// TIA Portal V17 export
// export: Created 2025-07-01T14:26:04.7163189Z, ExportSetting WithDefaults, DisplayName Totally Integrated Automation Portal, DisplayVersion V17 Update 8, DisplayName TIA Portal Openness, DisplayVersion V17 Update 8, DisplayName TIA Portal Version Control Interface, DisplayVersion V17, DisplayName SINAMICS Startdrive Advanced, DisplayVersion V17 SP2, DisplayName SINAMICS Startdrive G110M, G120, G120C, G120D, G120P, G115D, DisplayVersion V17 SP2, DisplayName SINAMICS Startdrive G130, G150, S120, S150, SINAMICS MV, S210, DisplayVersion V17 SP2, DisplayName STEP 7 Professional, DisplayVersion V17 Update 8, DisplayName SINUMERIK ONE STEP 7 Toolbox, DisplayVersion V17 Update 12, DisplayName SINUMERIK ONE PLC Basic Program Plus, DisplayVersion V17 Update 12, DisplayName SINUMERIK 840D sl STEP 7 Toolbox, DisplayVersion V17 Update 12, DisplayName STEP 7 Safety, DisplayVersion V17 Update 6, DisplayName WinCC Advanced, DisplayVersion V17 Update 8
FUNCTION "FC1032_TEST_STOP_CLADDING" : Void   // FC1032, LAD
{ S7_Optimized_Access := 'FALSE' }
AUTHOR : ETXETAR
VERSION : 1.0
// stored: AutoNumber false, IsIECCheckEnabled false, SetENOAutomatically false, UDAEnableTagReadback false
   VAR_TEMP
      AUX_START_TEST_STOP : Bool;   // AUXILIARY START TEST STOP
      OPTION_ON : Bool;   // OPTION ON
      OPTION_OFF : Bool;   // OPTION OFF
      BRAKE_TEST_AXIS_X13 : Bool;   // BRAKE TEST AXIS X13
      BRAKE_TEST_AXIS_X23 : Bool;   // BRAKE TEST AXIS X23
      BRAKE_TEST_AXIS_W11 : Bool;   // BRAKE TEST AXIS W11
      BRAKE_TEST_AXIS_Z13 : Bool;   // BRAKE TEST AXIS Z13
      BRAKE_TEST_AXIS_Z14 : Bool;   // BRAKE TEST AXIS Z14
      BRAKE_TEST_AXIS_W21 : Bool;   // BRAKE TEST AXIS W21
      BRAKE_TEST_AXIS_Z23 : Bool;   // BRAKE TEST AXIS Z23
      BRAKE_TEST_AXIS_Z24 : Bool;   // BRAKE TEST AXIS Z24
      BRAKE_TEST_AXIS_C11 : Bool;   // BRAKE TEST AXIS C11
      BRAKE_TEST_AXIS_C12 : Bool;   // BRAKE TEST AXIS C12
      BRAKE_TEST_AXIS_C13 : Bool;   // BRAKE TEST AXIS C13
      BRAKE_TEST_AXIS_C14 : Bool;   // BRAKE TEST AXIS C14
      BRAKE_TEST_AXIS_C21 : Bool;   // BRAKE TEST AXIS C21
      BRAKE_TEST_AXIS_C22 : Bool;   // BRAKE TEST AXIS C22
      BRAKE_TEST_AXIS_C23 : Bool;   // BRAKE TEST AXIS C23
      BRAKE_TEST_AXIS_C24 : Bool;   // BRAKE TEST AXIS C24
      BRAKE_TEST_AXIS_C31 : Bool;   // BRAKE TEST AXISC31
   END_VAR
   VAR CONSTANT
      FC_NUMBER : DInt := 1032;
   END_VAR
   VAR_TEMP   // added for the SCL form of the ladder/FBD networks
      _w1 : Bool;
   END_VAR
BEGIN

REGION Network 1: OPTIONS OFF
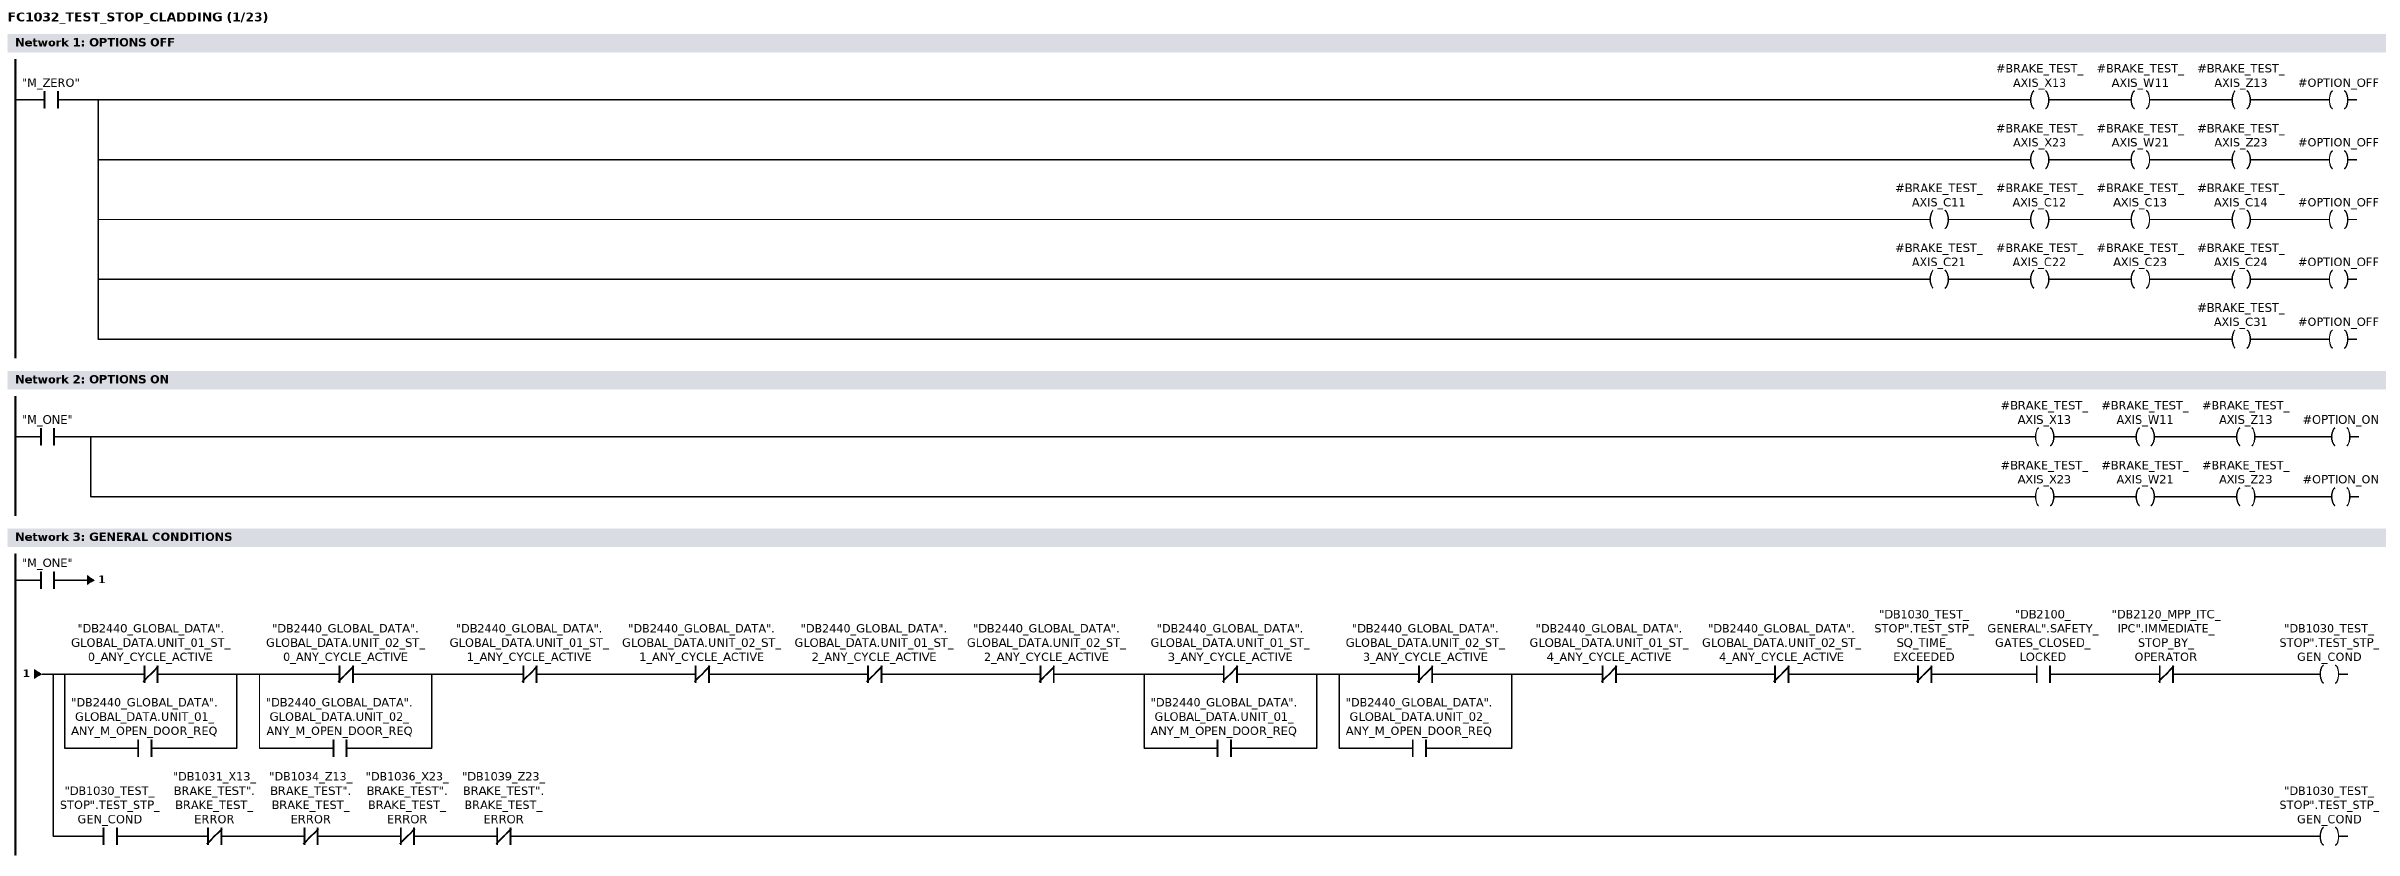
   RUNG wire#powerrail
      Contact( "M_ZERO" )
      wire#w1
      Coil( #BRAKE_TEST_AXIS_X13 )
      Coil( #BRAKE_TEST_AXIS_W11 )
      Coil( #BRAKE_TEST_AXIS_Z13 )
      Coil( #OPTION_OFF )
   END_RUNG
   RUNG wire#w1
      Coil( #BRAKE_TEST_AXIS_X23 )
      Coil( #BRAKE_TEST_AXIS_W21 )
      Coil( #BRAKE_TEST_AXIS_Z23 )
      Coil( #OPTION_OFF )
   END_RUNG
   RUNG wire#w1
      Coil( #BRAKE_TEST_AXIS_C11 )
      Coil( #BRAKE_TEST_AXIS_C12 )
      Coil( #BRAKE_TEST_AXIS_C13 )
      Coil( #BRAKE_TEST_AXIS_C14 )
      Coil( #OPTION_OFF )
   END_RUNG
   RUNG wire#w1
      Coil( #BRAKE_TEST_AXIS_C21 )
      Coil( #BRAKE_TEST_AXIS_C22 )
      Coil( #BRAKE_TEST_AXIS_C23 )
      Coil( #BRAKE_TEST_AXIS_C24 )
      Coil( #OPTION_OFF )
   END_RUNG
   RUNG wire#w1
      Coil( #BRAKE_TEST_AXIS_C31 )
      Coil( #OPTION_OFF )
   END_RUNG
   // the same network as SCL:
   #BRAKE_TEST_AXIS_X13 := "M_ZERO";
   #BRAKE_TEST_AXIS_W11 := "M_ZERO";
   #BRAKE_TEST_AXIS_Z13 := "M_ZERO";
   #OPTION_OFF := "M_ZERO";
   #BRAKE_TEST_AXIS_X23 := "M_ZERO";
   #BRAKE_TEST_AXIS_W21 := "M_ZERO";
   #BRAKE_TEST_AXIS_Z23 := "M_ZERO";
   #OPTION_OFF := "M_ZERO";
   #BRAKE_TEST_AXIS_C11 := "M_ZERO";
   #BRAKE_TEST_AXIS_C12 := "M_ZERO";
   #BRAKE_TEST_AXIS_C13 := "M_ZERO";
   #BRAKE_TEST_AXIS_C14 := "M_ZERO";
   #OPTION_OFF := "M_ZERO";
   #BRAKE_TEST_AXIS_C21 := "M_ZERO";
   #BRAKE_TEST_AXIS_C22 := "M_ZERO";
   #BRAKE_TEST_AXIS_C23 := "M_ZERO";
   #BRAKE_TEST_AXIS_C24 := "M_ZERO";
   #OPTION_OFF := "M_ZERO";
   #BRAKE_TEST_AXIS_C31 := "M_ZERO";
   #OPTION_OFF := "M_ZERO";
END_REGION

REGION Network 2: OPTIONS ON
   RUNG wire#powerrail
      Contact( "M_ONE" )
      wire#w1
      Coil( #BRAKE_TEST_AXIS_X13 )
      Coil( #BRAKE_TEST_AXIS_W11 )
      Coil( #BRAKE_TEST_AXIS_Z13 )
      Coil( #OPTION_ON )
   END_RUNG
   RUNG wire#w1
      Coil( #BRAKE_TEST_AXIS_X23 )
      Coil( #BRAKE_TEST_AXIS_W21 )
      Coil( #BRAKE_TEST_AXIS_Z23 )
      Coil( #OPTION_ON )
   END_RUNG
   // the same network as SCL:
   #BRAKE_TEST_AXIS_X13 := "M_ONE";
   #BRAKE_TEST_AXIS_W11 := "M_ONE";
   #BRAKE_TEST_AXIS_Z13 := "M_ONE";
   #OPTION_ON := "M_ONE";
   #BRAKE_TEST_AXIS_X23 := "M_ONE";
   #BRAKE_TEST_AXIS_W21 := "M_ONE";
   #BRAKE_TEST_AXIS_Z23 := "M_ONE";
   #OPTION_ON := "M_ONE";
END_REGION

REGION Network 3: GENERAL CONDITIONS
   RUNG wire#powerrail
      Contact( "M_ONE" )
      wire#w1
      I_Contact( "DB2440_GLOBAL_DATA".GLOBAL_DATA.UNIT_01_ST_0_ANY_CYCLE_ACTIVE )
      wire#w2
      I_Contact( "DB2440_GLOBAL_DATA".GLOBAL_DATA.UNIT_02_ST_0_ANY_CYCLE_ACTIVE )
      wire#w3
      I_Contact( "DB2440_GLOBAL_DATA".GLOBAL_DATA.UNIT_01_ST_1_ANY_CYCLE_ACTIVE )
      I_Contact( "DB2440_GLOBAL_DATA".GLOBAL_DATA.UNIT_02_ST_1_ANY_CYCLE_ACTIVE )
      I_Contact( "DB2440_GLOBAL_DATA".GLOBAL_DATA.UNIT_01_ST_2_ANY_CYCLE_ACTIVE )
      I_Contact( "DB2440_GLOBAL_DATA".GLOBAL_DATA.UNIT_02_ST_2_ANY_CYCLE_ACTIVE )
      wire#w4
      I_Contact( "DB2440_GLOBAL_DATA".GLOBAL_DATA.UNIT_01_ST_3_ANY_CYCLE_ACTIVE )
      wire#w5
      I_Contact( "DB2440_GLOBAL_DATA".GLOBAL_DATA.UNIT_02_ST_3_ANY_CYCLE_ACTIVE )
      wire#w6
      I_Contact( "DB2440_GLOBAL_DATA".GLOBAL_DATA.UNIT_01_ST_4_ANY_CYCLE_ACTIVE )
      I_Contact( "DB2440_GLOBAL_DATA".GLOBAL_DATA.UNIT_02_ST_4_ANY_CYCLE_ACTIVE )
      I_Contact( "DB1030_TEST_STOP".TEST_STP_SQ_TIME_EXCEEDED )
      Contact( "DB2100_GENERAL".SAFETY_GATES_CLOSED_LOCKED )
      I_Contact( "DB2120_MPP_ITC_IPC".IMMEDIATE_STOP_BY_OPERATOR )
      Coil( "DB1030_TEST_STOP".TEST_STP_GEN_COND )
   END_RUNG
   RUNG wire#w1
      Contact( "DB2440_GLOBAL_DATA".GLOBAL_DATA.UNIT_01_ANY_M_OPEN_DOOR_REQ )
   END_RUNG wire#w2
   RUNG wire#w2
      Contact( "DB2440_GLOBAL_DATA".GLOBAL_DATA.UNIT_02_ANY_M_OPEN_DOOR_REQ )
   END_RUNG wire#w3
   RUNG wire#w4
      Contact( "DB2440_GLOBAL_DATA".GLOBAL_DATA.UNIT_01_ANY_M_OPEN_DOOR_REQ )
   END_RUNG wire#w5
   RUNG wire#w5
      Contact( "DB2440_GLOBAL_DATA".GLOBAL_DATA.UNIT_02_ANY_M_OPEN_DOOR_REQ )
   END_RUNG wire#w6
   RUNG wire#w1
      Contact( "DB1030_TEST_STOP".TEST_STP_GEN_COND )
      I_Contact( "DB1031_X13_BRAKE_TEST".BRAKE_TEST_ERROR )
      I_Contact( "DB1034_Z13_BRAKE_TEST".BRAKE_TEST_ERROR )
      I_Contact( "DB1036_X23_BRAKE_TEST".BRAKE_TEST_ERROR )
      I_Contact( "DB1039_Z23_BRAKE_TEST".BRAKE_TEST_ERROR )
      Coil( "DB1030_TEST_STOP".TEST_STP_GEN_COND )
   END_RUNG
   // the same network as SCL:
   "DB1030_TEST_STOP".TEST_STP_GEN_COND := "M_ONE" AND (NOT "DB2440_GLOBAL_DATA".GLOBAL_DATA.UNIT_01_ST_0_ANY_CYCLE_ACTIVE OR "DB2440_GLOBAL_DATA".GLOBAL_DATA.UNIT_01_ANY_M_OPEN_DOOR_REQ) AND (NOT "DB2440_GLOBAL_DATA".GLOBAL_DATA.UNIT_02_ST_0_ANY_CYCLE_ACTIVE OR "DB2440_GLOBAL_DATA".GLOBAL_DATA.UNIT_02_ANY_M_OPEN_DOOR_REQ) AND NOT "DB2440_GLOBAL_DATA".GLOBAL_DATA.UNIT_01_ST_1_ANY_CYCLE_ACTIVE AND NOT "DB2440_GLOBAL_DATA".GLOBAL_DATA.UNIT_02_ST_1_ANY_CYCLE_ACTIVE AND NOT "DB2440_GLOBAL_DATA".GLOBAL_DATA.UNIT_01_ST_2_ANY_CYCLE_ACTIVE AND NOT "DB2440_GLOBAL_DATA".GLOBAL_DATA.UNIT_02_ST_2_ANY_CYCLE_ACTIVE AND (NOT "DB2440_GLOBAL_DATA".GLOBAL_DATA.UNIT_01_ST_3_ANY_CYCLE_ACTIVE OR "DB2440_GLOBAL_DATA".GLOBAL_DATA.UNIT_01_ANY_M_OPEN_DOOR_REQ) AND (NOT "DB2440_GLOBAL_DATA".GLOBAL_DATA.UNIT_02_ST_3_ANY_CYCLE_ACTIVE OR "DB2440_GLOBAL_DATA".GLOBAL_DATA.UNIT_02_ANY_M_OPEN_DOOR_REQ) AND NOT "DB2440_GLOBAL_DATA".GLOBAL_DATA.UNIT_01_ST_4_ANY_CYCLE_ACTIVE AND NOT "DB2440_GLOBAL_DATA".GLOBAL_DATA.UNIT_02_ST_4_ANY_CYCLE_ACTIVE AND NOT "DB1030_TEST_STOP".TEST_STP_SQ_TIME_EXCEEDED AND "DB2100_GENERAL".SAFETY_GATES_CLOSED_LOCKED AND NOT "DB2120_MPP_ITC_IPC".IMMEDIATE_STOP_BY_OPERATOR;
   "DB1030_TEST_STOP".TEST_STP_GEN_COND := "M_ONE" AND "DB1030_TEST_STOP".TEST_STP_GEN_COND AND NOT "DB1031_X13_BRAKE_TEST".BRAKE_TEST_ERROR AND NOT "DB1034_Z13_BRAKE_TEST".BRAKE_TEST_ERROR AND NOT "DB1036_X23_BRAKE_TEST".BRAKE_TEST_ERROR AND NOT "DB1039_Z23_BRAKE_TEST".BRAKE_TEST_ERROR;
END_REGION

REGION Network 4: INITIAL CONDITIONS
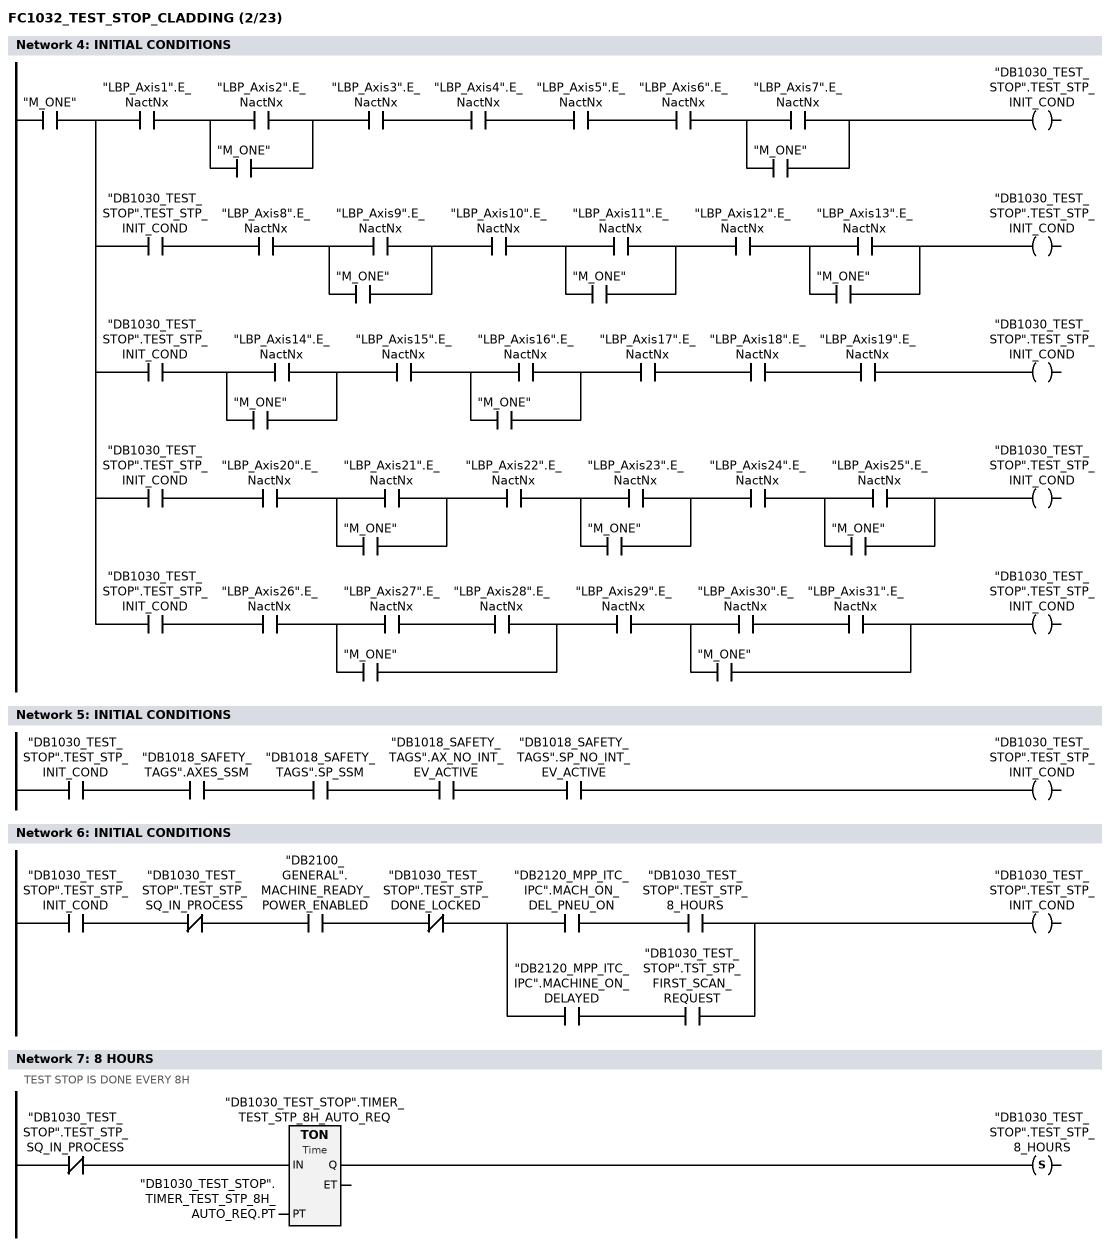
   RUNG wire#powerrail
      Contact( "M_ONE" )
      wire#w1
      Contact( "LBP_Axis1".E_NactNx )
      wire#w2
      Contact( "LBP_Axis2".E_NactNx )
      wire#w3
      Contact( "LBP_Axis3".E_NactNx )
      Contact( "LBP_Axis4".E_NactNx )
      Contact( "LBP_Axis5".E_NactNx )
      Contact( "LBP_Axis6".E_NactNx )
      wire#w4
      Contact( "LBP_Axis7".E_NactNx )
      wire#w5
      Coil( "DB1030_TEST_STOP".TEST_STP_INIT_COND )
   END_RUNG
   RUNG wire#w2
      Contact( "M_ONE" )
   END_RUNG wire#w3
   RUNG wire#w4
      Contact( "M_ONE" )
   END_RUNG wire#w5
   RUNG wire#w1
      Contact( "DB1030_TEST_STOP".TEST_STP_INIT_COND )
      Contact( "LBP_Axis8".E_NactNx )
      wire#w6
      Contact( "LBP_Axis9".E_NactNx )
      wire#w7
      Contact( "LBP_Axis10".E_NactNx )
      wire#w8
      Contact( "LBP_Axis11".E_NactNx )
      wire#w9
      Contact( "LBP_Axis12".E_NactNx )
      wire#w10
      Contact( "LBP_Axis13".E_NactNx )
      wire#w11
      Coil( "DB1030_TEST_STOP".TEST_STP_INIT_COND )
   END_RUNG
   RUNG wire#w6
      Contact( "M_ONE" )
   END_RUNG wire#w7
   RUNG wire#w8
      Contact( "M_ONE" )
   END_RUNG wire#w9
   RUNG wire#w10
      Contact( "M_ONE" )
   END_RUNG wire#w11
   RUNG wire#w1
      Contact( "DB1030_TEST_STOP".TEST_STP_INIT_COND )
      wire#w12
      Contact( "LBP_Axis14".E_NactNx )
      wire#w13
      Contact( "LBP_Axis15".E_NactNx )
      wire#w14
      Contact( "LBP_Axis16".E_NactNx )
      wire#w15
      Contact( "LBP_Axis17".E_NactNx )
      Contact( "LBP_Axis18".E_NactNx )
      Contact( "LBP_Axis19".E_NactNx )
      Coil( "DB1030_TEST_STOP".TEST_STP_INIT_COND )
   END_RUNG
   RUNG wire#w12
      Contact( "M_ONE" )
   END_RUNG wire#w13
   RUNG wire#w14
      Contact( "M_ONE" )
   END_RUNG wire#w15
   RUNG wire#w1
      Contact( "DB1030_TEST_STOP".TEST_STP_INIT_COND )
      Contact( "LBP_Axis20".E_NactNx )
      wire#w16
      Contact( "LBP_Axis21".E_NactNx )
      wire#w17
      Contact( "LBP_Axis22".E_NactNx )
      wire#w18
      Contact( "LBP_Axis23".E_NactNx )
      wire#w19
      Contact( "LBP_Axis24".E_NactNx )
      wire#w20
      Contact( "LBP_Axis25".E_NactNx )
      wire#w21
      Coil( "DB1030_TEST_STOP".TEST_STP_INIT_COND )
   END_RUNG
   RUNG wire#w16
      Contact( "M_ONE" )
   END_RUNG wire#w17
   RUNG wire#w18
      Contact( "M_ONE" )
   END_RUNG wire#w19
   RUNG wire#w20
      Contact( "M_ONE" )
   END_RUNG wire#w21
   RUNG wire#w1
      Contact( "DB1030_TEST_STOP".TEST_STP_INIT_COND )
      Contact( "LBP_Axis26".E_NactNx )
      wire#w22
      Contact( "LBP_Axis27".E_NactNx )
      Contact( "LBP_Axis28".E_NactNx )
      wire#w23
      Contact( "LBP_Axis29".E_NactNx )
      wire#w24
      Contact( "LBP_Axis30".E_NactNx )
      Contact( "LBP_Axis31".E_NactNx )
      wire#w25
      Coil( "DB1030_TEST_STOP".TEST_STP_INIT_COND )
   END_RUNG
   RUNG wire#w22
      Contact( "M_ONE" )
   END_RUNG wire#w23
   RUNG wire#w24
      Contact( "M_ONE" )
   END_RUNG wire#w25
   // the same network as SCL:
   "DB1030_TEST_STOP".TEST_STP_INIT_COND := "M_ONE" AND "LBP_Axis1".E_NactNx AND ("LBP_Axis2".E_NactNx OR "M_ONE") AND "LBP_Axis3".E_NactNx AND "LBP_Axis4".E_NactNx AND "LBP_Axis5".E_NactNx AND "LBP_Axis6".E_NactNx AND ("LBP_Axis7".E_NactNx OR "M_ONE");
   "DB1030_TEST_STOP".TEST_STP_INIT_COND := "M_ONE" AND "DB1030_TEST_STOP".TEST_STP_INIT_COND AND "LBP_Axis8".E_NactNx AND ("LBP_Axis9".E_NactNx OR "M_ONE") AND "LBP_Axis10".E_NactNx AND ("LBP_Axis11".E_NactNx OR "M_ONE") AND "LBP_Axis12".E_NactNx AND ("LBP_Axis13".E_NactNx OR "M_ONE");
   "DB1030_TEST_STOP".TEST_STP_INIT_COND := "M_ONE" AND "DB1030_TEST_STOP".TEST_STP_INIT_COND AND ("LBP_Axis14".E_NactNx OR "M_ONE") AND "LBP_Axis15".E_NactNx AND ("LBP_Axis16".E_NactNx OR "M_ONE") AND "LBP_Axis17".E_NactNx AND "LBP_Axis18".E_NactNx AND "LBP_Axis19".E_NactNx;
   "DB1030_TEST_STOP".TEST_STP_INIT_COND := "M_ONE" AND "DB1030_TEST_STOP".TEST_STP_INIT_COND AND "LBP_Axis20".E_NactNx AND ("LBP_Axis21".E_NactNx OR "M_ONE") AND "LBP_Axis22".E_NactNx AND ("LBP_Axis23".E_NactNx OR "M_ONE") AND "LBP_Axis24".E_NactNx AND ("LBP_Axis25".E_NactNx OR "M_ONE");
   "DB1030_TEST_STOP".TEST_STP_INIT_COND := "M_ONE" AND "DB1030_TEST_STOP".TEST_STP_INIT_COND AND "LBP_Axis26".E_NactNx AND (("LBP_Axis27".E_NactNx AND "LBP_Axis28".E_NactNx) OR "M_ONE") AND "LBP_Axis29".E_NactNx AND (("LBP_Axis30".E_NactNx AND "LBP_Axis31".E_NactNx) OR "M_ONE");
END_REGION

REGION Network 5: INITIAL CONDITIONS
   RUNG wire#powerrail
      Contact( "DB1030_TEST_STOP".TEST_STP_INIT_COND )
      Contact( "DB1018_SAFETY_TAGS".AXES_SSM )
      Contact( "DB1018_SAFETY_TAGS".SP_SSM )
      Contact( "DB1018_SAFETY_TAGS".AX_NO_INT_EV_ACTIVE )
      Contact( "DB1018_SAFETY_TAGS".SP_NO_INT_EV_ACTIVE )
      Coil( "DB1030_TEST_STOP".TEST_STP_INIT_COND )
   END_RUNG
   // the same network as SCL:
   "DB1030_TEST_STOP".TEST_STP_INIT_COND := "DB1030_TEST_STOP".TEST_STP_INIT_COND AND "DB1018_SAFETY_TAGS".AXES_SSM AND "DB1018_SAFETY_TAGS".SP_SSM AND "DB1018_SAFETY_TAGS".AX_NO_INT_EV_ACTIVE AND "DB1018_SAFETY_TAGS".SP_NO_INT_EV_ACTIVE;
END_REGION

REGION Network 6: INITIAL CONDITIONS
   RUNG wire#powerrail
      Contact( "DB1030_TEST_STOP".TEST_STP_INIT_COND )
      I_Contact( "DB1030_TEST_STOP".TEST_STP_SQ_IN_PROCESS )
      Contact( "DB2100_GENERAL".MACHINE_READY_POWER_ENABLED )
      I_Contact( "DB1030_TEST_STOP".TEST_STP_DONE_LOCKED )
      wire#w1
      Contact( "DB2120_MPP_ITC_IPC".MACH_ON_DEL_PNEU_ON )
      Contact( "DB1030_TEST_STOP".TEST_STP_8_HOURS )
      wire#w2
      Coil( "DB1030_TEST_STOP".TEST_STP_INIT_COND )
   END_RUNG
   RUNG wire#w1
      Contact( "DB2120_MPP_ITC_IPC".MACHINE_ON_DELAYED )
      Contact( "DB1030_TEST_STOP".TST_STP_FIRST_SCAN_REQUEST )
   END_RUNG wire#w2
   // the same network as SCL:
   "DB1030_TEST_STOP".TEST_STP_INIT_COND := "DB1030_TEST_STOP".TEST_STP_INIT_COND AND NOT "DB1030_TEST_STOP".TEST_STP_SQ_IN_PROCESS AND "DB2100_GENERAL".MACHINE_READY_POWER_ENABLED AND NOT "DB1030_TEST_STOP".TEST_STP_DONE_LOCKED AND (("DB2120_MPP_ITC_IPC".MACH_ON_DEL_PNEU_ON AND "DB1030_TEST_STOP".TEST_STP_8_HOURS) OR ("DB2120_MPP_ITC_IPC".MACHINE_ON_DELAYED AND "DB1030_TEST_STOP".TST_STP_FIRST_SCAN_REQUEST));
END_REGION

REGION Network 7: 8 HOURS
   // TEST STOP IS DONE EVERY 8H
   RUNG wire#powerrail
      I_Contact( "DB1030_TEST_STOP".TEST_STP_SQ_IN_PROCESS )
      { S7_Templates := "time_type := Time" } "DB1030_TEST_STOP".TIMER_TEST_STP_8H_AUTO_REQ.TON(pt := "DB1030_TEST_STOP".TIMER_TEST_STP_8H_AUTO_REQ.PT, et =>)
      S_Coil( "DB1030_TEST_STOP".TEST_STP_8_HOURS )
   END_RUNG
   // the same network as SCL:
   "DB1030_TEST_STOP".TIMER_TEST_STP_8H_AUTO_REQ.TON(IN := NOT "DB1030_TEST_STOP".TEST_STP_SQ_IN_PROCESS,
                           PT := "DB1030_TEST_STOP".TIMER_TEST_STP_8H_AUTO_REQ.PT);
   IF "DB1030_TEST_STOP".TIMER_TEST_STP_8H_AUTO_REQ.Q THEN
       "DB1030_TEST_STOP".TEST_STP_8_HOURS := TRUE;
   END_IF;
END_REGION

REGION Network 8: START REQUEST
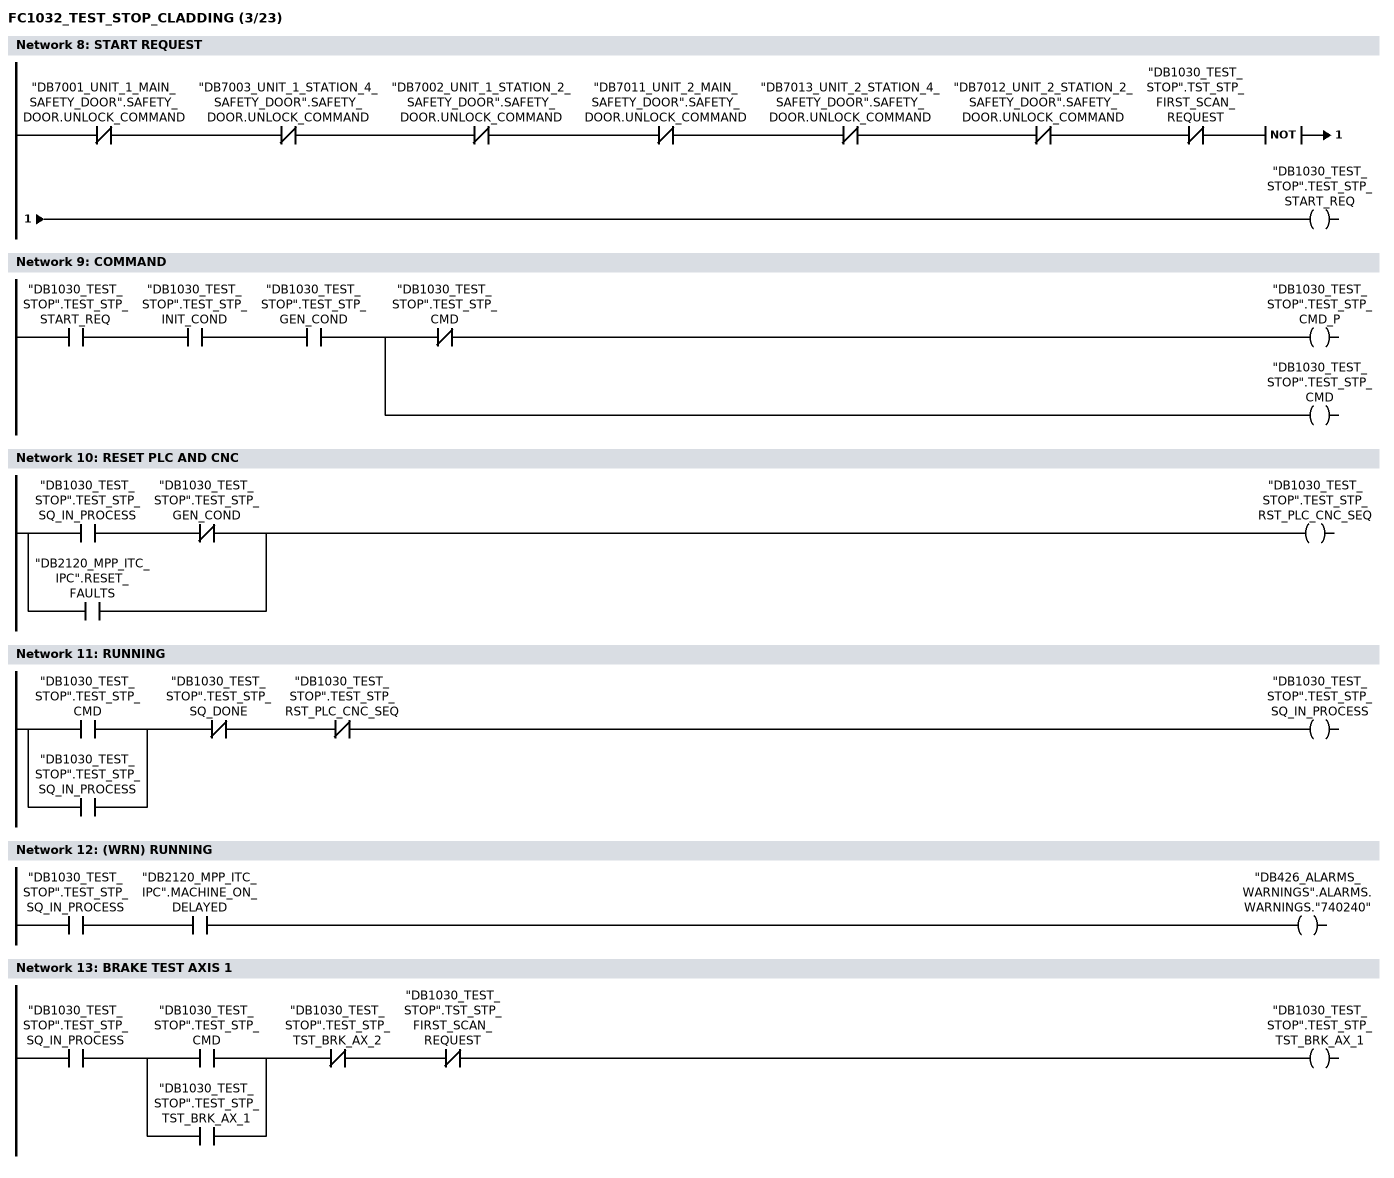
   RUNG wire#powerrail
      I_Contact( "DB7001_UNIT_1_MAIN_SAFETY_DOOR".SAFETY_DOOR.UNLOCK_COMMAND )
      I_Contact( "DB7003_UNIT_1_STATION_4_SAFETY_DOOR".SAFETY_DOOR.UNLOCK_COMMAND )
      I_Contact( "DB7002_UNIT_1_STATION_2_SAFETY_DOOR".SAFETY_DOOR.UNLOCK_COMMAND )
      I_Contact( "DB7011_UNIT_2_MAIN_SAFETY_DOOR".SAFETY_DOOR.UNLOCK_COMMAND )
      I_Contact( "DB7013_UNIT_2_STATION_4_SAFETY_DOOR".SAFETY_DOOR.UNLOCK_COMMAND )
      I_Contact( "DB7012_UNIT_2_STATION_2_SAFETY_DOOR".SAFETY_DOOR.UNLOCK_COMMAND )
      I_Contact( "DB1030_TEST_STOP".TST_STP_FIRST_SCAN_REQUEST )
      Not()
      Coil( "DB1030_TEST_STOP".TEST_STP_START_REQ )
   END_RUNG
   // the same network as SCL:
   "DB1030_TEST_STOP".TEST_STP_START_REQ := NOT (NOT "DB7001_UNIT_1_MAIN_SAFETY_DOOR".SAFETY_DOOR.UNLOCK_COMMAND AND NOT "DB7003_UNIT_1_STATION_4_SAFETY_DOOR".SAFETY_DOOR.UNLOCK_COMMAND AND NOT "DB7002_UNIT_1_STATION_2_SAFETY_DOOR".SAFETY_DOOR.UNLOCK_COMMAND AND NOT "DB7011_UNIT_2_MAIN_SAFETY_DOOR".SAFETY_DOOR.UNLOCK_COMMAND AND NOT "DB7013_UNIT_2_STATION_4_SAFETY_DOOR".SAFETY_DOOR.UNLOCK_COMMAND AND NOT "DB7012_UNIT_2_STATION_2_SAFETY_DOOR".SAFETY_DOOR.UNLOCK_COMMAND AND NOT "DB1030_TEST_STOP".TST_STP_FIRST_SCAN_REQUEST);
END_REGION

REGION Network 9: COMMAND
   RUNG wire#powerrail
      Contact( "DB1030_TEST_STOP".TEST_STP_START_REQ )
      Contact( "DB1030_TEST_STOP".TEST_STP_INIT_COND )
      Contact( "DB1030_TEST_STOP".TEST_STP_GEN_COND )
      wire#w1
      I_Contact( "DB1030_TEST_STOP".TEST_STP_CMD )
      Coil( "DB1030_TEST_STOP".TEST_STP_CMD_P )
   END_RUNG
   RUNG wire#w1
      Coil( "DB1030_TEST_STOP".TEST_STP_CMD )
   END_RUNG
   // the same network as SCL:
   #_w1 := "DB1030_TEST_STOP".TEST_STP_START_REQ AND "DB1030_TEST_STOP".TEST_STP_INIT_COND AND "DB1030_TEST_STOP".TEST_STP_GEN_COND;
   "DB1030_TEST_STOP".TEST_STP_CMD_P := #_w1 AND NOT "DB1030_TEST_STOP".TEST_STP_CMD;
   "DB1030_TEST_STOP".TEST_STP_CMD := #_w1;
END_REGION

REGION Network 10: RESET PLC AND CNC
   RUNG wire#powerrail
      Contact( "DB1030_TEST_STOP".TEST_STP_SQ_IN_PROCESS )
      I_Contact( "DB1030_TEST_STOP".TEST_STP_GEN_COND )
      wire#w1
      Coil( "DB1030_TEST_STOP".TEST_STP_RST_PLC_CNC_SEQ )
   END_RUNG
   RUNG wire#powerrail
      Contact( "DB2120_MPP_ITC_IPC".RESET_FAULTS )
   END_RUNG wire#w1
   // the same network as SCL:
   "DB1030_TEST_STOP".TEST_STP_RST_PLC_CNC_SEQ := ("DB1030_TEST_STOP".TEST_STP_SQ_IN_PROCESS AND NOT "DB1030_TEST_STOP".TEST_STP_GEN_COND) OR "DB2120_MPP_ITC_IPC".RESET_FAULTS;
END_REGION

REGION Network 11: RUNNING
   RUNG wire#powerrail
      Contact( "DB1030_TEST_STOP".TEST_STP_CMD )
      wire#w1
      I_Contact( "DB1030_TEST_STOP".TEST_STP_SQ_DONE )
      I_Contact( "DB1030_TEST_STOP".TEST_STP_RST_PLC_CNC_SEQ )
      Coil( "DB1030_TEST_STOP".TEST_STP_SQ_IN_PROCESS )
   END_RUNG
   RUNG wire#powerrail
      Contact( "DB1030_TEST_STOP".TEST_STP_SQ_IN_PROCESS )
   END_RUNG wire#w1
   // the same network as SCL:
   "DB1030_TEST_STOP".TEST_STP_SQ_IN_PROCESS := ("DB1030_TEST_STOP".TEST_STP_CMD OR "DB1030_TEST_STOP".TEST_STP_SQ_IN_PROCESS) AND NOT "DB1030_TEST_STOP".TEST_STP_SQ_DONE AND NOT "DB1030_TEST_STOP".TEST_STP_RST_PLC_CNC_SEQ;
END_REGION

REGION Network 12: (WRN) RUNNING
   RUNG wire#powerrail
      Contact( "DB1030_TEST_STOP".TEST_STP_SQ_IN_PROCESS )
      Contact( "DB2120_MPP_ITC_IPC".MACHINE_ON_DELAYED )
      Coil( "DB426_ALARMS_WARNINGS".ALARMS.WARNINGS."740240" )
   END_RUNG
   // the same network as SCL:
   "DB426_ALARMS_WARNINGS".ALARMS.WARNINGS."740240" := "DB1030_TEST_STOP".TEST_STP_SQ_IN_PROCESS AND "DB2120_MPP_ITC_IPC".MACHINE_ON_DELAYED;
END_REGION

REGION Network 13: BRAKE TEST AXIS 1
   RUNG wire#powerrail
      Contact( "DB1030_TEST_STOP".TEST_STP_SQ_IN_PROCESS )
      wire#w1
      Contact( "DB1030_TEST_STOP".TEST_STP_CMD )
      wire#w2
      I_Contact( "DB1030_TEST_STOP".TEST_STP_TST_BRK_AX_2 )
      I_Contact( "DB1030_TEST_STOP".TST_STP_FIRST_SCAN_REQUEST )
      Coil( "DB1030_TEST_STOP".TEST_STP_TST_BRK_AX_1 )
   END_RUNG
   RUNG wire#w1
      Contact( "DB1030_TEST_STOP".TEST_STP_TST_BRK_AX_1 )
   END_RUNG wire#w2
   // the same network as SCL:
   "DB1030_TEST_STOP".TEST_STP_TST_BRK_AX_1 := "DB1030_TEST_STOP".TEST_STP_SQ_IN_PROCESS AND ("DB1030_TEST_STOP".TEST_STP_CMD OR "DB1030_TEST_STOP".TEST_STP_TST_BRK_AX_1) AND NOT "DB1030_TEST_STOP".TEST_STP_TST_BRK_AX_2 AND NOT "DB1030_TEST_STOP".TST_STP_FIRST_SCAN_REQUEST;
END_REGION

REGION Network 14: CALL FB1031 BRAKE TEST AXIS 1
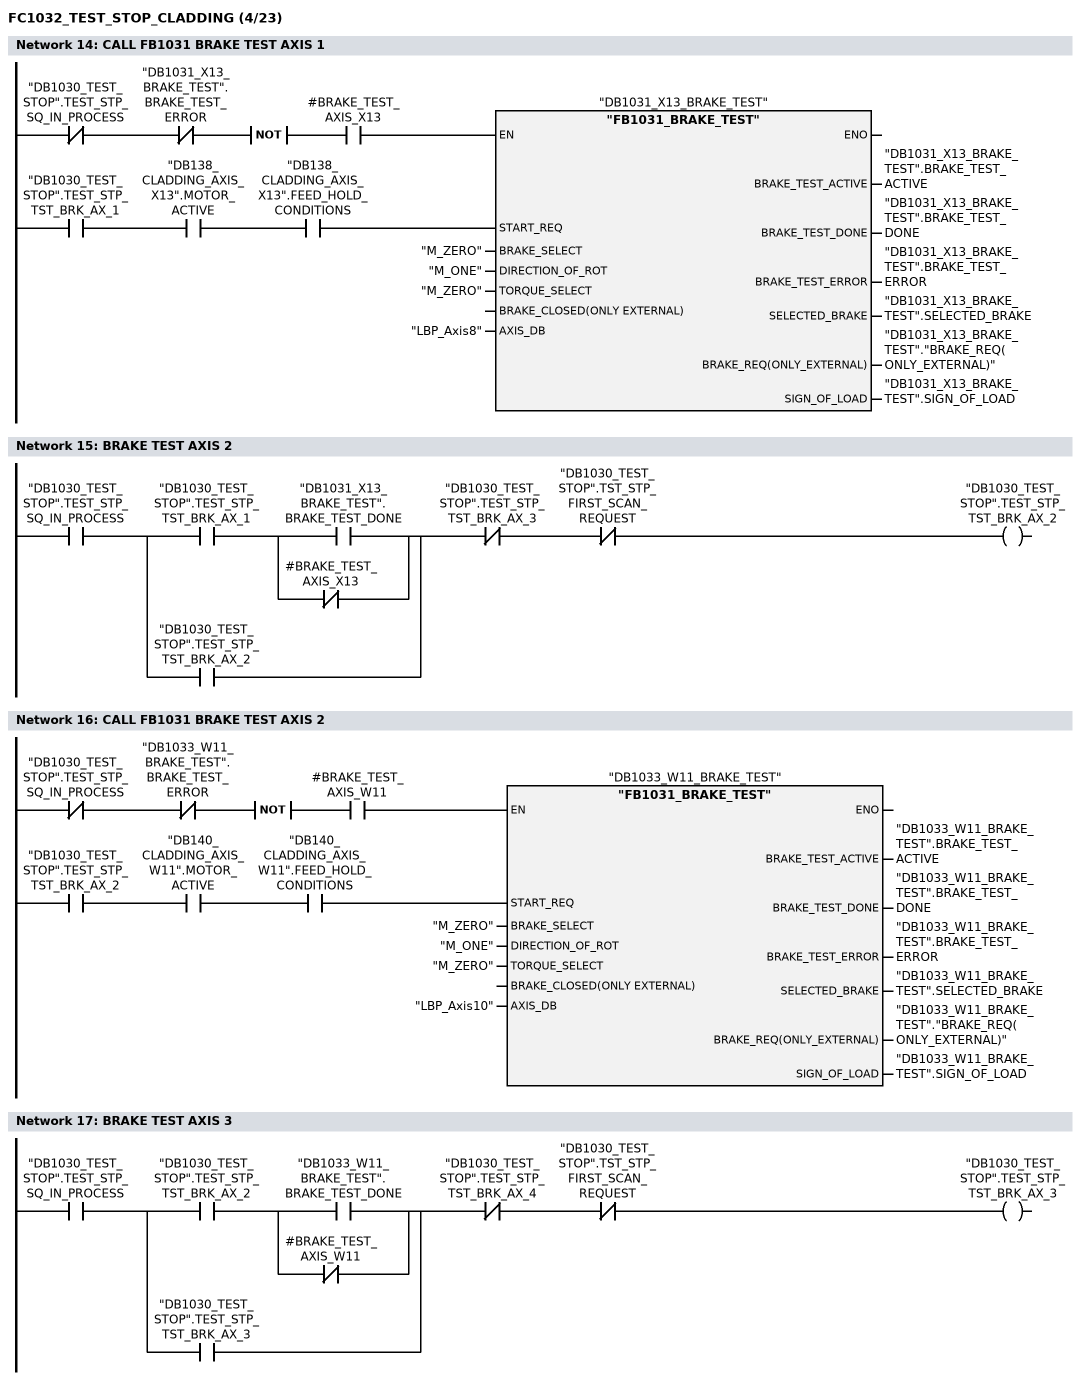
   RUNG wire#powerrail
      I_Contact( "DB1030_TEST_STOP".TEST_STP_SQ_IN_PROCESS )
      I_Contact( "DB1031_X13_BRAKE_TEST".BRAKE_TEST_ERROR )
      Not()
      Contact( #BRAKE_TEST_AXIS_X13 )
      "DB1031_X13_BRAKE_TEST"(START_REQ := wire#w1, BRAKE_SELECT := "M_ZERO", DIRECTION_OF_ROT := "M_ONE", TORQUE_SELECT := "M_ZERO", "BRAKE_CLOSED(ONLY EXTERNAL)" :=, AXIS_DB := "LBP_Axis8", BRAKE_TEST_ACTIVE => "DB1031_X13_BRAKE_TEST".BRAKE_TEST_ACTIVE, BRAKE_TEST_DONE => "DB1031_X13_BRAKE_TEST".BRAKE_TEST_DONE, BRAKE_TEST_ERROR => "DB1031_X13_BRAKE_TEST".BRAKE_TEST_ERROR, SELECTED_BRAKE => "DB1031_X13_BRAKE_TEST".SELECTED_BRAKE, "BRAKE_REQ(ONLY_EXTERNAL)" => "DB1031_X13_BRAKE_TEST"."BRAKE_REQ(ONLY_EXTERNAL)", SIGN_OF_LOAD => "DB1031_X13_BRAKE_TEST".SIGN_OF_LOAD)
   END_RUNG
   RUNG wire#powerrail
      Contact( "DB1030_TEST_STOP".TEST_STP_TST_BRK_AX_1 )
      Contact( "DB138_CLADDING_AXIS_X13".MOTOR_ACTIVE )
      Contact( "DB138_CLADDING_AXIS_X13".FEED_HOLD_CONDITIONS )
   END_RUNG wire#w1
   // the same network as SCL:
   IF NOT (NOT "DB1030_TEST_STOP".TEST_STP_SQ_IN_PROCESS AND NOT "DB1031_X13_BRAKE_TEST".BRAKE_TEST_ERROR) AND #BRAKE_TEST_AXIS_X13 THEN
       "DB1031_X13_BRAKE_TEST"(START_REQ := "DB1030_TEST_STOP".TEST_STP_TST_BRK_AX_1 AND "DB138_CLADDING_AXIS_X13".MOTOR_ACTIVE AND "DB138_CLADDING_AXIS_X13".FEED_HOLD_CONDITIONS,   // "FB1031_BRAKE_TEST"
                               BRAKE_SELECT := "M_ZERO",
                               DIRECTION_OF_ROT := "M_ONE",
                               TORQUE_SELECT := "M_ZERO",
                               AXIS_DB := "LBP_Axis8",
                               BRAKE_TEST_ACTIVE => "DB1031_X13_BRAKE_TEST".BRAKE_TEST_ACTIVE,
                               BRAKE_TEST_DONE => "DB1031_X13_BRAKE_TEST".BRAKE_TEST_DONE,
                               BRAKE_TEST_ERROR => "DB1031_X13_BRAKE_TEST".BRAKE_TEST_ERROR,
                               SELECTED_BRAKE => "DB1031_X13_BRAKE_TEST".SELECTED_BRAKE,
                               "BRAKE_REQ(ONLY_EXTERNAL)" => "DB1031_X13_BRAKE_TEST"."BRAKE_REQ(ONLY_EXTERNAL)",
                               SIGN_OF_LOAD => "DB1031_X13_BRAKE_TEST".SIGN_OF_LOAD);
   END_IF;
END_REGION

REGION Network 15: BRAKE TEST AXIS 2
   RUNG wire#powerrail
      Contact( "DB1030_TEST_STOP".TEST_STP_SQ_IN_PROCESS )
      wire#w1
      Contact( "DB1030_TEST_STOP".TEST_STP_TST_BRK_AX_1 )
      wire#w2
      Contact( "DB1031_X13_BRAKE_TEST".BRAKE_TEST_DONE )
      wire#w3
      I_Contact( "DB1030_TEST_STOP".TEST_STP_TST_BRK_AX_3 )
      I_Contact( "DB1030_TEST_STOP".TST_STP_FIRST_SCAN_REQUEST )
      Coil( "DB1030_TEST_STOP".TEST_STP_TST_BRK_AX_2 )
   END_RUNG
   RUNG wire#w2
      I_Contact( #BRAKE_TEST_AXIS_X13 )
   END_RUNG wire#w3
   RUNG wire#w1
      Contact( "DB1030_TEST_STOP".TEST_STP_TST_BRK_AX_2 )
   END_RUNG wire#w3
   // the same network as SCL:
   "DB1030_TEST_STOP".TEST_STP_TST_BRK_AX_2 := "DB1030_TEST_STOP".TEST_STP_SQ_IN_PROCESS AND (("DB1030_TEST_STOP".TEST_STP_TST_BRK_AX_1 AND ("DB1031_X13_BRAKE_TEST".BRAKE_TEST_DONE OR NOT #BRAKE_TEST_AXIS_X13)) OR "DB1030_TEST_STOP".TEST_STP_TST_BRK_AX_2) AND NOT "DB1030_TEST_STOP".TEST_STP_TST_BRK_AX_3 AND NOT "DB1030_TEST_STOP".TST_STP_FIRST_SCAN_REQUEST;
END_REGION

REGION Network 16: CALL FB1031 BRAKE TEST AXIS 2
   RUNG wire#powerrail
      I_Contact( "DB1030_TEST_STOP".TEST_STP_SQ_IN_PROCESS )
      I_Contact( "DB1033_W11_BRAKE_TEST".BRAKE_TEST_ERROR )
      Not()
      Contact( #BRAKE_TEST_AXIS_W11 )
      "DB1033_W11_BRAKE_TEST"(START_REQ := wire#w1, BRAKE_SELECT := "M_ZERO", DIRECTION_OF_ROT := "M_ONE", TORQUE_SELECT := "M_ZERO", "BRAKE_CLOSED(ONLY EXTERNAL)" :=, AXIS_DB := "LBP_Axis10", BRAKE_TEST_ACTIVE => "DB1033_W11_BRAKE_TEST".BRAKE_TEST_ACTIVE, BRAKE_TEST_DONE => "DB1033_W11_BRAKE_TEST".BRAKE_TEST_DONE, BRAKE_TEST_ERROR => "DB1033_W11_BRAKE_TEST".BRAKE_TEST_ERROR, SELECTED_BRAKE => "DB1033_W11_BRAKE_TEST".SELECTED_BRAKE, "BRAKE_REQ(ONLY_EXTERNAL)" => "DB1033_W11_BRAKE_TEST"."BRAKE_REQ(ONLY_EXTERNAL)", SIGN_OF_LOAD => "DB1033_W11_BRAKE_TEST".SIGN_OF_LOAD)
   END_RUNG
   RUNG wire#powerrail
      Contact( "DB1030_TEST_STOP".TEST_STP_TST_BRK_AX_2 )
      Contact( "DB140_CLADDING_AXIS_W11".MOTOR_ACTIVE )
      Contact( "DB140_CLADDING_AXIS_W11".FEED_HOLD_CONDITIONS )
   END_RUNG wire#w1
   // the same network as SCL:
   IF NOT (NOT "DB1030_TEST_STOP".TEST_STP_SQ_IN_PROCESS AND NOT "DB1033_W11_BRAKE_TEST".BRAKE_TEST_ERROR) AND #BRAKE_TEST_AXIS_W11 THEN
       "DB1033_W11_BRAKE_TEST"(START_REQ := "DB1030_TEST_STOP".TEST_STP_TST_BRK_AX_2 AND "DB140_CLADDING_AXIS_W11".MOTOR_ACTIVE AND "DB140_CLADDING_AXIS_W11".FEED_HOLD_CONDITIONS,   // "FB1031_BRAKE_TEST"
                               BRAKE_SELECT := "M_ZERO",
                               DIRECTION_OF_ROT := "M_ONE",
                               TORQUE_SELECT := "M_ZERO",
                               AXIS_DB := "LBP_Axis10",
                               BRAKE_TEST_ACTIVE => "DB1033_W11_BRAKE_TEST".BRAKE_TEST_ACTIVE,
                               BRAKE_TEST_DONE => "DB1033_W11_BRAKE_TEST".BRAKE_TEST_DONE,
                               BRAKE_TEST_ERROR => "DB1033_W11_BRAKE_TEST".BRAKE_TEST_ERROR,
                               SELECTED_BRAKE => "DB1033_W11_BRAKE_TEST".SELECTED_BRAKE,
                               "BRAKE_REQ(ONLY_EXTERNAL)" => "DB1033_W11_BRAKE_TEST"."BRAKE_REQ(ONLY_EXTERNAL)",
                               SIGN_OF_LOAD => "DB1033_W11_BRAKE_TEST".SIGN_OF_LOAD);
   END_IF;
END_REGION

REGION Network 17: BRAKE TEST AXIS 3
   RUNG wire#powerrail
      Contact( "DB1030_TEST_STOP".TEST_STP_SQ_IN_PROCESS )
      wire#w1
      Contact( "DB1030_TEST_STOP".TEST_STP_TST_BRK_AX_2 )
      wire#w2
      Contact( "DB1033_W11_BRAKE_TEST".BRAKE_TEST_DONE )
      wire#w3
      I_Contact( "DB1030_TEST_STOP".TEST_STP_TST_BRK_AX_4 )
      I_Contact( "DB1030_TEST_STOP".TST_STP_FIRST_SCAN_REQUEST )
      Coil( "DB1030_TEST_STOP".TEST_STP_TST_BRK_AX_3 )
   END_RUNG
   RUNG wire#w2
      I_Contact( #BRAKE_TEST_AXIS_W11 )
   END_RUNG wire#w3
   RUNG wire#w1
      Contact( "DB1030_TEST_STOP".TEST_STP_TST_BRK_AX_3 )
   END_RUNG wire#w3
   // the same network as SCL:
   "DB1030_TEST_STOP".TEST_STP_TST_BRK_AX_3 := "DB1030_TEST_STOP".TEST_STP_SQ_IN_PROCESS AND (("DB1030_TEST_STOP".TEST_STP_TST_BRK_AX_2 AND ("DB1033_W11_BRAKE_TEST".BRAKE_TEST_DONE OR NOT #BRAKE_TEST_AXIS_W11)) OR "DB1030_TEST_STOP".TEST_STP_TST_BRK_AX_3) AND NOT "DB1030_TEST_STOP".TEST_STP_TST_BRK_AX_4 AND NOT "DB1030_TEST_STOP".TST_STP_FIRST_SCAN_REQUEST;
END_REGION

REGION Network 18: CALL FB1031 BRAKE TEST AXIS 3
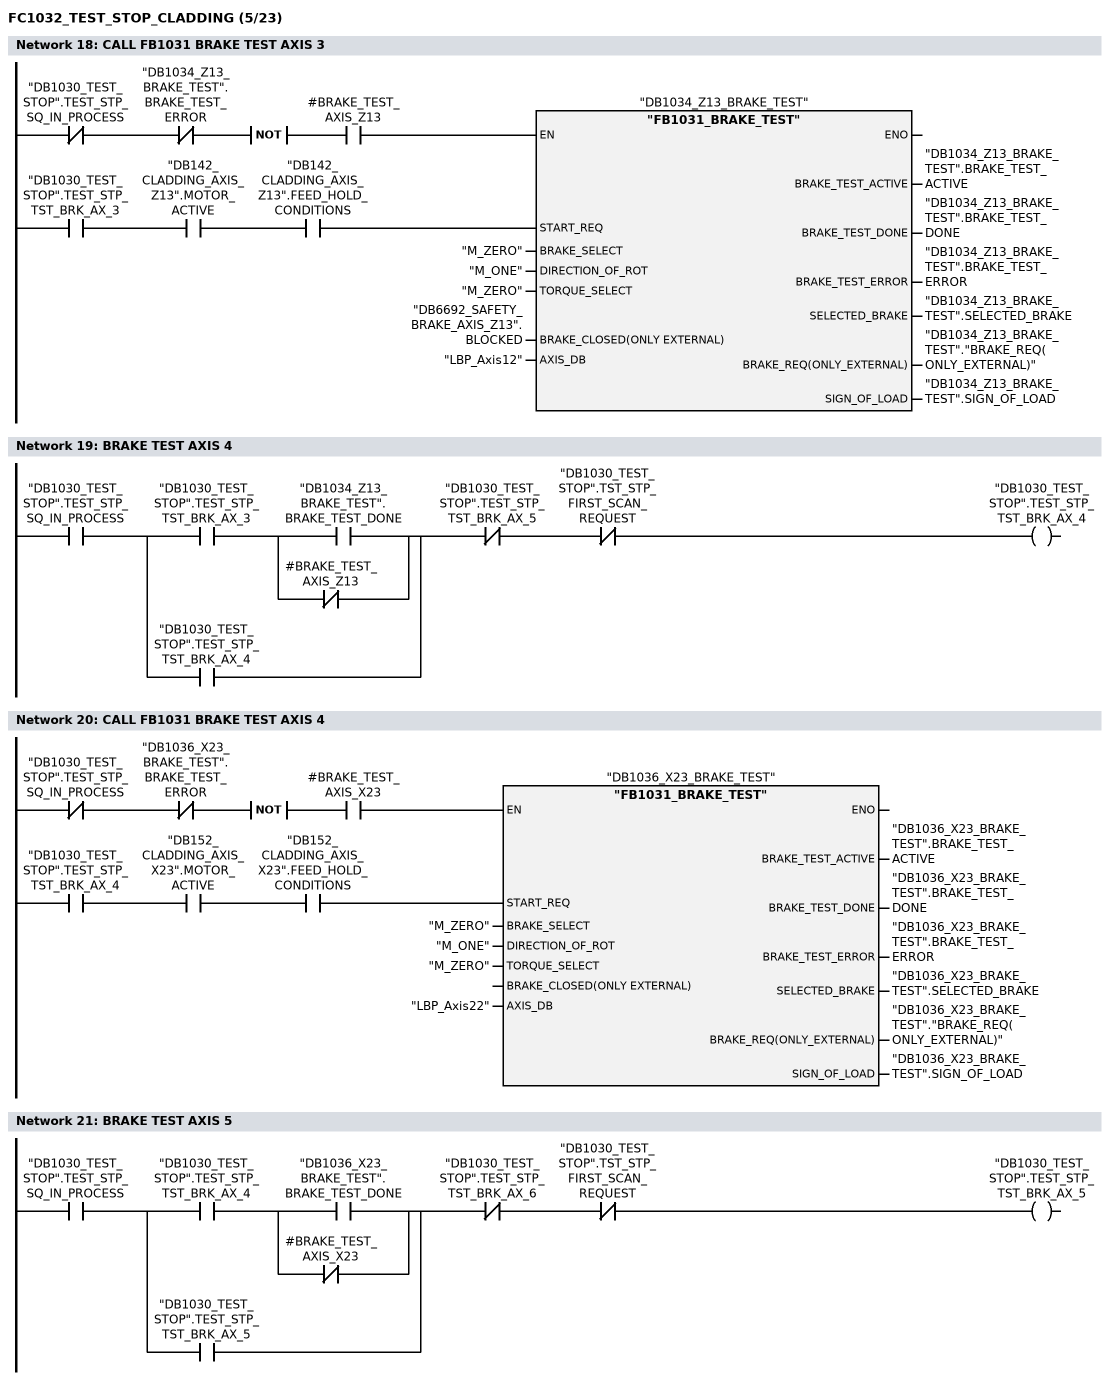
   RUNG wire#powerrail
      I_Contact( "DB1030_TEST_STOP".TEST_STP_SQ_IN_PROCESS )
      I_Contact( "DB1034_Z13_BRAKE_TEST".BRAKE_TEST_ERROR )
      Not()
      Contact( #BRAKE_TEST_AXIS_Z13 )
      "DB1034_Z13_BRAKE_TEST"(START_REQ := wire#w1, BRAKE_SELECT := "M_ZERO", DIRECTION_OF_ROT := "M_ONE", TORQUE_SELECT := "M_ZERO", "BRAKE_CLOSED(ONLY EXTERNAL)" := "DB6692_SAFETY_BRAKE_AXIS_Z13".BLOCKED, AXIS_DB := "LBP_Axis12", BRAKE_TEST_ACTIVE => "DB1034_Z13_BRAKE_TEST".BRAKE_TEST_ACTIVE, BRAKE_TEST_DONE => "DB1034_Z13_BRAKE_TEST".BRAKE_TEST_DONE, BRAKE_TEST_ERROR => "DB1034_Z13_BRAKE_TEST".BRAKE_TEST_ERROR, SELECTED_BRAKE => "DB1034_Z13_BRAKE_TEST".SELECTED_BRAKE, "BRAKE_REQ(ONLY_EXTERNAL)" => "DB1034_Z13_BRAKE_TEST"."BRAKE_REQ(ONLY_EXTERNAL)", SIGN_OF_LOAD => "DB1034_Z13_BRAKE_TEST".SIGN_OF_LOAD)
   END_RUNG
   RUNG wire#powerrail
      Contact( "DB1030_TEST_STOP".TEST_STP_TST_BRK_AX_3 )
      Contact( "DB142_CLADDING_AXIS_Z13".MOTOR_ACTIVE )
      Contact( "DB142_CLADDING_AXIS_Z13".FEED_HOLD_CONDITIONS )
   END_RUNG wire#w1
   // the same network as SCL:
   IF NOT (NOT "DB1030_TEST_STOP".TEST_STP_SQ_IN_PROCESS AND NOT "DB1034_Z13_BRAKE_TEST".BRAKE_TEST_ERROR) AND #BRAKE_TEST_AXIS_Z13 THEN
       "DB1034_Z13_BRAKE_TEST"(START_REQ := "DB1030_TEST_STOP".TEST_STP_TST_BRK_AX_3 AND "DB142_CLADDING_AXIS_Z13".MOTOR_ACTIVE AND "DB142_CLADDING_AXIS_Z13".FEED_HOLD_CONDITIONS,   // "FB1031_BRAKE_TEST"
                               BRAKE_SELECT := "M_ZERO",
                               DIRECTION_OF_ROT := "M_ONE",
                               TORQUE_SELECT := "M_ZERO",
                               "BRAKE_CLOSED(ONLY EXTERNAL)" := "DB6692_SAFETY_BRAKE_AXIS_Z13".BLOCKED,
                               AXIS_DB := "LBP_Axis12",
                               BRAKE_TEST_ACTIVE => "DB1034_Z13_BRAKE_TEST".BRAKE_TEST_ACTIVE,
                               BRAKE_TEST_DONE => "DB1034_Z13_BRAKE_TEST".BRAKE_TEST_DONE,
                               BRAKE_TEST_ERROR => "DB1034_Z13_BRAKE_TEST".BRAKE_TEST_ERROR,
                               SELECTED_BRAKE => "DB1034_Z13_BRAKE_TEST".SELECTED_BRAKE,
                               "BRAKE_REQ(ONLY_EXTERNAL)" => "DB1034_Z13_BRAKE_TEST"."BRAKE_REQ(ONLY_EXTERNAL)",
                               SIGN_OF_LOAD => "DB1034_Z13_BRAKE_TEST".SIGN_OF_LOAD);
   END_IF;
END_REGION

REGION Network 19: BRAKE TEST AXIS 4
   RUNG wire#powerrail
      Contact( "DB1030_TEST_STOP".TEST_STP_SQ_IN_PROCESS )
      wire#w1
      Contact( "DB1030_TEST_STOP".TEST_STP_TST_BRK_AX_3 )
      wire#w2
      Contact( "DB1034_Z13_BRAKE_TEST".BRAKE_TEST_DONE )
      wire#w3
      I_Contact( "DB1030_TEST_STOP".TEST_STP_TST_BRK_AX_5 )
      I_Contact( "DB1030_TEST_STOP".TST_STP_FIRST_SCAN_REQUEST )
      Coil( "DB1030_TEST_STOP".TEST_STP_TST_BRK_AX_4 )
   END_RUNG
   RUNG wire#w2
      I_Contact( #BRAKE_TEST_AXIS_Z13 )
   END_RUNG wire#w3
   RUNG wire#w1
      Contact( "DB1030_TEST_STOP".TEST_STP_TST_BRK_AX_4 )
   END_RUNG wire#w3
   // the same network as SCL:
   "DB1030_TEST_STOP".TEST_STP_TST_BRK_AX_4 := "DB1030_TEST_STOP".TEST_STP_SQ_IN_PROCESS AND (("DB1030_TEST_STOP".TEST_STP_TST_BRK_AX_3 AND ("DB1034_Z13_BRAKE_TEST".BRAKE_TEST_DONE OR NOT #BRAKE_TEST_AXIS_Z13)) OR "DB1030_TEST_STOP".TEST_STP_TST_BRK_AX_4) AND NOT "DB1030_TEST_STOP".TEST_STP_TST_BRK_AX_5 AND NOT "DB1030_TEST_STOP".TST_STP_FIRST_SCAN_REQUEST;
END_REGION

REGION Network 20: CALL FB1031 BRAKE TEST AXIS 4
   RUNG wire#powerrail
      I_Contact( "DB1030_TEST_STOP".TEST_STP_SQ_IN_PROCESS )
      I_Contact( "DB1036_X23_BRAKE_TEST".BRAKE_TEST_ERROR )
      Not()
      Contact( #BRAKE_TEST_AXIS_X23 )
      "DB1036_X23_BRAKE_TEST"(START_REQ := wire#w1, BRAKE_SELECT := "M_ZERO", DIRECTION_OF_ROT := "M_ONE", TORQUE_SELECT := "M_ZERO", "BRAKE_CLOSED(ONLY EXTERNAL)" :=, AXIS_DB := "LBP_Axis22", BRAKE_TEST_ACTIVE => "DB1036_X23_BRAKE_TEST".BRAKE_TEST_ACTIVE, BRAKE_TEST_DONE => "DB1036_X23_BRAKE_TEST".BRAKE_TEST_DONE, BRAKE_TEST_ERROR => "DB1036_X23_BRAKE_TEST".BRAKE_TEST_ERROR, SELECTED_BRAKE => "DB1036_X23_BRAKE_TEST".SELECTED_BRAKE, "BRAKE_REQ(ONLY_EXTERNAL)" => "DB1036_X23_BRAKE_TEST"."BRAKE_REQ(ONLY_EXTERNAL)", SIGN_OF_LOAD => "DB1036_X23_BRAKE_TEST".SIGN_OF_LOAD)
   END_RUNG
   RUNG wire#powerrail
      Contact( "DB1030_TEST_STOP".TEST_STP_TST_BRK_AX_4 )
      Contact( "DB152_CLADDING_AXIS_X23".MOTOR_ACTIVE )
      Contact( "DB152_CLADDING_AXIS_X23".FEED_HOLD_CONDITIONS )
   END_RUNG wire#w1
   // the same network as SCL:
   IF NOT (NOT "DB1030_TEST_STOP".TEST_STP_SQ_IN_PROCESS AND NOT "DB1036_X23_BRAKE_TEST".BRAKE_TEST_ERROR) AND #BRAKE_TEST_AXIS_X23 THEN
       "DB1036_X23_BRAKE_TEST"(START_REQ := "DB1030_TEST_STOP".TEST_STP_TST_BRK_AX_4 AND "DB152_CLADDING_AXIS_X23".MOTOR_ACTIVE AND "DB152_CLADDING_AXIS_X23".FEED_HOLD_CONDITIONS,   // "FB1031_BRAKE_TEST"
                               BRAKE_SELECT := "M_ZERO",
                               DIRECTION_OF_ROT := "M_ONE",
                               TORQUE_SELECT := "M_ZERO",
                               AXIS_DB := "LBP_Axis22",
                               BRAKE_TEST_ACTIVE => "DB1036_X23_BRAKE_TEST".BRAKE_TEST_ACTIVE,
                               BRAKE_TEST_DONE => "DB1036_X23_BRAKE_TEST".BRAKE_TEST_DONE,
                               BRAKE_TEST_ERROR => "DB1036_X23_BRAKE_TEST".BRAKE_TEST_ERROR,
                               SELECTED_BRAKE => "DB1036_X23_BRAKE_TEST".SELECTED_BRAKE,
                               "BRAKE_REQ(ONLY_EXTERNAL)" => "DB1036_X23_BRAKE_TEST"."BRAKE_REQ(ONLY_EXTERNAL)",
                               SIGN_OF_LOAD => "DB1036_X23_BRAKE_TEST".SIGN_OF_LOAD);
   END_IF;
END_REGION

REGION Network 21: BRAKE TEST AXIS 5
   RUNG wire#powerrail
      Contact( "DB1030_TEST_STOP".TEST_STP_SQ_IN_PROCESS )
      wire#w1
      Contact( "DB1030_TEST_STOP".TEST_STP_TST_BRK_AX_4 )
      wire#w2
      Contact( "DB1036_X23_BRAKE_TEST".BRAKE_TEST_DONE )
      wire#w3
      I_Contact( "DB1030_TEST_STOP".TEST_STP_TST_BRK_AX_6 )
      I_Contact( "DB1030_TEST_STOP".TST_STP_FIRST_SCAN_REQUEST )
      Coil( "DB1030_TEST_STOP".TEST_STP_TST_BRK_AX_5 )
   END_RUNG
   RUNG wire#w2
      I_Contact( #BRAKE_TEST_AXIS_X23 )
   END_RUNG wire#w3
   RUNG wire#w1
      Contact( "DB1030_TEST_STOP".TEST_STP_TST_BRK_AX_5 )
   END_RUNG wire#w3
   // the same network as SCL:
   "DB1030_TEST_STOP".TEST_STP_TST_BRK_AX_5 := "DB1030_TEST_STOP".TEST_STP_SQ_IN_PROCESS AND (("DB1030_TEST_STOP".TEST_STP_TST_BRK_AX_4 AND ("DB1036_X23_BRAKE_TEST".BRAKE_TEST_DONE OR NOT #BRAKE_TEST_AXIS_X23)) OR "DB1030_TEST_STOP".TEST_STP_TST_BRK_AX_5) AND NOT "DB1030_TEST_STOP".TEST_STP_TST_BRK_AX_6 AND NOT "DB1030_TEST_STOP".TST_STP_FIRST_SCAN_REQUEST;
END_REGION

REGION Network 22: CALL FB1031 BRAKE TEST AXIS 5
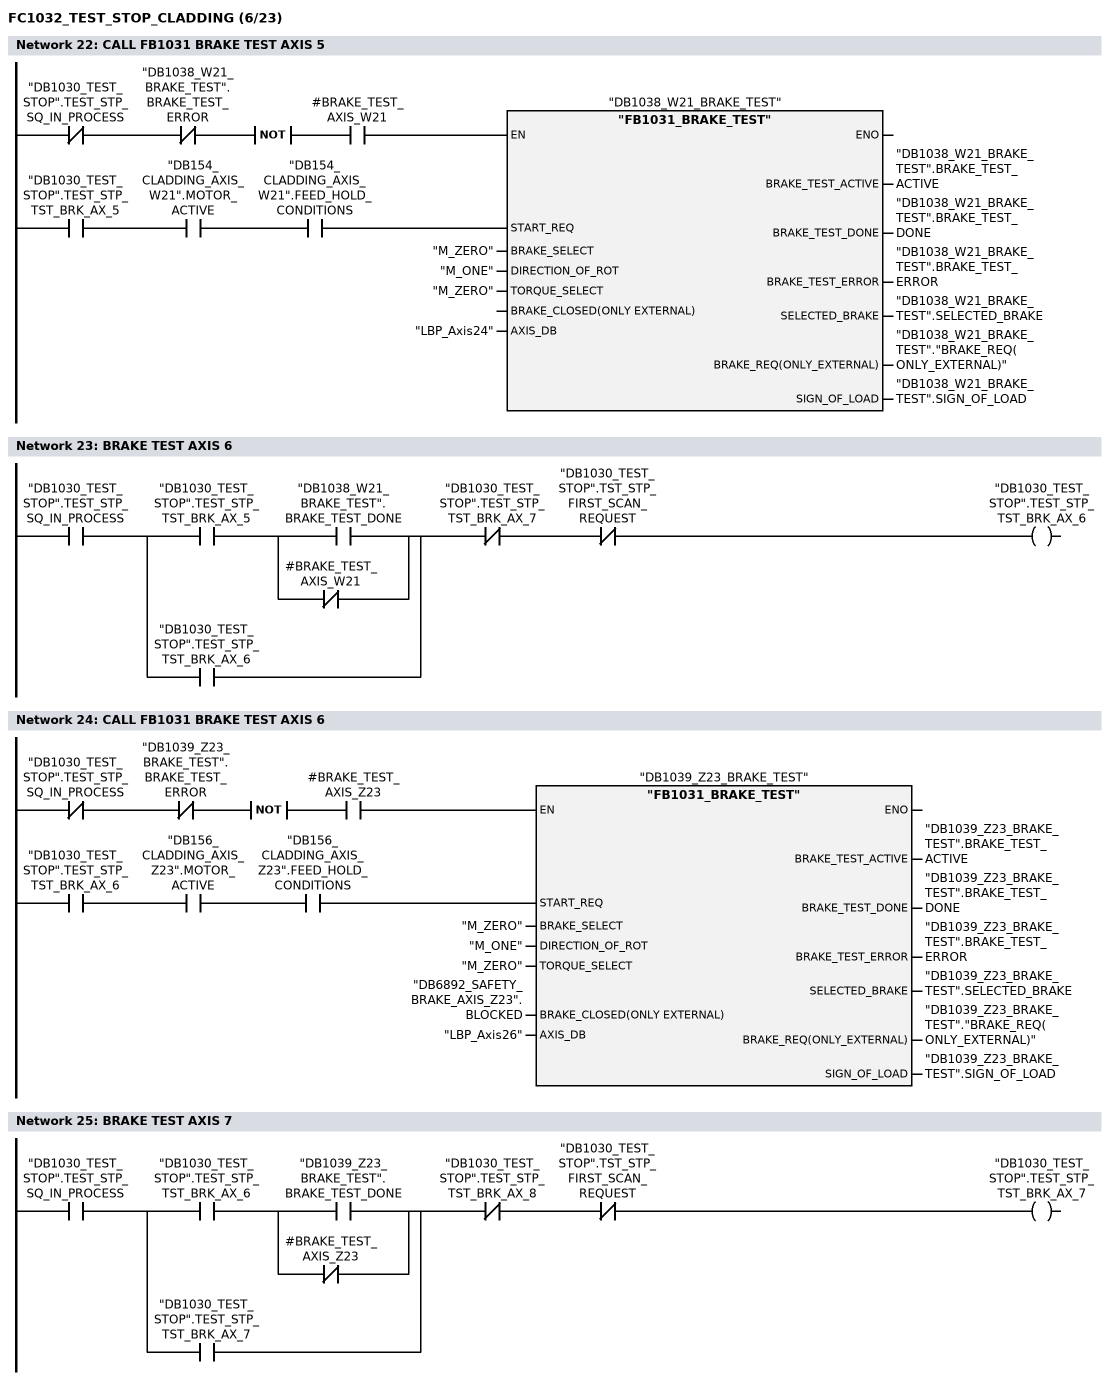
   RUNG wire#powerrail
      I_Contact( "DB1030_TEST_STOP".TEST_STP_SQ_IN_PROCESS )
      I_Contact( "DB1038_W21_BRAKE_TEST".BRAKE_TEST_ERROR )
      Not()
      Contact( #BRAKE_TEST_AXIS_W21 )
      "DB1038_W21_BRAKE_TEST"(START_REQ := wire#w1, BRAKE_SELECT := "M_ZERO", DIRECTION_OF_ROT := "M_ONE", TORQUE_SELECT := "M_ZERO", "BRAKE_CLOSED(ONLY EXTERNAL)" :=, AXIS_DB := "LBP_Axis24", BRAKE_TEST_ACTIVE => "DB1038_W21_BRAKE_TEST".BRAKE_TEST_ACTIVE, BRAKE_TEST_DONE => "DB1038_W21_BRAKE_TEST".BRAKE_TEST_DONE, BRAKE_TEST_ERROR => "DB1038_W21_BRAKE_TEST".BRAKE_TEST_ERROR, SELECTED_BRAKE => "DB1038_W21_BRAKE_TEST".SELECTED_BRAKE, "BRAKE_REQ(ONLY_EXTERNAL)" => "DB1038_W21_BRAKE_TEST"."BRAKE_REQ(ONLY_EXTERNAL)", SIGN_OF_LOAD => "DB1038_W21_BRAKE_TEST".SIGN_OF_LOAD)
   END_RUNG
   RUNG wire#powerrail
      Contact( "DB1030_TEST_STOP".TEST_STP_TST_BRK_AX_5 )
      Contact( "DB154_CLADDING_AXIS_W21".MOTOR_ACTIVE )
      Contact( "DB154_CLADDING_AXIS_W21".FEED_HOLD_CONDITIONS )
   END_RUNG wire#w1
   // the same network as SCL:
   IF NOT (NOT "DB1030_TEST_STOP".TEST_STP_SQ_IN_PROCESS AND NOT "DB1038_W21_BRAKE_TEST".BRAKE_TEST_ERROR) AND #BRAKE_TEST_AXIS_W21 THEN
       "DB1038_W21_BRAKE_TEST"(START_REQ := "DB1030_TEST_STOP".TEST_STP_TST_BRK_AX_5 AND "DB154_CLADDING_AXIS_W21".MOTOR_ACTIVE AND "DB154_CLADDING_AXIS_W21".FEED_HOLD_CONDITIONS,   // "FB1031_BRAKE_TEST"
                               BRAKE_SELECT := "M_ZERO",
                               DIRECTION_OF_ROT := "M_ONE",
                               TORQUE_SELECT := "M_ZERO",
                               AXIS_DB := "LBP_Axis24",
                               BRAKE_TEST_ACTIVE => "DB1038_W21_BRAKE_TEST".BRAKE_TEST_ACTIVE,
                               BRAKE_TEST_DONE => "DB1038_W21_BRAKE_TEST".BRAKE_TEST_DONE,
                               BRAKE_TEST_ERROR => "DB1038_W21_BRAKE_TEST".BRAKE_TEST_ERROR,
                               SELECTED_BRAKE => "DB1038_W21_BRAKE_TEST".SELECTED_BRAKE,
                               "BRAKE_REQ(ONLY_EXTERNAL)" => "DB1038_W21_BRAKE_TEST"."BRAKE_REQ(ONLY_EXTERNAL)",
                               SIGN_OF_LOAD => "DB1038_W21_BRAKE_TEST".SIGN_OF_LOAD);
   END_IF;
END_REGION

REGION Network 23: BRAKE TEST AXIS 6
   RUNG wire#powerrail
      Contact( "DB1030_TEST_STOP".TEST_STP_SQ_IN_PROCESS )
      wire#w1
      Contact( "DB1030_TEST_STOP".TEST_STP_TST_BRK_AX_5 )
      wire#w2
      Contact( "DB1038_W21_BRAKE_TEST".BRAKE_TEST_DONE )
      wire#w3
      I_Contact( "DB1030_TEST_STOP".TEST_STP_TST_BRK_AX_7 )
      I_Contact( "DB1030_TEST_STOP".TST_STP_FIRST_SCAN_REQUEST )
      Coil( "DB1030_TEST_STOP".TEST_STP_TST_BRK_AX_6 )
   END_RUNG
   RUNG wire#w2
      I_Contact( #BRAKE_TEST_AXIS_W21 )
   END_RUNG wire#w3
   RUNG wire#w1
      Contact( "DB1030_TEST_STOP".TEST_STP_TST_BRK_AX_6 )
   END_RUNG wire#w3
   // the same network as SCL:
   "DB1030_TEST_STOP".TEST_STP_TST_BRK_AX_6 := "DB1030_TEST_STOP".TEST_STP_SQ_IN_PROCESS AND (("DB1030_TEST_STOP".TEST_STP_TST_BRK_AX_5 AND ("DB1038_W21_BRAKE_TEST".BRAKE_TEST_DONE OR NOT #BRAKE_TEST_AXIS_W21)) OR "DB1030_TEST_STOP".TEST_STP_TST_BRK_AX_6) AND NOT "DB1030_TEST_STOP".TEST_STP_TST_BRK_AX_7 AND NOT "DB1030_TEST_STOP".TST_STP_FIRST_SCAN_REQUEST;
END_REGION

REGION Network 24: CALL FB1031 BRAKE TEST AXIS 6
   RUNG wire#powerrail
      I_Contact( "DB1030_TEST_STOP".TEST_STP_SQ_IN_PROCESS )
      I_Contact( "DB1039_Z23_BRAKE_TEST".BRAKE_TEST_ERROR )
      Not()
      Contact( #BRAKE_TEST_AXIS_Z23 )
      "DB1039_Z23_BRAKE_TEST"(START_REQ := wire#w1, BRAKE_SELECT := "M_ZERO", DIRECTION_OF_ROT := "M_ONE", TORQUE_SELECT := "M_ZERO", "BRAKE_CLOSED(ONLY EXTERNAL)" := "DB6892_SAFETY_BRAKE_AXIS_Z23".BLOCKED, AXIS_DB := "LBP_Axis26", BRAKE_TEST_ACTIVE => "DB1039_Z23_BRAKE_TEST".BRAKE_TEST_ACTIVE, BRAKE_TEST_DONE => "DB1039_Z23_BRAKE_TEST".BRAKE_TEST_DONE, BRAKE_TEST_ERROR => "DB1039_Z23_BRAKE_TEST".BRAKE_TEST_ERROR, SELECTED_BRAKE => "DB1039_Z23_BRAKE_TEST".SELECTED_BRAKE, "BRAKE_REQ(ONLY_EXTERNAL)" => "DB1039_Z23_BRAKE_TEST"."BRAKE_REQ(ONLY_EXTERNAL)", SIGN_OF_LOAD => "DB1039_Z23_BRAKE_TEST".SIGN_OF_LOAD)
   END_RUNG
   RUNG wire#powerrail
      Contact( "DB1030_TEST_STOP".TEST_STP_TST_BRK_AX_6 )
      Contact( "DB156_CLADDING_AXIS_Z23".MOTOR_ACTIVE )
      Contact( "DB156_CLADDING_AXIS_Z23".FEED_HOLD_CONDITIONS )
   END_RUNG wire#w1
   // the same network as SCL:
   IF NOT (NOT "DB1030_TEST_STOP".TEST_STP_SQ_IN_PROCESS AND NOT "DB1039_Z23_BRAKE_TEST".BRAKE_TEST_ERROR) AND #BRAKE_TEST_AXIS_Z23 THEN
       "DB1039_Z23_BRAKE_TEST"(START_REQ := "DB1030_TEST_STOP".TEST_STP_TST_BRK_AX_6 AND "DB156_CLADDING_AXIS_Z23".MOTOR_ACTIVE AND "DB156_CLADDING_AXIS_Z23".FEED_HOLD_CONDITIONS,   // "FB1031_BRAKE_TEST"
                               BRAKE_SELECT := "M_ZERO",
                               DIRECTION_OF_ROT := "M_ONE",
                               TORQUE_SELECT := "M_ZERO",
                               "BRAKE_CLOSED(ONLY EXTERNAL)" := "DB6892_SAFETY_BRAKE_AXIS_Z23".BLOCKED,
                               AXIS_DB := "LBP_Axis26",
                               BRAKE_TEST_ACTIVE => "DB1039_Z23_BRAKE_TEST".BRAKE_TEST_ACTIVE,
                               BRAKE_TEST_DONE => "DB1039_Z23_BRAKE_TEST".BRAKE_TEST_DONE,
                               BRAKE_TEST_ERROR => "DB1039_Z23_BRAKE_TEST".BRAKE_TEST_ERROR,
                               SELECTED_BRAKE => "DB1039_Z23_BRAKE_TEST".SELECTED_BRAKE,
                               "BRAKE_REQ(ONLY_EXTERNAL)" => "DB1039_Z23_BRAKE_TEST"."BRAKE_REQ(ONLY_EXTERNAL)",
                               SIGN_OF_LOAD => "DB1039_Z23_BRAKE_TEST".SIGN_OF_LOAD);
   END_IF;
END_REGION

REGION Network 25: BRAKE TEST AXIS 7
   RUNG wire#powerrail
      Contact( "DB1030_TEST_STOP".TEST_STP_SQ_IN_PROCESS )
      wire#w1
      Contact( "DB1030_TEST_STOP".TEST_STP_TST_BRK_AX_6 )
      wire#w2
      Contact( "DB1039_Z23_BRAKE_TEST".BRAKE_TEST_DONE )
      wire#w3
      I_Contact( "DB1030_TEST_STOP".TEST_STP_TST_BRK_AX_8 )
      I_Contact( "DB1030_TEST_STOP".TST_STP_FIRST_SCAN_REQUEST )
      Coil( "DB1030_TEST_STOP".TEST_STP_TST_BRK_AX_7 )
   END_RUNG
   RUNG wire#w2
      I_Contact( #BRAKE_TEST_AXIS_Z23 )
   END_RUNG wire#w3
   RUNG wire#w1
      Contact( "DB1030_TEST_STOP".TEST_STP_TST_BRK_AX_7 )
   END_RUNG wire#w3
   // the same network as SCL:
   "DB1030_TEST_STOP".TEST_STP_TST_BRK_AX_7 := "DB1030_TEST_STOP".TEST_STP_SQ_IN_PROCESS AND (("DB1030_TEST_STOP".TEST_STP_TST_BRK_AX_6 AND ("DB1039_Z23_BRAKE_TEST".BRAKE_TEST_DONE OR NOT #BRAKE_TEST_AXIS_Z23)) OR "DB1030_TEST_STOP".TEST_STP_TST_BRK_AX_7) AND NOT "DB1030_TEST_STOP".TEST_STP_TST_BRK_AX_8 AND NOT "DB1030_TEST_STOP".TST_STP_FIRST_SCAN_REQUEST;
END_REGION

REGION Network 26: CALL FB1031 BRAKE TEST AXIS 7
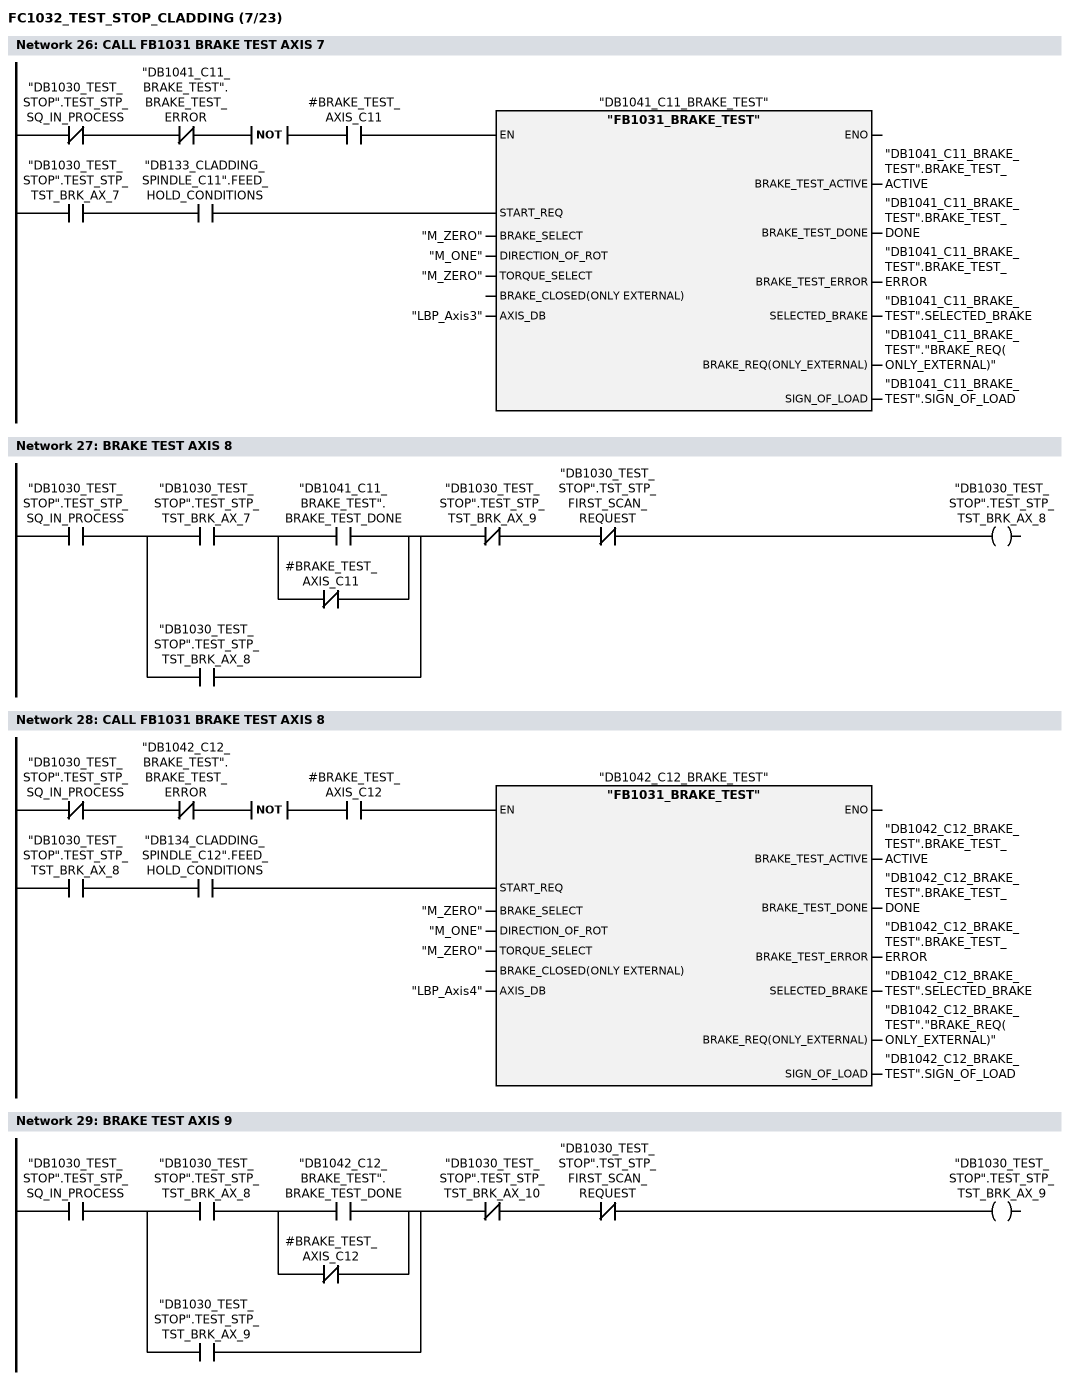
   RUNG wire#powerrail
      I_Contact( "DB1030_TEST_STOP".TEST_STP_SQ_IN_PROCESS )
      I_Contact( "DB1041_C11_BRAKE_TEST".BRAKE_TEST_ERROR )
      Not()
      Contact( #BRAKE_TEST_AXIS_C11 )
      "DB1041_C11_BRAKE_TEST"(START_REQ := wire#w1, BRAKE_SELECT := "M_ZERO", DIRECTION_OF_ROT := "M_ONE", TORQUE_SELECT := "M_ZERO", "BRAKE_CLOSED(ONLY EXTERNAL)" :=, AXIS_DB := "LBP_Axis3", BRAKE_TEST_ACTIVE => "DB1041_C11_BRAKE_TEST".BRAKE_TEST_ACTIVE, BRAKE_TEST_DONE => "DB1041_C11_BRAKE_TEST".BRAKE_TEST_DONE, BRAKE_TEST_ERROR => "DB1041_C11_BRAKE_TEST".BRAKE_TEST_ERROR, SELECTED_BRAKE => "DB1041_C11_BRAKE_TEST".SELECTED_BRAKE, "BRAKE_REQ(ONLY_EXTERNAL)" => "DB1041_C11_BRAKE_TEST"."BRAKE_REQ(ONLY_EXTERNAL)", SIGN_OF_LOAD => "DB1041_C11_BRAKE_TEST".SIGN_OF_LOAD)
   END_RUNG
   RUNG wire#powerrail
      Contact( "DB1030_TEST_STOP".TEST_STP_TST_BRK_AX_7 )
      Contact( "DB133_CLADDING_SPINDLE_C11".FEED_HOLD_CONDITIONS )
   END_RUNG wire#w1
   // the same network as SCL:
   IF NOT (NOT "DB1030_TEST_STOP".TEST_STP_SQ_IN_PROCESS AND NOT "DB1041_C11_BRAKE_TEST".BRAKE_TEST_ERROR) AND #BRAKE_TEST_AXIS_C11 THEN
       "DB1041_C11_BRAKE_TEST"(START_REQ := "DB1030_TEST_STOP".TEST_STP_TST_BRK_AX_7 AND "DB133_CLADDING_SPINDLE_C11".FEED_HOLD_CONDITIONS,   // "FB1031_BRAKE_TEST"
                               BRAKE_SELECT := "M_ZERO",
                               DIRECTION_OF_ROT := "M_ONE",
                               TORQUE_SELECT := "M_ZERO",
                               AXIS_DB := "LBP_Axis3",
                               BRAKE_TEST_ACTIVE => "DB1041_C11_BRAKE_TEST".BRAKE_TEST_ACTIVE,
                               BRAKE_TEST_DONE => "DB1041_C11_BRAKE_TEST".BRAKE_TEST_DONE,
                               BRAKE_TEST_ERROR => "DB1041_C11_BRAKE_TEST".BRAKE_TEST_ERROR,
                               SELECTED_BRAKE => "DB1041_C11_BRAKE_TEST".SELECTED_BRAKE,
                               "BRAKE_REQ(ONLY_EXTERNAL)" => "DB1041_C11_BRAKE_TEST"."BRAKE_REQ(ONLY_EXTERNAL)",
                               SIGN_OF_LOAD => "DB1041_C11_BRAKE_TEST".SIGN_OF_LOAD);
   END_IF;
END_REGION

REGION Network 27: BRAKE TEST AXIS 8
   RUNG wire#powerrail
      Contact( "DB1030_TEST_STOP".TEST_STP_SQ_IN_PROCESS )
      wire#w1
      Contact( "DB1030_TEST_STOP".TEST_STP_TST_BRK_AX_7 )
      wire#w2
      Contact( "DB1041_C11_BRAKE_TEST".BRAKE_TEST_DONE )
      wire#w3
      I_Contact( "DB1030_TEST_STOP".TEST_STP_TST_BRK_AX_9 )
      I_Contact( "DB1030_TEST_STOP".TST_STP_FIRST_SCAN_REQUEST )
      Coil( "DB1030_TEST_STOP".TEST_STP_TST_BRK_AX_8 )
   END_RUNG
   RUNG wire#w2
      I_Contact( #BRAKE_TEST_AXIS_C11 )
   END_RUNG wire#w3
   RUNG wire#w1
      Contact( "DB1030_TEST_STOP".TEST_STP_TST_BRK_AX_8 )
   END_RUNG wire#w3
   // the same network as SCL:
   "DB1030_TEST_STOP".TEST_STP_TST_BRK_AX_8 := "DB1030_TEST_STOP".TEST_STP_SQ_IN_PROCESS AND (("DB1030_TEST_STOP".TEST_STP_TST_BRK_AX_7 AND ("DB1041_C11_BRAKE_TEST".BRAKE_TEST_DONE OR NOT #BRAKE_TEST_AXIS_C11)) OR "DB1030_TEST_STOP".TEST_STP_TST_BRK_AX_8) AND NOT "DB1030_TEST_STOP".TEST_STP_TST_BRK_AX_9 AND NOT "DB1030_TEST_STOP".TST_STP_FIRST_SCAN_REQUEST;
END_REGION

REGION Network 28: CALL FB1031 BRAKE TEST AXIS 8
   RUNG wire#powerrail
      I_Contact( "DB1030_TEST_STOP".TEST_STP_SQ_IN_PROCESS )
      I_Contact( "DB1042_C12_BRAKE_TEST".BRAKE_TEST_ERROR )
      Not()
      Contact( #BRAKE_TEST_AXIS_C12 )
      "DB1042_C12_BRAKE_TEST"(START_REQ := wire#w1, BRAKE_SELECT := "M_ZERO", DIRECTION_OF_ROT := "M_ONE", TORQUE_SELECT := "M_ZERO", "BRAKE_CLOSED(ONLY EXTERNAL)" :=, AXIS_DB := "LBP_Axis4", BRAKE_TEST_ACTIVE => "DB1042_C12_BRAKE_TEST".BRAKE_TEST_ACTIVE, BRAKE_TEST_DONE => "DB1042_C12_BRAKE_TEST".BRAKE_TEST_DONE, BRAKE_TEST_ERROR => "DB1042_C12_BRAKE_TEST".BRAKE_TEST_ERROR, SELECTED_BRAKE => "DB1042_C12_BRAKE_TEST".SELECTED_BRAKE, "BRAKE_REQ(ONLY_EXTERNAL)" => "DB1042_C12_BRAKE_TEST"."BRAKE_REQ(ONLY_EXTERNAL)", SIGN_OF_LOAD => "DB1042_C12_BRAKE_TEST".SIGN_OF_LOAD)
   END_RUNG
   RUNG wire#powerrail
      Contact( "DB1030_TEST_STOP".TEST_STP_TST_BRK_AX_8 )
      Contact( "DB134_CLADDING_SPINDLE_C12".FEED_HOLD_CONDITIONS )
   END_RUNG wire#w1
   // the same network as SCL:
   IF NOT (NOT "DB1030_TEST_STOP".TEST_STP_SQ_IN_PROCESS AND NOT "DB1042_C12_BRAKE_TEST".BRAKE_TEST_ERROR) AND #BRAKE_TEST_AXIS_C12 THEN
       "DB1042_C12_BRAKE_TEST"(START_REQ := "DB1030_TEST_STOP".TEST_STP_TST_BRK_AX_8 AND "DB134_CLADDING_SPINDLE_C12".FEED_HOLD_CONDITIONS,   // "FB1031_BRAKE_TEST"
                               BRAKE_SELECT := "M_ZERO",
                               DIRECTION_OF_ROT := "M_ONE",
                               TORQUE_SELECT := "M_ZERO",
                               AXIS_DB := "LBP_Axis4",
                               BRAKE_TEST_ACTIVE => "DB1042_C12_BRAKE_TEST".BRAKE_TEST_ACTIVE,
                               BRAKE_TEST_DONE => "DB1042_C12_BRAKE_TEST".BRAKE_TEST_DONE,
                               BRAKE_TEST_ERROR => "DB1042_C12_BRAKE_TEST".BRAKE_TEST_ERROR,
                               SELECTED_BRAKE => "DB1042_C12_BRAKE_TEST".SELECTED_BRAKE,
                               "BRAKE_REQ(ONLY_EXTERNAL)" => "DB1042_C12_BRAKE_TEST"."BRAKE_REQ(ONLY_EXTERNAL)",
                               SIGN_OF_LOAD => "DB1042_C12_BRAKE_TEST".SIGN_OF_LOAD);
   END_IF;
END_REGION

REGION Network 29: BRAKE TEST AXIS 9
   RUNG wire#powerrail
      Contact( "DB1030_TEST_STOP".TEST_STP_SQ_IN_PROCESS )
      wire#w1
      Contact( "DB1030_TEST_STOP".TEST_STP_TST_BRK_AX_8 )
      wire#w2
      Contact( "DB1042_C12_BRAKE_TEST".BRAKE_TEST_DONE )
      wire#w3
      I_Contact( "DB1030_TEST_STOP".TEST_STP_TST_BRK_AX_10 )
      I_Contact( "DB1030_TEST_STOP".TST_STP_FIRST_SCAN_REQUEST )
      Coil( "DB1030_TEST_STOP".TEST_STP_TST_BRK_AX_9 )
   END_RUNG
   RUNG wire#w2
      I_Contact( #BRAKE_TEST_AXIS_C12 )
   END_RUNG wire#w3
   RUNG wire#w1
      Contact( "DB1030_TEST_STOP".TEST_STP_TST_BRK_AX_9 )
   END_RUNG wire#w3
   // the same network as SCL:
   "DB1030_TEST_STOP".TEST_STP_TST_BRK_AX_9 := "DB1030_TEST_STOP".TEST_STP_SQ_IN_PROCESS AND (("DB1030_TEST_STOP".TEST_STP_TST_BRK_AX_8 AND ("DB1042_C12_BRAKE_TEST".BRAKE_TEST_DONE OR NOT #BRAKE_TEST_AXIS_C12)) OR "DB1030_TEST_STOP".TEST_STP_TST_BRK_AX_9) AND NOT "DB1030_TEST_STOP".TEST_STP_TST_BRK_AX_10 AND NOT "DB1030_TEST_STOP".TST_STP_FIRST_SCAN_REQUEST;
END_REGION

REGION Network 30: CALL FB1031 BRAKE TEST AXIS 9
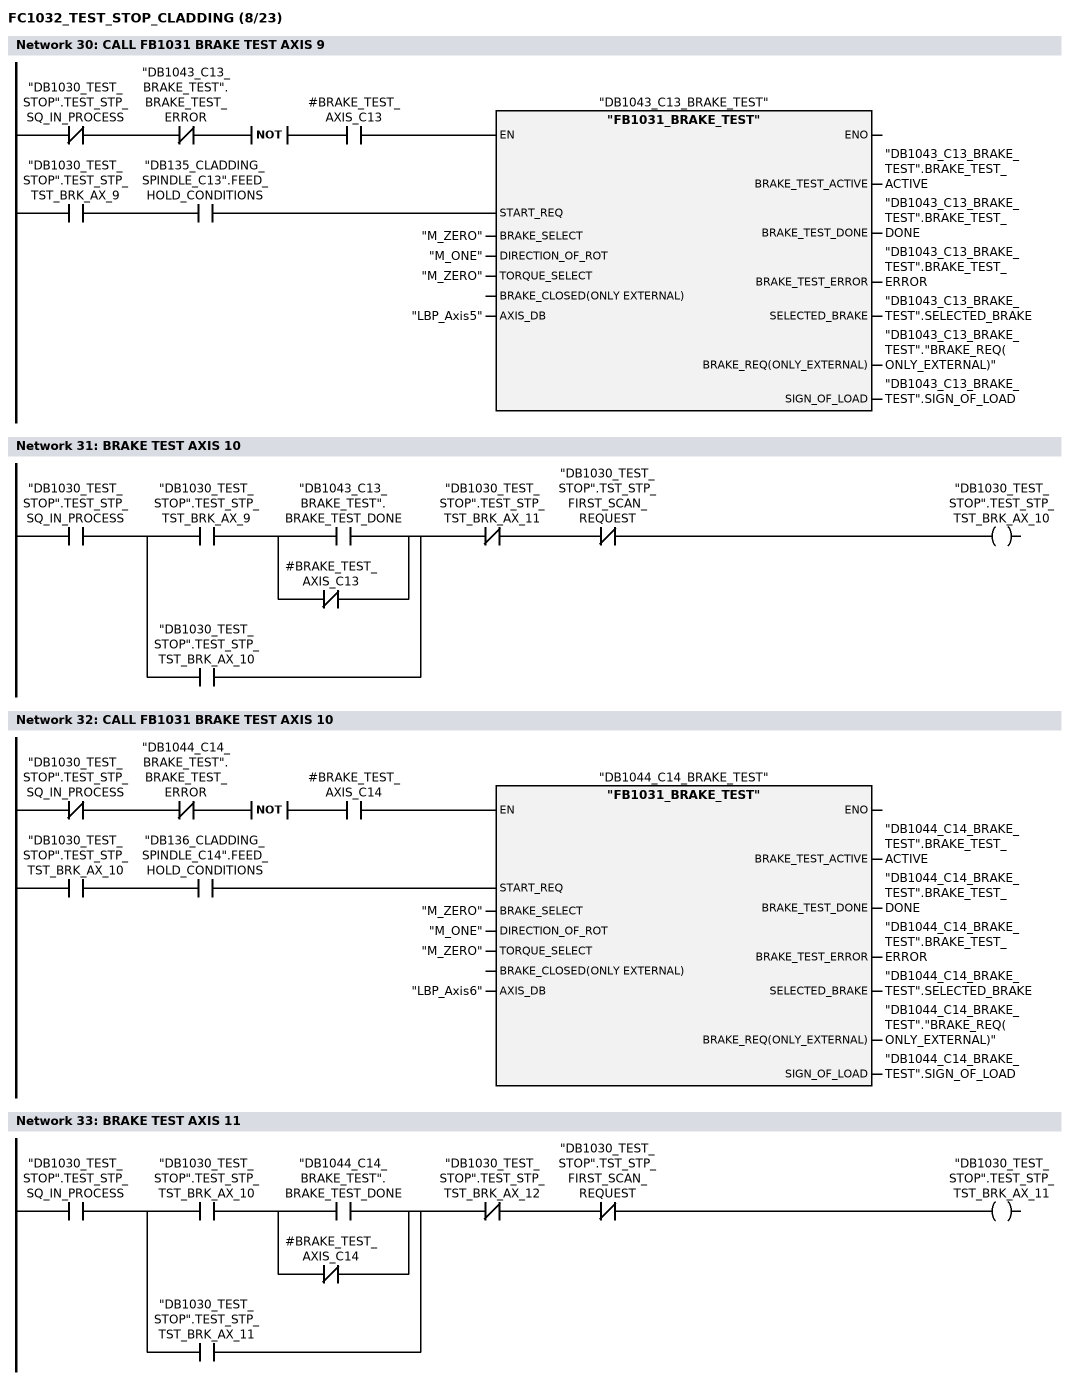
   RUNG wire#powerrail
      I_Contact( "DB1030_TEST_STOP".TEST_STP_SQ_IN_PROCESS )
      I_Contact( "DB1043_C13_BRAKE_TEST".BRAKE_TEST_ERROR )
      Not()
      Contact( #BRAKE_TEST_AXIS_C13 )
      "DB1043_C13_BRAKE_TEST"(START_REQ := wire#w1, BRAKE_SELECT := "M_ZERO", DIRECTION_OF_ROT := "M_ONE", TORQUE_SELECT := "M_ZERO", "BRAKE_CLOSED(ONLY EXTERNAL)" :=, AXIS_DB := "LBP_Axis5", BRAKE_TEST_ACTIVE => "DB1043_C13_BRAKE_TEST".BRAKE_TEST_ACTIVE, BRAKE_TEST_DONE => "DB1043_C13_BRAKE_TEST".BRAKE_TEST_DONE, BRAKE_TEST_ERROR => "DB1043_C13_BRAKE_TEST".BRAKE_TEST_ERROR, SELECTED_BRAKE => "DB1043_C13_BRAKE_TEST".SELECTED_BRAKE, "BRAKE_REQ(ONLY_EXTERNAL)" => "DB1043_C13_BRAKE_TEST"."BRAKE_REQ(ONLY_EXTERNAL)", SIGN_OF_LOAD => "DB1043_C13_BRAKE_TEST".SIGN_OF_LOAD)
   END_RUNG
   RUNG wire#powerrail
      Contact( "DB1030_TEST_STOP".TEST_STP_TST_BRK_AX_9 )
      Contact( "DB135_CLADDING_SPINDLE_C13".FEED_HOLD_CONDITIONS )
   END_RUNG wire#w1
   // the same network as SCL:
   IF NOT (NOT "DB1030_TEST_STOP".TEST_STP_SQ_IN_PROCESS AND NOT "DB1043_C13_BRAKE_TEST".BRAKE_TEST_ERROR) AND #BRAKE_TEST_AXIS_C13 THEN
       "DB1043_C13_BRAKE_TEST"(START_REQ := "DB1030_TEST_STOP".TEST_STP_TST_BRK_AX_9 AND "DB135_CLADDING_SPINDLE_C13".FEED_HOLD_CONDITIONS,   // "FB1031_BRAKE_TEST"
                               BRAKE_SELECT := "M_ZERO",
                               DIRECTION_OF_ROT := "M_ONE",
                               TORQUE_SELECT := "M_ZERO",
                               AXIS_DB := "LBP_Axis5",
                               BRAKE_TEST_ACTIVE => "DB1043_C13_BRAKE_TEST".BRAKE_TEST_ACTIVE,
                               BRAKE_TEST_DONE => "DB1043_C13_BRAKE_TEST".BRAKE_TEST_DONE,
                               BRAKE_TEST_ERROR => "DB1043_C13_BRAKE_TEST".BRAKE_TEST_ERROR,
                               SELECTED_BRAKE => "DB1043_C13_BRAKE_TEST".SELECTED_BRAKE,
                               "BRAKE_REQ(ONLY_EXTERNAL)" => "DB1043_C13_BRAKE_TEST"."BRAKE_REQ(ONLY_EXTERNAL)",
                               SIGN_OF_LOAD => "DB1043_C13_BRAKE_TEST".SIGN_OF_LOAD);
   END_IF;
END_REGION

REGION Network 31: BRAKE TEST AXIS 10
   RUNG wire#powerrail
      Contact( "DB1030_TEST_STOP".TEST_STP_SQ_IN_PROCESS )
      wire#w1
      Contact( "DB1030_TEST_STOP".TEST_STP_TST_BRK_AX_9 )
      wire#w2
      Contact( "DB1043_C13_BRAKE_TEST".BRAKE_TEST_DONE )
      wire#w3
      I_Contact( "DB1030_TEST_STOP".TEST_STP_TST_BRK_AX_11 )
      I_Contact( "DB1030_TEST_STOP".TST_STP_FIRST_SCAN_REQUEST )
      Coil( "DB1030_TEST_STOP".TEST_STP_TST_BRK_AX_10 )
   END_RUNG
   RUNG wire#w2
      I_Contact( #BRAKE_TEST_AXIS_C13 )
   END_RUNG wire#w3
   RUNG wire#w1
      Contact( "DB1030_TEST_STOP".TEST_STP_TST_BRK_AX_10 )
   END_RUNG wire#w3
   // the same network as SCL:
   "DB1030_TEST_STOP".TEST_STP_TST_BRK_AX_10 := "DB1030_TEST_STOP".TEST_STP_SQ_IN_PROCESS AND (("DB1030_TEST_STOP".TEST_STP_TST_BRK_AX_9 AND ("DB1043_C13_BRAKE_TEST".BRAKE_TEST_DONE OR NOT #BRAKE_TEST_AXIS_C13)) OR "DB1030_TEST_STOP".TEST_STP_TST_BRK_AX_10) AND NOT "DB1030_TEST_STOP".TEST_STP_TST_BRK_AX_11 AND NOT "DB1030_TEST_STOP".TST_STP_FIRST_SCAN_REQUEST;
END_REGION

REGION Network 32: CALL FB1031 BRAKE TEST AXIS 10
   RUNG wire#powerrail
      I_Contact( "DB1030_TEST_STOP".TEST_STP_SQ_IN_PROCESS )
      I_Contact( "DB1044_C14_BRAKE_TEST".BRAKE_TEST_ERROR )
      Not()
      Contact( #BRAKE_TEST_AXIS_C14 )
      "DB1044_C14_BRAKE_TEST"(START_REQ := wire#w1, BRAKE_SELECT := "M_ZERO", DIRECTION_OF_ROT := "M_ONE", TORQUE_SELECT := "M_ZERO", "BRAKE_CLOSED(ONLY EXTERNAL)" :=, AXIS_DB := "LBP_Axis6", BRAKE_TEST_ACTIVE => "DB1044_C14_BRAKE_TEST".BRAKE_TEST_ACTIVE, BRAKE_TEST_DONE => "DB1044_C14_BRAKE_TEST".BRAKE_TEST_DONE, BRAKE_TEST_ERROR => "DB1044_C14_BRAKE_TEST".BRAKE_TEST_ERROR, SELECTED_BRAKE => "DB1044_C14_BRAKE_TEST".SELECTED_BRAKE, "BRAKE_REQ(ONLY_EXTERNAL)" => "DB1044_C14_BRAKE_TEST"."BRAKE_REQ(ONLY_EXTERNAL)", SIGN_OF_LOAD => "DB1044_C14_BRAKE_TEST".SIGN_OF_LOAD)
   END_RUNG
   RUNG wire#powerrail
      Contact( "DB1030_TEST_STOP".TEST_STP_TST_BRK_AX_10 )
      Contact( "DB136_CLADDING_SPINDLE_C14".FEED_HOLD_CONDITIONS )
   END_RUNG wire#w1
   // the same network as SCL:
   IF NOT (NOT "DB1030_TEST_STOP".TEST_STP_SQ_IN_PROCESS AND NOT "DB1044_C14_BRAKE_TEST".BRAKE_TEST_ERROR) AND #BRAKE_TEST_AXIS_C14 THEN
       "DB1044_C14_BRAKE_TEST"(START_REQ := "DB1030_TEST_STOP".TEST_STP_TST_BRK_AX_10 AND "DB136_CLADDING_SPINDLE_C14".FEED_HOLD_CONDITIONS,   // "FB1031_BRAKE_TEST"
                               BRAKE_SELECT := "M_ZERO",
                               DIRECTION_OF_ROT := "M_ONE",
                               TORQUE_SELECT := "M_ZERO",
                               AXIS_DB := "LBP_Axis6",
                               BRAKE_TEST_ACTIVE => "DB1044_C14_BRAKE_TEST".BRAKE_TEST_ACTIVE,
                               BRAKE_TEST_DONE => "DB1044_C14_BRAKE_TEST".BRAKE_TEST_DONE,
                               BRAKE_TEST_ERROR => "DB1044_C14_BRAKE_TEST".BRAKE_TEST_ERROR,
                               SELECTED_BRAKE => "DB1044_C14_BRAKE_TEST".SELECTED_BRAKE,
                               "BRAKE_REQ(ONLY_EXTERNAL)" => "DB1044_C14_BRAKE_TEST"."BRAKE_REQ(ONLY_EXTERNAL)",
                               SIGN_OF_LOAD => "DB1044_C14_BRAKE_TEST".SIGN_OF_LOAD);
   END_IF;
END_REGION

REGION Network 33: BRAKE TEST AXIS 11
   RUNG wire#powerrail
      Contact( "DB1030_TEST_STOP".TEST_STP_SQ_IN_PROCESS )
      wire#w1
      Contact( "DB1030_TEST_STOP".TEST_STP_TST_BRK_AX_10 )
      wire#w2
      Contact( "DB1044_C14_BRAKE_TEST".BRAKE_TEST_DONE )
      wire#w3
      I_Contact( "DB1030_TEST_STOP".TEST_STP_TST_BRK_AX_12 )
      I_Contact( "DB1030_TEST_STOP".TST_STP_FIRST_SCAN_REQUEST )
      Coil( "DB1030_TEST_STOP".TEST_STP_TST_BRK_AX_11 )
   END_RUNG
   RUNG wire#w2
      I_Contact( #BRAKE_TEST_AXIS_C14 )
   END_RUNG wire#w3
   RUNG wire#w1
      Contact( "DB1030_TEST_STOP".TEST_STP_TST_BRK_AX_11 )
   END_RUNG wire#w3
   // the same network as SCL:
   "DB1030_TEST_STOP".TEST_STP_TST_BRK_AX_11 := "DB1030_TEST_STOP".TEST_STP_SQ_IN_PROCESS AND (("DB1030_TEST_STOP".TEST_STP_TST_BRK_AX_10 AND ("DB1044_C14_BRAKE_TEST".BRAKE_TEST_DONE OR NOT #BRAKE_TEST_AXIS_C14)) OR "DB1030_TEST_STOP".TEST_STP_TST_BRK_AX_11) AND NOT "DB1030_TEST_STOP".TEST_STP_TST_BRK_AX_12 AND NOT "DB1030_TEST_STOP".TST_STP_FIRST_SCAN_REQUEST;
END_REGION

REGION Network 34: CALL FB1031 BRAKE TEST AXIS 11
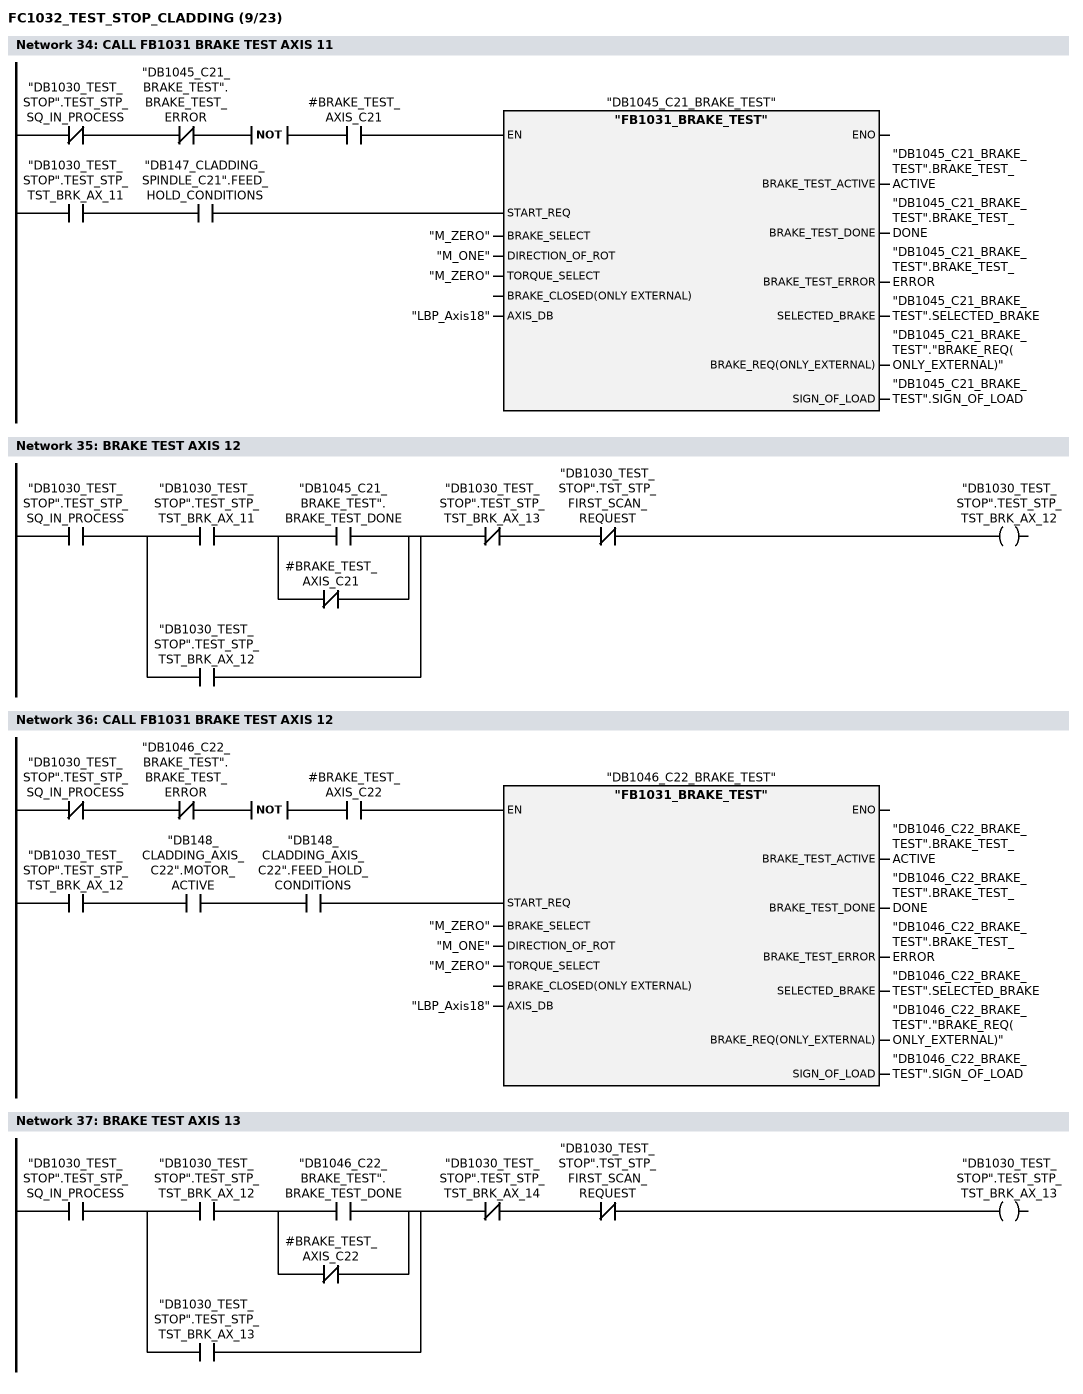
   RUNG wire#powerrail
      I_Contact( "DB1030_TEST_STOP".TEST_STP_SQ_IN_PROCESS )
      I_Contact( "DB1045_C21_BRAKE_TEST".BRAKE_TEST_ERROR )
      Not()
      Contact( #BRAKE_TEST_AXIS_C21 )
      "DB1045_C21_BRAKE_TEST"(START_REQ := wire#w1, BRAKE_SELECT := "M_ZERO", DIRECTION_OF_ROT := "M_ONE", TORQUE_SELECT := "M_ZERO", "BRAKE_CLOSED(ONLY EXTERNAL)" :=, AXIS_DB := "LBP_Axis18", BRAKE_TEST_ACTIVE => "DB1045_C21_BRAKE_TEST".BRAKE_TEST_ACTIVE, BRAKE_TEST_DONE => "DB1045_C21_BRAKE_TEST".BRAKE_TEST_DONE, BRAKE_TEST_ERROR => "DB1045_C21_BRAKE_TEST".BRAKE_TEST_ERROR, SELECTED_BRAKE => "DB1045_C21_BRAKE_TEST".SELECTED_BRAKE, "BRAKE_REQ(ONLY_EXTERNAL)" => "DB1045_C21_BRAKE_TEST"."BRAKE_REQ(ONLY_EXTERNAL)", SIGN_OF_LOAD => "DB1045_C21_BRAKE_TEST".SIGN_OF_LOAD)
   END_RUNG
   RUNG wire#powerrail
      Contact( "DB1030_TEST_STOP".TEST_STP_TST_BRK_AX_11 )
      Contact( "DB147_CLADDING_SPINDLE_C21".FEED_HOLD_CONDITIONS )
   END_RUNG wire#w1
   // the same network as SCL:
   IF NOT (NOT "DB1030_TEST_STOP".TEST_STP_SQ_IN_PROCESS AND NOT "DB1045_C21_BRAKE_TEST".BRAKE_TEST_ERROR) AND #BRAKE_TEST_AXIS_C21 THEN
       "DB1045_C21_BRAKE_TEST"(START_REQ := "DB1030_TEST_STOP".TEST_STP_TST_BRK_AX_11 AND "DB147_CLADDING_SPINDLE_C21".FEED_HOLD_CONDITIONS,   // "FB1031_BRAKE_TEST"
                               BRAKE_SELECT := "M_ZERO",
                               DIRECTION_OF_ROT := "M_ONE",
                               TORQUE_SELECT := "M_ZERO",
                               AXIS_DB := "LBP_Axis18",
                               BRAKE_TEST_ACTIVE => "DB1045_C21_BRAKE_TEST".BRAKE_TEST_ACTIVE,
                               BRAKE_TEST_DONE => "DB1045_C21_BRAKE_TEST".BRAKE_TEST_DONE,
                               BRAKE_TEST_ERROR => "DB1045_C21_BRAKE_TEST".BRAKE_TEST_ERROR,
                               SELECTED_BRAKE => "DB1045_C21_BRAKE_TEST".SELECTED_BRAKE,
                               "BRAKE_REQ(ONLY_EXTERNAL)" => "DB1045_C21_BRAKE_TEST"."BRAKE_REQ(ONLY_EXTERNAL)",
                               SIGN_OF_LOAD => "DB1045_C21_BRAKE_TEST".SIGN_OF_LOAD);
   END_IF;
END_REGION

REGION Network 35: BRAKE TEST AXIS 12
   RUNG wire#powerrail
      Contact( "DB1030_TEST_STOP".TEST_STP_SQ_IN_PROCESS )
      wire#w1
      Contact( "DB1030_TEST_STOP".TEST_STP_TST_BRK_AX_11 )
      wire#w2
      Contact( "DB1045_C21_BRAKE_TEST".BRAKE_TEST_DONE )
      wire#w3
      I_Contact( "DB1030_TEST_STOP".TEST_STP_TST_BRK_AX_13 )
      I_Contact( "DB1030_TEST_STOP".TST_STP_FIRST_SCAN_REQUEST )
      Coil( "DB1030_TEST_STOP".TEST_STP_TST_BRK_AX_12 )
   END_RUNG
   RUNG wire#w2
      I_Contact( #BRAKE_TEST_AXIS_C21 )
   END_RUNG wire#w3
   RUNG wire#w1
      Contact( "DB1030_TEST_STOP".TEST_STP_TST_BRK_AX_12 )
   END_RUNG wire#w3
   // the same network as SCL:
   "DB1030_TEST_STOP".TEST_STP_TST_BRK_AX_12 := "DB1030_TEST_STOP".TEST_STP_SQ_IN_PROCESS AND (("DB1030_TEST_STOP".TEST_STP_TST_BRK_AX_11 AND ("DB1045_C21_BRAKE_TEST".BRAKE_TEST_DONE OR NOT #BRAKE_TEST_AXIS_C21)) OR "DB1030_TEST_STOP".TEST_STP_TST_BRK_AX_12) AND NOT "DB1030_TEST_STOP".TEST_STP_TST_BRK_AX_13 AND NOT "DB1030_TEST_STOP".TST_STP_FIRST_SCAN_REQUEST;
END_REGION

REGION Network 36: CALL FB1031 BRAKE TEST AXIS 12
   RUNG wire#powerrail
      I_Contact( "DB1030_TEST_STOP".TEST_STP_SQ_IN_PROCESS )
      I_Contact( "DB1046_C22_BRAKE_TEST".BRAKE_TEST_ERROR )
      Not()
      Contact( #BRAKE_TEST_AXIS_C22 )
      "DB1046_C22_BRAKE_TEST"(START_REQ := wire#w1, BRAKE_SELECT := "M_ZERO", DIRECTION_OF_ROT := "M_ONE", TORQUE_SELECT := "M_ZERO", "BRAKE_CLOSED(ONLY EXTERNAL)" :=, AXIS_DB := "LBP_Axis18", BRAKE_TEST_ACTIVE => "DB1046_C22_BRAKE_TEST".BRAKE_TEST_ACTIVE, BRAKE_TEST_DONE => "DB1046_C22_BRAKE_TEST".BRAKE_TEST_DONE, BRAKE_TEST_ERROR => "DB1046_C22_BRAKE_TEST".BRAKE_TEST_ERROR, SELECTED_BRAKE => "DB1046_C22_BRAKE_TEST".SELECTED_BRAKE, "BRAKE_REQ(ONLY_EXTERNAL)" => "DB1046_C22_BRAKE_TEST"."BRAKE_REQ(ONLY_EXTERNAL)", SIGN_OF_LOAD => "DB1046_C22_BRAKE_TEST".SIGN_OF_LOAD)
   END_RUNG
   RUNG wire#powerrail
      Contact( "DB1030_TEST_STOP".TEST_STP_TST_BRK_AX_12 )
      Contact( "DB148_CLADDING_AXIS_C22".MOTOR_ACTIVE )
      Contact( "DB148_CLADDING_AXIS_C22".FEED_HOLD_CONDITIONS )
   END_RUNG wire#w1
   // the same network as SCL:
   IF NOT (NOT "DB1030_TEST_STOP".TEST_STP_SQ_IN_PROCESS AND NOT "DB1046_C22_BRAKE_TEST".BRAKE_TEST_ERROR) AND #BRAKE_TEST_AXIS_C22 THEN
       "DB1046_C22_BRAKE_TEST"(START_REQ := "DB1030_TEST_STOP".TEST_STP_TST_BRK_AX_12 AND "DB148_CLADDING_AXIS_C22".MOTOR_ACTIVE AND "DB148_CLADDING_AXIS_C22".FEED_HOLD_CONDITIONS,   // "FB1031_BRAKE_TEST"
                               BRAKE_SELECT := "M_ZERO",
                               DIRECTION_OF_ROT := "M_ONE",
                               TORQUE_SELECT := "M_ZERO",
                               AXIS_DB := "LBP_Axis18",
                               BRAKE_TEST_ACTIVE => "DB1046_C22_BRAKE_TEST".BRAKE_TEST_ACTIVE,
                               BRAKE_TEST_DONE => "DB1046_C22_BRAKE_TEST".BRAKE_TEST_DONE,
                               BRAKE_TEST_ERROR => "DB1046_C22_BRAKE_TEST".BRAKE_TEST_ERROR,
                               SELECTED_BRAKE => "DB1046_C22_BRAKE_TEST".SELECTED_BRAKE,
                               "BRAKE_REQ(ONLY_EXTERNAL)" => "DB1046_C22_BRAKE_TEST"."BRAKE_REQ(ONLY_EXTERNAL)",
                               SIGN_OF_LOAD => "DB1046_C22_BRAKE_TEST".SIGN_OF_LOAD);
   END_IF;
END_REGION

REGION Network 37: BRAKE TEST AXIS 13
   RUNG wire#powerrail
      Contact( "DB1030_TEST_STOP".TEST_STP_SQ_IN_PROCESS )
      wire#w1
      Contact( "DB1030_TEST_STOP".TEST_STP_TST_BRK_AX_12 )
      wire#w2
      Contact( "DB1046_C22_BRAKE_TEST".BRAKE_TEST_DONE )
      wire#w3
      I_Contact( "DB1030_TEST_STOP".TEST_STP_TST_BRK_AX_14 )
      I_Contact( "DB1030_TEST_STOP".TST_STP_FIRST_SCAN_REQUEST )
      Coil( "DB1030_TEST_STOP".TEST_STP_TST_BRK_AX_13 )
   END_RUNG
   RUNG wire#w2
      I_Contact( #BRAKE_TEST_AXIS_C22 )
   END_RUNG wire#w3
   RUNG wire#w1
      Contact( "DB1030_TEST_STOP".TEST_STP_TST_BRK_AX_13 )
   END_RUNG wire#w3
   // the same network as SCL:
   "DB1030_TEST_STOP".TEST_STP_TST_BRK_AX_13 := "DB1030_TEST_STOP".TEST_STP_SQ_IN_PROCESS AND (("DB1030_TEST_STOP".TEST_STP_TST_BRK_AX_12 AND ("DB1046_C22_BRAKE_TEST".BRAKE_TEST_DONE OR NOT #BRAKE_TEST_AXIS_C22)) OR "DB1030_TEST_STOP".TEST_STP_TST_BRK_AX_13) AND NOT "DB1030_TEST_STOP".TEST_STP_TST_BRK_AX_14 AND NOT "DB1030_TEST_STOP".TST_STP_FIRST_SCAN_REQUEST;
END_REGION

REGION Network 38: CALL FB1031 BRAKE TEST AXIS 13
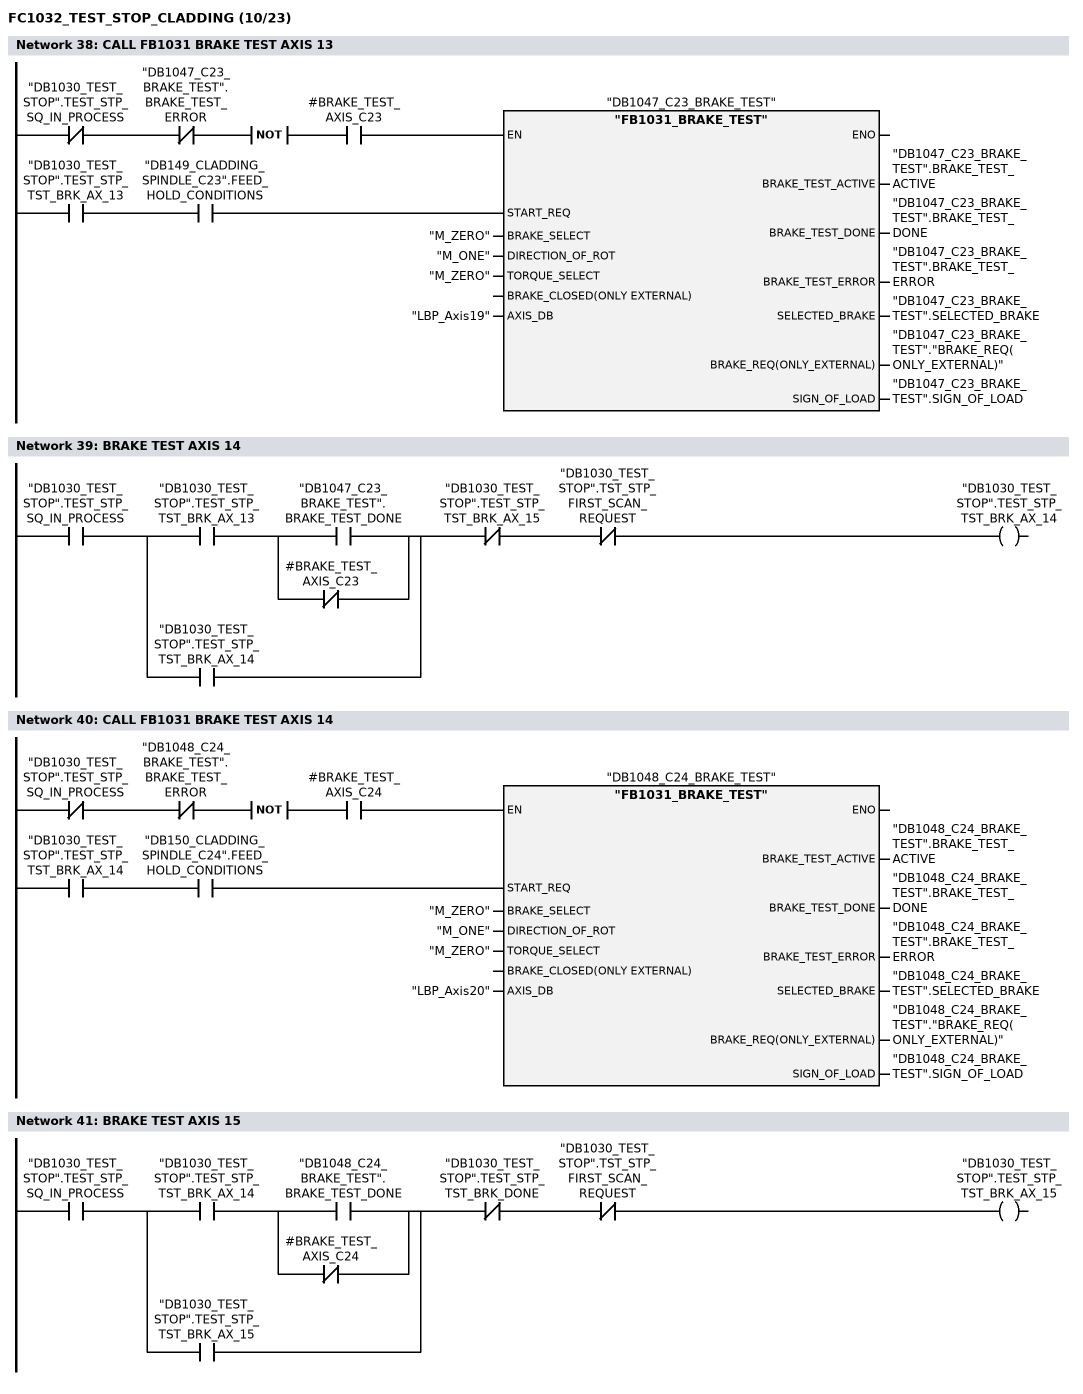
   RUNG wire#powerrail
      I_Contact( "DB1030_TEST_STOP".TEST_STP_SQ_IN_PROCESS )
      I_Contact( "DB1047_C23_BRAKE_TEST".BRAKE_TEST_ERROR )
      Not()
      Contact( #BRAKE_TEST_AXIS_C23 )
      "DB1047_C23_BRAKE_TEST"(START_REQ := wire#w1, BRAKE_SELECT := "M_ZERO", DIRECTION_OF_ROT := "M_ONE", TORQUE_SELECT := "M_ZERO", "BRAKE_CLOSED(ONLY EXTERNAL)" :=, AXIS_DB := "LBP_Axis19", BRAKE_TEST_ACTIVE => "DB1047_C23_BRAKE_TEST".BRAKE_TEST_ACTIVE, BRAKE_TEST_DONE => "DB1047_C23_BRAKE_TEST".BRAKE_TEST_DONE, BRAKE_TEST_ERROR => "DB1047_C23_BRAKE_TEST".BRAKE_TEST_ERROR, SELECTED_BRAKE => "DB1047_C23_BRAKE_TEST".SELECTED_BRAKE, "BRAKE_REQ(ONLY_EXTERNAL)" => "DB1047_C23_BRAKE_TEST"."BRAKE_REQ(ONLY_EXTERNAL)", SIGN_OF_LOAD => "DB1047_C23_BRAKE_TEST".SIGN_OF_LOAD)
   END_RUNG
   RUNG wire#powerrail
      Contact( "DB1030_TEST_STOP".TEST_STP_TST_BRK_AX_13 )
      Contact( "DB149_CLADDING_SPINDLE_C23".FEED_HOLD_CONDITIONS )
   END_RUNG wire#w1
   // the same network as SCL:
   IF NOT (NOT "DB1030_TEST_STOP".TEST_STP_SQ_IN_PROCESS AND NOT "DB1047_C23_BRAKE_TEST".BRAKE_TEST_ERROR) AND #BRAKE_TEST_AXIS_C23 THEN
       "DB1047_C23_BRAKE_TEST"(START_REQ := "DB1030_TEST_STOP".TEST_STP_TST_BRK_AX_13 AND "DB149_CLADDING_SPINDLE_C23".FEED_HOLD_CONDITIONS,   // "FB1031_BRAKE_TEST"
                               BRAKE_SELECT := "M_ZERO",
                               DIRECTION_OF_ROT := "M_ONE",
                               TORQUE_SELECT := "M_ZERO",
                               AXIS_DB := "LBP_Axis19",
                               BRAKE_TEST_ACTIVE => "DB1047_C23_BRAKE_TEST".BRAKE_TEST_ACTIVE,
                               BRAKE_TEST_DONE => "DB1047_C23_BRAKE_TEST".BRAKE_TEST_DONE,
                               BRAKE_TEST_ERROR => "DB1047_C23_BRAKE_TEST".BRAKE_TEST_ERROR,
                               SELECTED_BRAKE => "DB1047_C23_BRAKE_TEST".SELECTED_BRAKE,
                               "BRAKE_REQ(ONLY_EXTERNAL)" => "DB1047_C23_BRAKE_TEST"."BRAKE_REQ(ONLY_EXTERNAL)",
                               SIGN_OF_LOAD => "DB1047_C23_BRAKE_TEST".SIGN_OF_LOAD);
   END_IF;
END_REGION

REGION Network 39: BRAKE TEST AXIS 14
   RUNG wire#powerrail
      Contact( "DB1030_TEST_STOP".TEST_STP_SQ_IN_PROCESS )
      wire#w1
      Contact( "DB1030_TEST_STOP".TEST_STP_TST_BRK_AX_13 )
      wire#w2
      Contact( "DB1047_C23_BRAKE_TEST".BRAKE_TEST_DONE )
      wire#w3
      I_Contact( "DB1030_TEST_STOP".TEST_STP_TST_BRK_AX_15 )
      I_Contact( "DB1030_TEST_STOP".TST_STP_FIRST_SCAN_REQUEST )
      Coil( "DB1030_TEST_STOP".TEST_STP_TST_BRK_AX_14 )
   END_RUNG
   RUNG wire#w2
      I_Contact( #BRAKE_TEST_AXIS_C23 )
   END_RUNG wire#w3
   RUNG wire#w1
      Contact( "DB1030_TEST_STOP".TEST_STP_TST_BRK_AX_14 )
   END_RUNG wire#w3
   // the same network as SCL:
   "DB1030_TEST_STOP".TEST_STP_TST_BRK_AX_14 := "DB1030_TEST_STOP".TEST_STP_SQ_IN_PROCESS AND (("DB1030_TEST_STOP".TEST_STP_TST_BRK_AX_13 AND ("DB1047_C23_BRAKE_TEST".BRAKE_TEST_DONE OR NOT #BRAKE_TEST_AXIS_C23)) OR "DB1030_TEST_STOP".TEST_STP_TST_BRK_AX_14) AND NOT "DB1030_TEST_STOP".TEST_STP_TST_BRK_AX_15 AND NOT "DB1030_TEST_STOP".TST_STP_FIRST_SCAN_REQUEST;
END_REGION

REGION Network 40: CALL FB1031 BRAKE TEST AXIS 14
   RUNG wire#powerrail
      I_Contact( "DB1030_TEST_STOP".TEST_STP_SQ_IN_PROCESS )
      I_Contact( "DB1048_C24_BRAKE_TEST".BRAKE_TEST_ERROR )
      Not()
      Contact( #BRAKE_TEST_AXIS_C24 )
      "DB1048_C24_BRAKE_TEST"(START_REQ := wire#w1, BRAKE_SELECT := "M_ZERO", DIRECTION_OF_ROT := "M_ONE", TORQUE_SELECT := "M_ZERO", "BRAKE_CLOSED(ONLY EXTERNAL)" :=, AXIS_DB := "LBP_Axis20", BRAKE_TEST_ACTIVE => "DB1048_C24_BRAKE_TEST".BRAKE_TEST_ACTIVE, BRAKE_TEST_DONE => "DB1048_C24_BRAKE_TEST".BRAKE_TEST_DONE, BRAKE_TEST_ERROR => "DB1048_C24_BRAKE_TEST".BRAKE_TEST_ERROR, SELECTED_BRAKE => "DB1048_C24_BRAKE_TEST".SELECTED_BRAKE, "BRAKE_REQ(ONLY_EXTERNAL)" => "DB1048_C24_BRAKE_TEST"."BRAKE_REQ(ONLY_EXTERNAL)", SIGN_OF_LOAD => "DB1048_C24_BRAKE_TEST".SIGN_OF_LOAD)
   END_RUNG
   RUNG wire#powerrail
      Contact( "DB1030_TEST_STOP".TEST_STP_TST_BRK_AX_14 )
      Contact( "DB150_CLADDING_SPINDLE_C24".FEED_HOLD_CONDITIONS )
   END_RUNG wire#w1
   // the same network as SCL:
   IF NOT (NOT "DB1030_TEST_STOP".TEST_STP_SQ_IN_PROCESS AND NOT "DB1048_C24_BRAKE_TEST".BRAKE_TEST_ERROR) AND #BRAKE_TEST_AXIS_C24 THEN
       "DB1048_C24_BRAKE_TEST"(START_REQ := "DB1030_TEST_STOP".TEST_STP_TST_BRK_AX_14 AND "DB150_CLADDING_SPINDLE_C24".FEED_HOLD_CONDITIONS,   // "FB1031_BRAKE_TEST"
                               BRAKE_SELECT := "M_ZERO",
                               DIRECTION_OF_ROT := "M_ONE",
                               TORQUE_SELECT := "M_ZERO",
                               AXIS_DB := "LBP_Axis20",
                               BRAKE_TEST_ACTIVE => "DB1048_C24_BRAKE_TEST".BRAKE_TEST_ACTIVE,
                               BRAKE_TEST_DONE => "DB1048_C24_BRAKE_TEST".BRAKE_TEST_DONE,
                               BRAKE_TEST_ERROR => "DB1048_C24_BRAKE_TEST".BRAKE_TEST_ERROR,
                               SELECTED_BRAKE => "DB1048_C24_BRAKE_TEST".SELECTED_BRAKE,
                               "BRAKE_REQ(ONLY_EXTERNAL)" => "DB1048_C24_BRAKE_TEST"."BRAKE_REQ(ONLY_EXTERNAL)",
                               SIGN_OF_LOAD => "DB1048_C24_BRAKE_TEST".SIGN_OF_LOAD);
   END_IF;
END_REGION

REGION Network 41: BRAKE TEST AXIS 15
   RUNG wire#powerrail
      Contact( "DB1030_TEST_STOP".TEST_STP_SQ_IN_PROCESS )
      wire#w1
      Contact( "DB1030_TEST_STOP".TEST_STP_TST_BRK_AX_14 )
      wire#w2
      Contact( "DB1048_C24_BRAKE_TEST".BRAKE_TEST_DONE )
      wire#w3
      I_Contact( "DB1030_TEST_STOP".TEST_STP_TST_BRK_DONE )
      I_Contact( "DB1030_TEST_STOP".TST_STP_FIRST_SCAN_REQUEST )
      Coil( "DB1030_TEST_STOP".TEST_STP_TST_BRK_AX_15 )
   END_RUNG
   RUNG wire#w2
      I_Contact( #BRAKE_TEST_AXIS_C24 )
   END_RUNG wire#w3
   RUNG wire#w1
      Contact( "DB1030_TEST_STOP".TEST_STP_TST_BRK_AX_15 )
   END_RUNG wire#w3
   // the same network as SCL:
   "DB1030_TEST_STOP".TEST_STP_TST_BRK_AX_15 := "DB1030_TEST_STOP".TEST_STP_SQ_IN_PROCESS AND (("DB1030_TEST_STOP".TEST_STP_TST_BRK_AX_14 AND ("DB1048_C24_BRAKE_TEST".BRAKE_TEST_DONE OR NOT #BRAKE_TEST_AXIS_C24)) OR "DB1030_TEST_STOP".TEST_STP_TST_BRK_AX_15) AND NOT "DB1030_TEST_STOP".TEST_STP_TST_BRK_DONE AND NOT "DB1030_TEST_STOP".TST_STP_FIRST_SCAN_REQUEST;
END_REGION

REGION Network 42: CALL FB1031 BRAKE TEST AXIS 15
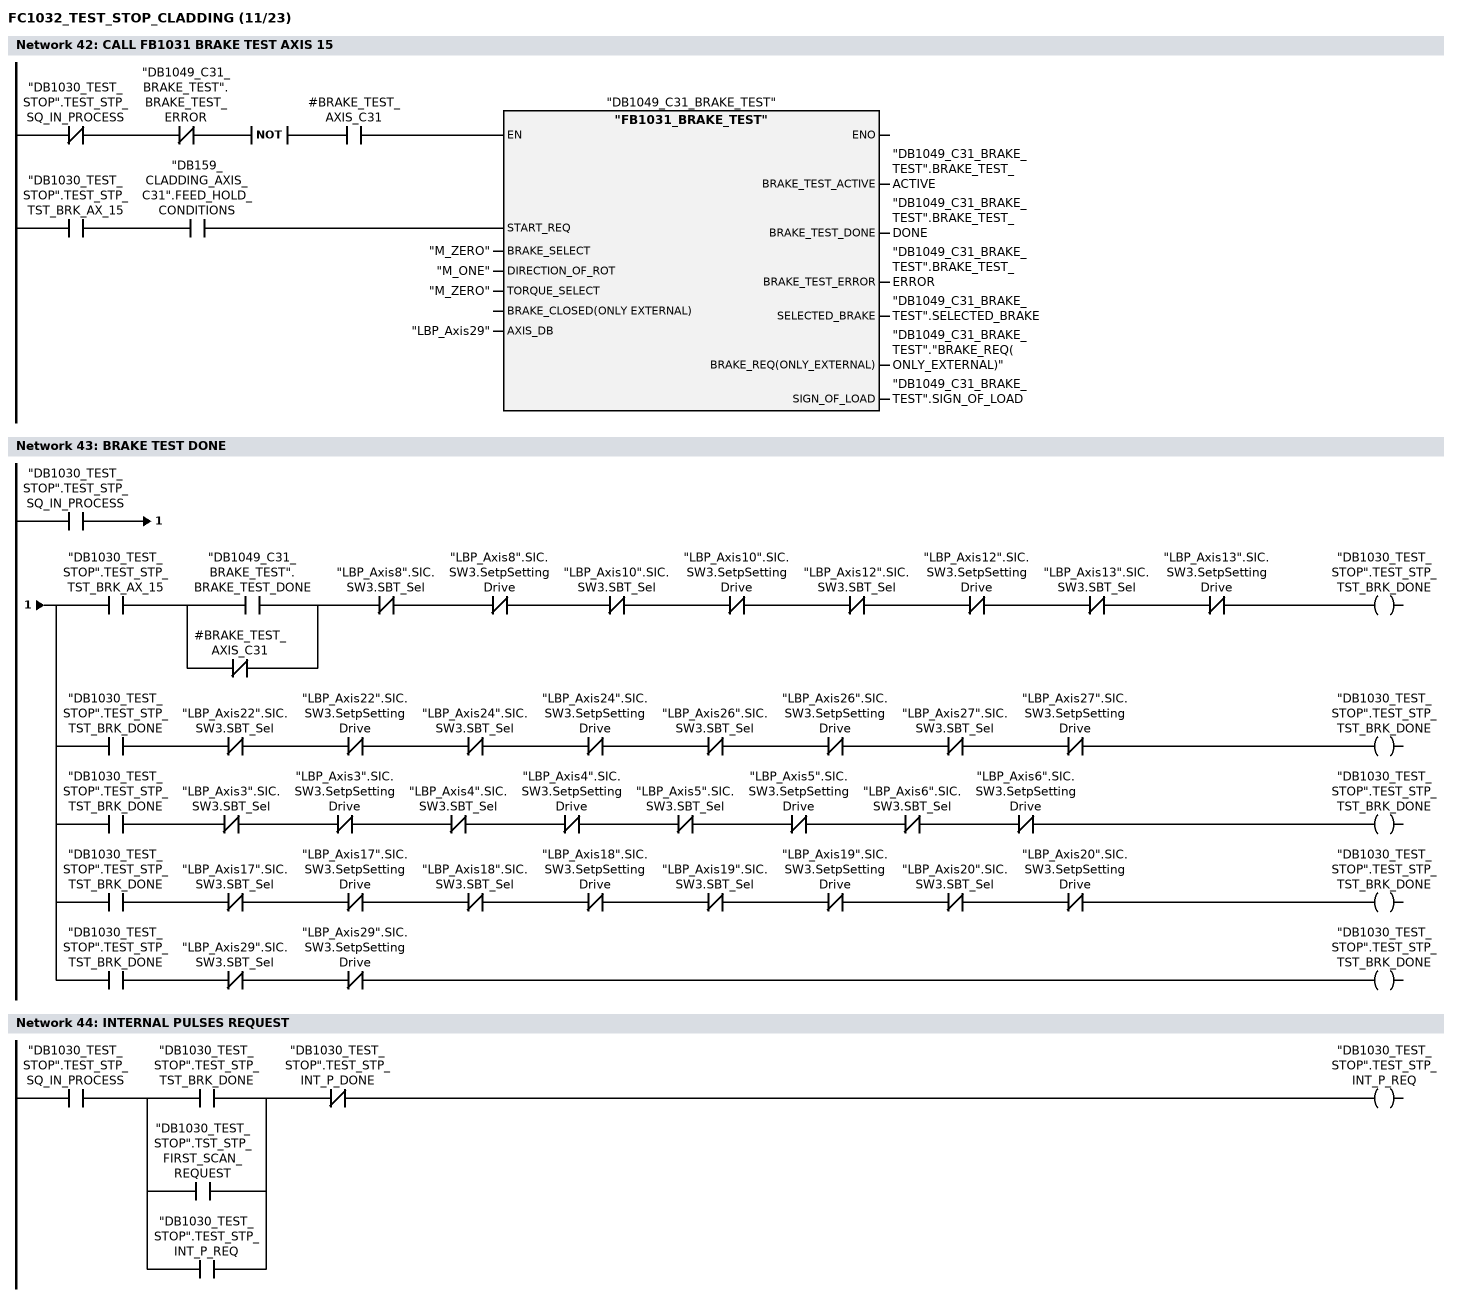
   RUNG wire#powerrail
      I_Contact( "DB1030_TEST_STOP".TEST_STP_SQ_IN_PROCESS )
      I_Contact( "DB1049_C31_BRAKE_TEST".BRAKE_TEST_ERROR )
      Not()
      Contact( #BRAKE_TEST_AXIS_C31 )
      "DB1049_C31_BRAKE_TEST"(START_REQ := wire#w1, BRAKE_SELECT := "M_ZERO", DIRECTION_OF_ROT := "M_ONE", TORQUE_SELECT := "M_ZERO", "BRAKE_CLOSED(ONLY EXTERNAL)" :=, AXIS_DB := "LBP_Axis29", BRAKE_TEST_ACTIVE => "DB1049_C31_BRAKE_TEST".BRAKE_TEST_ACTIVE, BRAKE_TEST_DONE => "DB1049_C31_BRAKE_TEST".BRAKE_TEST_DONE, BRAKE_TEST_ERROR => "DB1049_C31_BRAKE_TEST".BRAKE_TEST_ERROR, SELECTED_BRAKE => "DB1049_C31_BRAKE_TEST".SELECTED_BRAKE, "BRAKE_REQ(ONLY_EXTERNAL)" => "DB1049_C31_BRAKE_TEST"."BRAKE_REQ(ONLY_EXTERNAL)", SIGN_OF_LOAD => "DB1049_C31_BRAKE_TEST".SIGN_OF_LOAD)
   END_RUNG
   RUNG wire#powerrail
      Contact( "DB1030_TEST_STOP".TEST_STP_TST_BRK_AX_15 )
      Contact( "DB159_CLADDING_AXIS_C31".FEED_HOLD_CONDITIONS )
   END_RUNG wire#w1
   // the same network as SCL:
   IF NOT (NOT "DB1030_TEST_STOP".TEST_STP_SQ_IN_PROCESS AND NOT "DB1049_C31_BRAKE_TEST".BRAKE_TEST_ERROR) AND #BRAKE_TEST_AXIS_C31 THEN
       "DB1049_C31_BRAKE_TEST"(START_REQ := "DB1030_TEST_STOP".TEST_STP_TST_BRK_AX_15 AND "DB159_CLADDING_AXIS_C31".FEED_HOLD_CONDITIONS,   // "FB1031_BRAKE_TEST"
                               BRAKE_SELECT := "M_ZERO",
                               DIRECTION_OF_ROT := "M_ONE",
                               TORQUE_SELECT := "M_ZERO",
                               AXIS_DB := "LBP_Axis29",
                               BRAKE_TEST_ACTIVE => "DB1049_C31_BRAKE_TEST".BRAKE_TEST_ACTIVE,
                               BRAKE_TEST_DONE => "DB1049_C31_BRAKE_TEST".BRAKE_TEST_DONE,
                               BRAKE_TEST_ERROR => "DB1049_C31_BRAKE_TEST".BRAKE_TEST_ERROR,
                               SELECTED_BRAKE => "DB1049_C31_BRAKE_TEST".SELECTED_BRAKE,
                               "BRAKE_REQ(ONLY_EXTERNAL)" => "DB1049_C31_BRAKE_TEST"."BRAKE_REQ(ONLY_EXTERNAL)",
                               SIGN_OF_LOAD => "DB1049_C31_BRAKE_TEST".SIGN_OF_LOAD);
   END_IF;
END_REGION

REGION Network 43: BRAKE TEST DONE
   RUNG wire#powerrail
      Contact( "DB1030_TEST_STOP".TEST_STP_SQ_IN_PROCESS )
      wire#w1
      Contact( "DB1030_TEST_STOP".TEST_STP_TST_BRK_AX_15 )
      wire#w2
      Contact( "DB1049_C31_BRAKE_TEST".BRAKE_TEST_DONE )
      wire#w3
      I_Contact( "LBP_Axis8".SIC.SW3.SBT_Sel )
      I_Contact( "LBP_Axis8".SIC.SW3.SetpSettingDrive )
      I_Contact( "LBP_Axis10".SIC.SW3.SBT_Sel )
      I_Contact( "LBP_Axis10".SIC.SW3.SetpSettingDrive )
      I_Contact( "LBP_Axis12".SIC.SW3.SBT_Sel )
      I_Contact( "LBP_Axis12".SIC.SW3.SetpSettingDrive )
      I_Contact( "LBP_Axis13".SIC.SW3.SBT_Sel )
      I_Contact( "LBP_Axis13".SIC.SW3.SetpSettingDrive )
      Coil( "DB1030_TEST_STOP".TEST_STP_TST_BRK_DONE )
   END_RUNG
   RUNG wire#w2
      I_Contact( #BRAKE_TEST_AXIS_C31 )
   END_RUNG wire#w3
   RUNG wire#w1
      Contact( "DB1030_TEST_STOP".TEST_STP_TST_BRK_DONE )
      I_Contact( "LBP_Axis22".SIC.SW3.SBT_Sel )
      I_Contact( "LBP_Axis22".SIC.SW3.SetpSettingDrive )
      I_Contact( "LBP_Axis24".SIC.SW3.SBT_Sel )
      I_Contact( "LBP_Axis24".SIC.SW3.SetpSettingDrive )
      I_Contact( "LBP_Axis26".SIC.SW3.SBT_Sel )
      I_Contact( "LBP_Axis26".SIC.SW3.SetpSettingDrive )
      I_Contact( "LBP_Axis27".SIC.SW3.SBT_Sel )
      I_Contact( "LBP_Axis27".SIC.SW3.SetpSettingDrive )
      Coil( "DB1030_TEST_STOP".TEST_STP_TST_BRK_DONE )
   END_RUNG
   RUNG wire#w1
      Contact( "DB1030_TEST_STOP".TEST_STP_TST_BRK_DONE )
      I_Contact( "LBP_Axis3".SIC.SW3.SBT_Sel )
      I_Contact( "LBP_Axis3".SIC.SW3.SetpSettingDrive )
      I_Contact( "LBP_Axis4".SIC.SW3.SBT_Sel )
      I_Contact( "LBP_Axis4".SIC.SW3.SetpSettingDrive )
      I_Contact( "LBP_Axis5".SIC.SW3.SBT_Sel )
      I_Contact( "LBP_Axis5".SIC.SW3.SetpSettingDrive )
      I_Contact( "LBP_Axis6".SIC.SW3.SBT_Sel )
      I_Contact( "LBP_Axis6".SIC.SW3.SetpSettingDrive )
      Coil( "DB1030_TEST_STOP".TEST_STP_TST_BRK_DONE )
   END_RUNG
   RUNG wire#w1
      Contact( "DB1030_TEST_STOP".TEST_STP_TST_BRK_DONE )
      I_Contact( "LBP_Axis17".SIC.SW3.SBT_Sel )
      I_Contact( "LBP_Axis17".SIC.SW3.SetpSettingDrive )
      I_Contact( "LBP_Axis18".SIC.SW3.SBT_Sel )
      I_Contact( "LBP_Axis18".SIC.SW3.SetpSettingDrive )
      I_Contact( "LBP_Axis19".SIC.SW3.SBT_Sel )
      I_Contact( "LBP_Axis19".SIC.SW3.SetpSettingDrive )
      I_Contact( "LBP_Axis20".SIC.SW3.SBT_Sel )
      I_Contact( "LBP_Axis20".SIC.SW3.SetpSettingDrive )
      Coil( "DB1030_TEST_STOP".TEST_STP_TST_BRK_DONE )
   END_RUNG
   RUNG wire#w1
      Contact( "DB1030_TEST_STOP".TEST_STP_TST_BRK_DONE )
      I_Contact( "LBP_Axis29".SIC.SW3.SBT_Sel )
      I_Contact( "LBP_Axis29".SIC.SW3.SetpSettingDrive )
      Coil( "DB1030_TEST_STOP".TEST_STP_TST_BRK_DONE )
   END_RUNG
   // the same network as SCL:
   "DB1030_TEST_STOP".TEST_STP_TST_BRK_DONE := "DB1030_TEST_STOP".TEST_STP_SQ_IN_PROCESS AND "DB1030_TEST_STOP".TEST_STP_TST_BRK_AX_15 AND ("DB1049_C31_BRAKE_TEST".BRAKE_TEST_DONE OR NOT #BRAKE_TEST_AXIS_C31) AND NOT "LBP_Axis8".SIC.SW3.SBT_Sel AND NOT "LBP_Axis8".SIC.SW3.SetpSettingDrive AND NOT "LBP_Axis10".SIC.SW3.SBT_Sel AND NOT "LBP_Axis10".SIC.SW3.SetpSettingDrive AND NOT "LBP_Axis12".SIC.SW3.SBT_Sel AND NOT "LBP_Axis12".SIC.SW3.SetpSettingDrive AND NOT "LBP_Axis13".SIC.SW3.SBT_Sel AND NOT "LBP_Axis13".SIC.SW3.SetpSettingDrive;
   "DB1030_TEST_STOP".TEST_STP_TST_BRK_DONE := "DB1030_TEST_STOP".TEST_STP_SQ_IN_PROCESS AND "DB1030_TEST_STOP".TEST_STP_TST_BRK_DONE AND NOT "LBP_Axis22".SIC.SW3.SBT_Sel AND NOT "LBP_Axis22".SIC.SW3.SetpSettingDrive AND NOT "LBP_Axis24".SIC.SW3.SBT_Sel AND NOT "LBP_Axis24".SIC.SW3.SetpSettingDrive AND NOT "LBP_Axis26".SIC.SW3.SBT_Sel AND NOT "LBP_Axis26".SIC.SW3.SetpSettingDrive AND NOT "LBP_Axis27".SIC.SW3.SBT_Sel AND NOT "LBP_Axis27".SIC.SW3.SetpSettingDrive;
   "DB1030_TEST_STOP".TEST_STP_TST_BRK_DONE := "DB1030_TEST_STOP".TEST_STP_SQ_IN_PROCESS AND "DB1030_TEST_STOP".TEST_STP_TST_BRK_DONE AND NOT "LBP_Axis3".SIC.SW3.SBT_Sel AND NOT "LBP_Axis3".SIC.SW3.SetpSettingDrive AND NOT "LBP_Axis4".SIC.SW3.SBT_Sel AND NOT "LBP_Axis4".SIC.SW3.SetpSettingDrive AND NOT "LBP_Axis5".SIC.SW3.SBT_Sel AND NOT "LBP_Axis5".SIC.SW3.SetpSettingDrive AND NOT "LBP_Axis6".SIC.SW3.SBT_Sel AND NOT "LBP_Axis6".SIC.SW3.SetpSettingDrive;
   "DB1030_TEST_STOP".TEST_STP_TST_BRK_DONE := "DB1030_TEST_STOP".TEST_STP_SQ_IN_PROCESS AND "DB1030_TEST_STOP".TEST_STP_TST_BRK_DONE AND NOT "LBP_Axis17".SIC.SW3.SBT_Sel AND NOT "LBP_Axis17".SIC.SW3.SetpSettingDrive AND NOT "LBP_Axis18".SIC.SW3.SBT_Sel AND NOT "LBP_Axis18".SIC.SW3.SetpSettingDrive AND NOT "LBP_Axis19".SIC.SW3.SBT_Sel AND NOT "LBP_Axis19".SIC.SW3.SetpSettingDrive AND NOT "LBP_Axis20".SIC.SW3.SBT_Sel AND NOT "LBP_Axis20".SIC.SW3.SetpSettingDrive;
   "DB1030_TEST_STOP".TEST_STP_TST_BRK_DONE := "DB1030_TEST_STOP".TEST_STP_SQ_IN_PROCESS AND "DB1030_TEST_STOP".TEST_STP_TST_BRK_DONE AND NOT "LBP_Axis29".SIC.SW3.SBT_Sel AND NOT "LBP_Axis29".SIC.SW3.SetpSettingDrive;
END_REGION

REGION Network 44: INTERNAL PULSES REQUEST
   RUNG wire#powerrail
      Contact( "DB1030_TEST_STOP".TEST_STP_SQ_IN_PROCESS )
      wire#w1
      Contact( "DB1030_TEST_STOP".TEST_STP_TST_BRK_DONE )
      wire#w2
      I_Contact( "DB1030_TEST_STOP".TEST_STP_INT_P_DONE )
      Coil( "DB1030_TEST_STOP".TEST_STP_INT_P_REQ )
   END_RUNG
   RUNG wire#w1
      Contact( "DB1030_TEST_STOP".TST_STP_FIRST_SCAN_REQUEST )
   END_RUNG wire#w2
   RUNG wire#w1
      Contact( "DB1030_TEST_STOP".TEST_STP_INT_P_REQ )
   END_RUNG wire#w2
   // the same network as SCL:
   "DB1030_TEST_STOP".TEST_STP_INT_P_REQ := "DB1030_TEST_STOP".TEST_STP_SQ_IN_PROCESS AND ("DB1030_TEST_STOP".TEST_STP_TST_BRK_DONE OR "DB1030_TEST_STOP".TST_STP_FIRST_SCAN_REQUEST OR "DB1030_TEST_STOP".TEST_STP_INT_P_REQ) AND NOT "DB1030_TEST_STOP".TEST_STP_INT_P_DONE;
END_REGION

REGION Network 45: INTERNAL PULSES REQUEST AUXILIARY
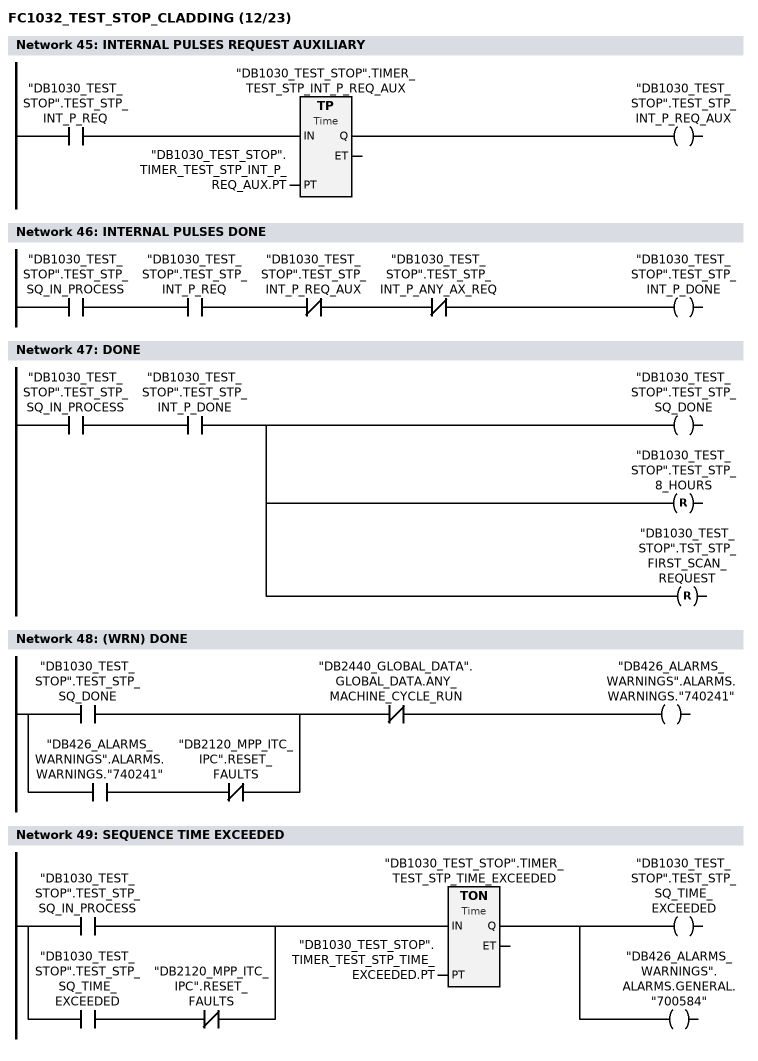
   RUNG wire#powerrail
      Contact( "DB1030_TEST_STOP".TEST_STP_INT_P_REQ )
      { S7_Templates := "time_type := Time" } "DB1030_TEST_STOP".TIMER_TEST_STP_INT_P_REQ_AUX.TP(pt := "DB1030_TEST_STOP".TIMER_TEST_STP_INT_P_REQ_AUX.PT, et =>)
      Coil( "DB1030_TEST_STOP".TEST_STP_INT_P_REQ_AUX )
   END_RUNG
   // the same network as SCL:
   "DB1030_TEST_STOP".TIMER_TEST_STP_INT_P_REQ_AUX.TP(IN := "DB1030_TEST_STOP".TEST_STP_INT_P_REQ,
                           PT := "DB1030_TEST_STOP".TIMER_TEST_STP_INT_P_REQ_AUX.PT);
   "DB1030_TEST_STOP".TEST_STP_INT_P_REQ_AUX := "DB1030_TEST_STOP".TIMER_TEST_STP_INT_P_REQ_AUX.Q;
END_REGION

REGION Network 46: INTERNAL PULSES DONE
   RUNG wire#powerrail
      Contact( "DB1030_TEST_STOP".TEST_STP_SQ_IN_PROCESS )
      Contact( "DB1030_TEST_STOP".TEST_STP_INT_P_REQ )
      I_Contact( "DB1030_TEST_STOP".TEST_STP_INT_P_REQ_AUX )
      I_Contact( "DB1030_TEST_STOP".TEST_STP_INT_P_ANY_AX_REQ )
      Coil( "DB1030_TEST_STOP".TEST_STP_INT_P_DONE )
   END_RUNG
   // the same network as SCL:
   "DB1030_TEST_STOP".TEST_STP_INT_P_DONE := "DB1030_TEST_STOP".TEST_STP_SQ_IN_PROCESS AND "DB1030_TEST_STOP".TEST_STP_INT_P_REQ AND NOT "DB1030_TEST_STOP".TEST_STP_INT_P_REQ_AUX AND NOT "DB1030_TEST_STOP".TEST_STP_INT_P_ANY_AX_REQ;
END_REGION

REGION Network 47: DONE
   RUNG wire#powerrail
      Contact( "DB1030_TEST_STOP".TEST_STP_SQ_IN_PROCESS )
      Contact( "DB1030_TEST_STOP".TEST_STP_INT_P_DONE )
      wire#w1
      Coil( "DB1030_TEST_STOP".TEST_STP_SQ_DONE )
   END_RUNG
   RUNG wire#w1
      R_Coil( "DB1030_TEST_STOP".TEST_STP_8_HOURS )
   END_RUNG
   RUNG wire#w1
      R_Coil( "DB1030_TEST_STOP".TST_STP_FIRST_SCAN_REQUEST )
   END_RUNG
   // the same network as SCL:
   "DB1030_TEST_STOP".TEST_STP_SQ_DONE := "DB1030_TEST_STOP".TEST_STP_SQ_IN_PROCESS AND "DB1030_TEST_STOP".TEST_STP_INT_P_DONE;
   IF "DB1030_TEST_STOP".TEST_STP_SQ_DONE THEN
       "DB1030_TEST_STOP".TEST_STP_8_HOURS := FALSE;
       "DB1030_TEST_STOP".TST_STP_FIRST_SCAN_REQUEST := FALSE;
   END_IF;
END_REGION

REGION Network 48: (WRN) DONE
   RUNG wire#powerrail
      Contact( "DB1030_TEST_STOP".TEST_STP_SQ_DONE )
      wire#w1
      I_Contact( "DB2440_GLOBAL_DATA".GLOBAL_DATA.ANY_MACHINE_CYCLE_RUN )
      Coil( "DB426_ALARMS_WARNINGS".ALARMS.WARNINGS."740241" )
   END_RUNG
   RUNG wire#powerrail
      Contact( "DB426_ALARMS_WARNINGS".ALARMS.WARNINGS."740241" )
      I_Contact( "DB2120_MPP_ITC_IPC".RESET_FAULTS )
   END_RUNG wire#w1
   // the same network as SCL:
   "DB426_ALARMS_WARNINGS".ALARMS.WARNINGS."740241" := ("DB1030_TEST_STOP".TEST_STP_SQ_DONE OR ("DB426_ALARMS_WARNINGS".ALARMS.WARNINGS."740241" AND NOT "DB2120_MPP_ITC_IPC".RESET_FAULTS)) AND NOT "DB2440_GLOBAL_DATA".GLOBAL_DATA.ANY_MACHINE_CYCLE_RUN;
END_REGION

REGION Network 49: SEQUENCE TIME EXCEEDED
   RUNG wire#powerrail
      Contact( "DB1030_TEST_STOP".TEST_STP_SQ_IN_PROCESS )
      wire#w1
      { S7_Templates := "time_type := Time" } "DB1030_TEST_STOP".TIMER_TEST_STP_TIME_EXCEEDED.TON(pt := "DB1030_TEST_STOP".TIMER_TEST_STP_TIME_EXCEEDED.PT, et =>)
      wire#w2
      Coil( "DB1030_TEST_STOP".TEST_STP_SQ_TIME_EXCEEDED )
   END_RUNG
   RUNG wire#powerrail
      Contact( "DB1030_TEST_STOP".TEST_STP_SQ_TIME_EXCEEDED )
      I_Contact( "DB2120_MPP_ITC_IPC".RESET_FAULTS )
   END_RUNG wire#w1
   RUNG wire#w2
      Coil( "DB426_ALARMS_WARNINGS".ALARMS.GENERAL."700584" )
   END_RUNG
   // the same network as SCL:
   "DB1030_TEST_STOP".TIMER_TEST_STP_TIME_EXCEEDED.TON(IN := "DB1030_TEST_STOP".TEST_STP_SQ_IN_PROCESS OR ("DB1030_TEST_STOP".TEST_STP_SQ_TIME_EXCEEDED AND NOT "DB2120_MPP_ITC_IPC".RESET_FAULTS),
                           PT := "DB1030_TEST_STOP".TIMER_TEST_STP_TIME_EXCEEDED.PT);
   "DB1030_TEST_STOP".TEST_STP_SQ_TIME_EXCEEDED := "DB1030_TEST_STOP".TIMER_TEST_STP_TIME_EXCEEDED.Q;
   "DB426_ALARMS_WARNINGS".ALARMS.GENERAL."700584" := "DB1030_TEST_STOP".TIMER_TEST_STP_TIME_EXCEEDED.Q;
END_REGION

REGION Network 50: INTERNAL PULSES ANY AXIS REQUEST
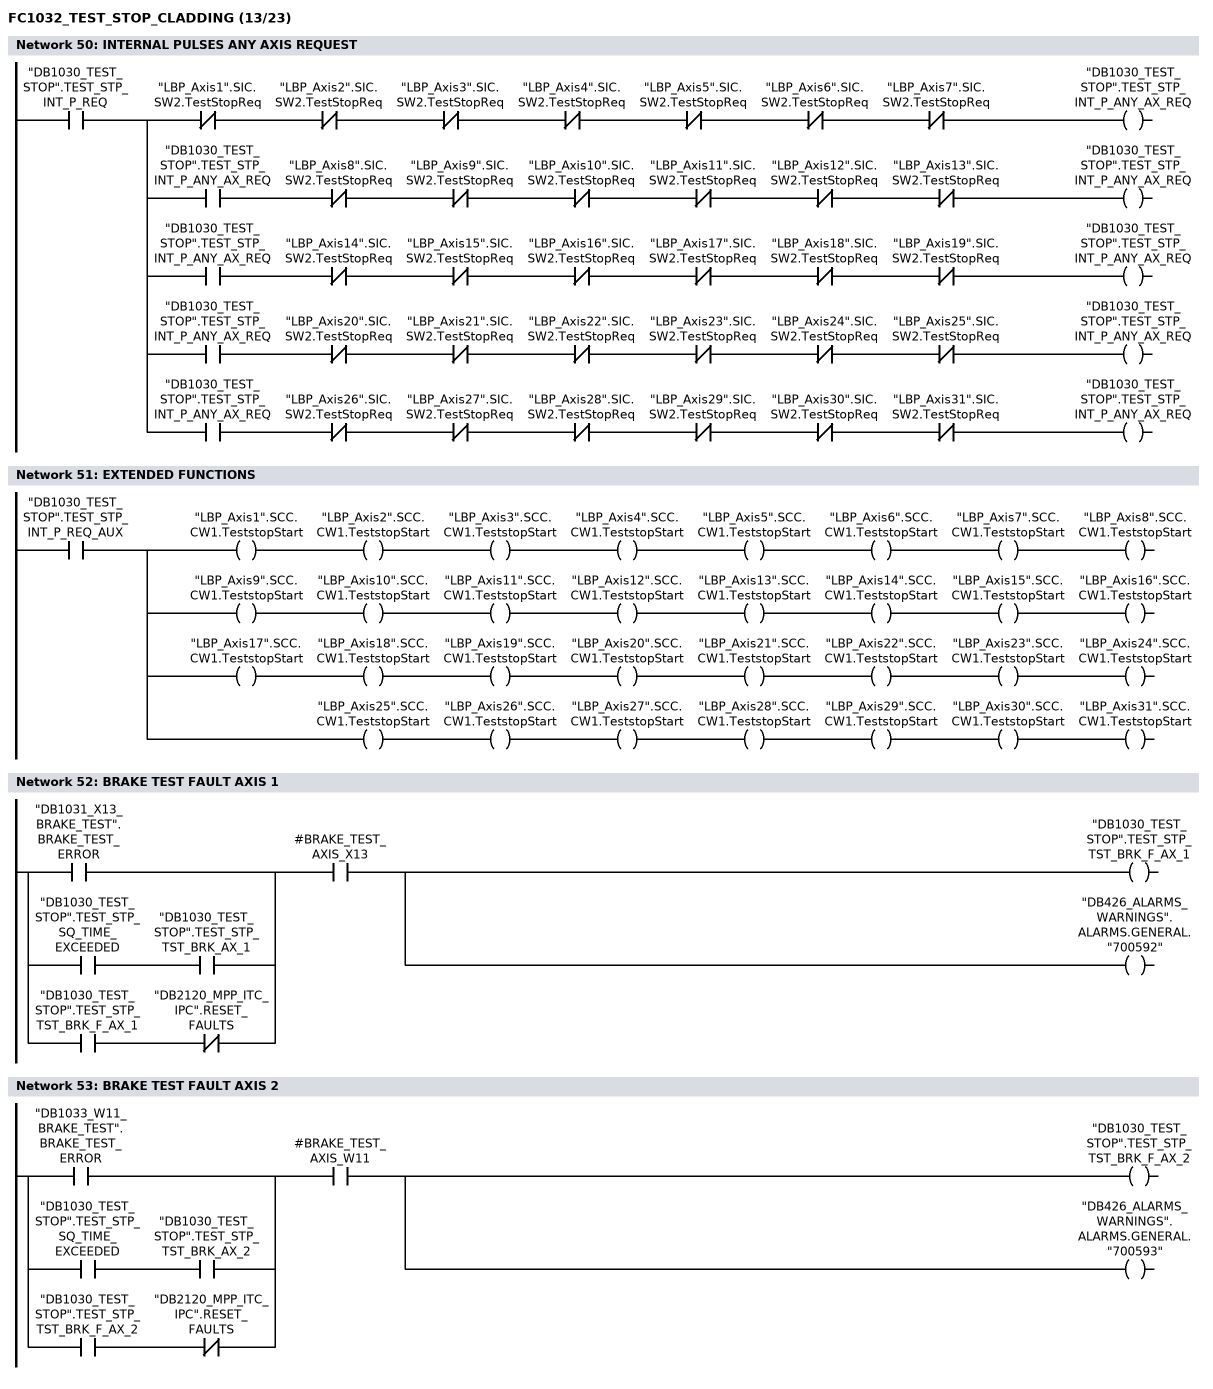
   RUNG wire#powerrail
      Contact( "DB1030_TEST_STOP".TEST_STP_INT_P_REQ )
      wire#w1
      I_Contact( "LBP_Axis1".SIC.SW2.TestStopReq )
      I_Contact( "LBP_Axis2".SIC.SW2.TestStopReq )
      I_Contact( "LBP_Axis3".SIC.SW2.TestStopReq )
      I_Contact( "LBP_Axis4".SIC.SW2.TestStopReq )
      I_Contact( "LBP_Axis5".SIC.SW2.TestStopReq )
      I_Contact( "LBP_Axis6".SIC.SW2.TestStopReq )
      I_Contact( "LBP_Axis7".SIC.SW2.TestStopReq )
      Coil( "DB1030_TEST_STOP".TEST_STP_INT_P_ANY_AX_REQ )
   END_RUNG
   RUNG wire#w1
      Contact( "DB1030_TEST_STOP".TEST_STP_INT_P_ANY_AX_REQ )
      I_Contact( "LBP_Axis8".SIC.SW2.TestStopReq )
      I_Contact( "LBP_Axis9".SIC.SW2.TestStopReq )
      I_Contact( "LBP_Axis10".SIC.SW2.TestStopReq )
      I_Contact( "LBP_Axis11".SIC.SW2.TestStopReq )
      I_Contact( "LBP_Axis12".SIC.SW2.TestStopReq )
      I_Contact( "LBP_Axis13".SIC.SW2.TestStopReq )
      Coil( "DB1030_TEST_STOP".TEST_STP_INT_P_ANY_AX_REQ )
   END_RUNG
   RUNG wire#w1
      Contact( "DB1030_TEST_STOP".TEST_STP_INT_P_ANY_AX_REQ )
      I_Contact( "LBP_Axis14".SIC.SW2.TestStopReq )
      I_Contact( "LBP_Axis15".SIC.SW2.TestStopReq )
      I_Contact( "LBP_Axis16".SIC.SW2.TestStopReq )
      I_Contact( "LBP_Axis17".SIC.SW2.TestStopReq )
      I_Contact( "LBP_Axis18".SIC.SW2.TestStopReq )
      I_Contact( "LBP_Axis19".SIC.SW2.TestStopReq )
      Coil( "DB1030_TEST_STOP".TEST_STP_INT_P_ANY_AX_REQ )
   END_RUNG
   RUNG wire#w1
      Contact( "DB1030_TEST_STOP".TEST_STP_INT_P_ANY_AX_REQ )
      I_Contact( "LBP_Axis20".SIC.SW2.TestStopReq )
      I_Contact( "LBP_Axis21".SIC.SW2.TestStopReq )
      I_Contact( "LBP_Axis22".SIC.SW2.TestStopReq )
      I_Contact( "LBP_Axis23".SIC.SW2.TestStopReq )
      I_Contact( "LBP_Axis24".SIC.SW2.TestStopReq )
      I_Contact( "LBP_Axis25".SIC.SW2.TestStopReq )
      Coil( "DB1030_TEST_STOP".TEST_STP_INT_P_ANY_AX_REQ )
   END_RUNG
   RUNG wire#w1
      Contact( "DB1030_TEST_STOP".TEST_STP_INT_P_ANY_AX_REQ )
      I_Contact( "LBP_Axis26".SIC.SW2.TestStopReq )
      I_Contact( "LBP_Axis27".SIC.SW2.TestStopReq )
      I_Contact( "LBP_Axis28".SIC.SW2.TestStopReq )
      I_Contact( "LBP_Axis29".SIC.SW2.TestStopReq )
      I_Contact( "LBP_Axis30".SIC.SW2.TestStopReq )
      I_Contact( "LBP_Axis31".SIC.SW2.TestStopReq )
      Coil( "DB1030_TEST_STOP".TEST_STP_INT_P_ANY_AX_REQ )
   END_RUNG
   // the same network as SCL:
   "DB1030_TEST_STOP".TEST_STP_INT_P_ANY_AX_REQ := "DB1030_TEST_STOP".TEST_STP_INT_P_REQ AND NOT "LBP_Axis1".SIC.SW2.TestStopReq AND NOT "LBP_Axis2".SIC.SW2.TestStopReq AND NOT "LBP_Axis3".SIC.SW2.TestStopReq AND NOT "LBP_Axis4".SIC.SW2.TestStopReq AND NOT "LBP_Axis5".SIC.SW2.TestStopReq AND NOT "LBP_Axis6".SIC.SW2.TestStopReq AND NOT "LBP_Axis7".SIC.SW2.TestStopReq;
   "DB1030_TEST_STOP".TEST_STP_INT_P_ANY_AX_REQ := "DB1030_TEST_STOP".TEST_STP_INT_P_REQ AND "DB1030_TEST_STOP".TEST_STP_INT_P_ANY_AX_REQ AND NOT "LBP_Axis8".SIC.SW2.TestStopReq AND NOT "LBP_Axis9".SIC.SW2.TestStopReq AND NOT "LBP_Axis10".SIC.SW2.TestStopReq AND NOT "LBP_Axis11".SIC.SW2.TestStopReq AND NOT "LBP_Axis12".SIC.SW2.TestStopReq AND NOT "LBP_Axis13".SIC.SW2.TestStopReq;
   "DB1030_TEST_STOP".TEST_STP_INT_P_ANY_AX_REQ := "DB1030_TEST_STOP".TEST_STP_INT_P_REQ AND "DB1030_TEST_STOP".TEST_STP_INT_P_ANY_AX_REQ AND NOT "LBP_Axis14".SIC.SW2.TestStopReq AND NOT "LBP_Axis15".SIC.SW2.TestStopReq AND NOT "LBP_Axis16".SIC.SW2.TestStopReq AND NOT "LBP_Axis17".SIC.SW2.TestStopReq AND NOT "LBP_Axis18".SIC.SW2.TestStopReq AND NOT "LBP_Axis19".SIC.SW2.TestStopReq;
   "DB1030_TEST_STOP".TEST_STP_INT_P_ANY_AX_REQ := "DB1030_TEST_STOP".TEST_STP_INT_P_REQ AND "DB1030_TEST_STOP".TEST_STP_INT_P_ANY_AX_REQ AND NOT "LBP_Axis20".SIC.SW2.TestStopReq AND NOT "LBP_Axis21".SIC.SW2.TestStopReq AND NOT "LBP_Axis22".SIC.SW2.TestStopReq AND NOT "LBP_Axis23".SIC.SW2.TestStopReq AND NOT "LBP_Axis24".SIC.SW2.TestStopReq AND NOT "LBP_Axis25".SIC.SW2.TestStopReq;
   "DB1030_TEST_STOP".TEST_STP_INT_P_ANY_AX_REQ := "DB1030_TEST_STOP".TEST_STP_INT_P_REQ AND "DB1030_TEST_STOP".TEST_STP_INT_P_ANY_AX_REQ AND NOT "LBP_Axis26".SIC.SW2.TestStopReq AND NOT "LBP_Axis27".SIC.SW2.TestStopReq AND NOT "LBP_Axis28".SIC.SW2.TestStopReq AND NOT "LBP_Axis29".SIC.SW2.TestStopReq AND NOT "LBP_Axis30".SIC.SW2.TestStopReq AND NOT "LBP_Axis31".SIC.SW2.TestStopReq;
END_REGION

REGION Network 51: EXTENDED FUNCTIONS
   RUNG wire#powerrail
      Contact( "DB1030_TEST_STOP".TEST_STP_INT_P_REQ_AUX )
      wire#w1
      Coil( "LBP_Axis1".SCC.CW1.TeststopStart )
      Coil( "LBP_Axis2".SCC.CW1.TeststopStart )
      Coil( "LBP_Axis3".SCC.CW1.TeststopStart )
      Coil( "LBP_Axis4".SCC.CW1.TeststopStart )
      Coil( "LBP_Axis5".SCC.CW1.TeststopStart )
      Coil( "LBP_Axis6".SCC.CW1.TeststopStart )
      Coil( "LBP_Axis7".SCC.CW1.TeststopStart )
      Coil( "LBP_Axis8".SCC.CW1.TeststopStart )
   END_RUNG
   RUNG wire#w1
      Coil( "LBP_Axis9".SCC.CW1.TeststopStart )
      Coil( "LBP_Axis10".SCC.CW1.TeststopStart )
      Coil( "LBP_Axis11".SCC.CW1.TeststopStart )
      Coil( "LBP_Axis12".SCC.CW1.TeststopStart )
      Coil( "LBP_Axis13".SCC.CW1.TeststopStart )
      Coil( "LBP_Axis14".SCC.CW1.TeststopStart )
      Coil( "LBP_Axis15".SCC.CW1.TeststopStart )
      Coil( "LBP_Axis16".SCC.CW1.TeststopStart )
   END_RUNG
   RUNG wire#w1
      Coil( "LBP_Axis17".SCC.CW1.TeststopStart )
      Coil( "LBP_Axis18".SCC.CW1.TeststopStart )
      Coil( "LBP_Axis19".SCC.CW1.TeststopStart )
      Coil( "LBP_Axis20".SCC.CW1.TeststopStart )
      Coil( "LBP_Axis21".SCC.CW1.TeststopStart )
      Coil( "LBP_Axis22".SCC.CW1.TeststopStart )
      Coil( "LBP_Axis23".SCC.CW1.TeststopStart )
      Coil( "LBP_Axis24".SCC.CW1.TeststopStart )
   END_RUNG
   RUNG wire#w1
      Coil( "LBP_Axis25".SCC.CW1.TeststopStart )
      Coil( "LBP_Axis26".SCC.CW1.TeststopStart )
      Coil( "LBP_Axis27".SCC.CW1.TeststopStart )
      Coil( "LBP_Axis28".SCC.CW1.TeststopStart )
      Coil( "LBP_Axis29".SCC.CW1.TeststopStart )
      Coil( "LBP_Axis30".SCC.CW1.TeststopStart )
      Coil( "LBP_Axis31".SCC.CW1.TeststopStart )
   END_RUNG
   // the same network as SCL:
   "LBP_Axis1".SCC.CW1.TeststopStart := "DB1030_TEST_STOP".TEST_STP_INT_P_REQ_AUX;
   "LBP_Axis2".SCC.CW1.TeststopStart := "DB1030_TEST_STOP".TEST_STP_INT_P_REQ_AUX;
   "LBP_Axis3".SCC.CW1.TeststopStart := "DB1030_TEST_STOP".TEST_STP_INT_P_REQ_AUX;
   "LBP_Axis4".SCC.CW1.TeststopStart := "DB1030_TEST_STOP".TEST_STP_INT_P_REQ_AUX;
   "LBP_Axis5".SCC.CW1.TeststopStart := "DB1030_TEST_STOP".TEST_STP_INT_P_REQ_AUX;
   "LBP_Axis6".SCC.CW1.TeststopStart := "DB1030_TEST_STOP".TEST_STP_INT_P_REQ_AUX;
   "LBP_Axis7".SCC.CW1.TeststopStart := "DB1030_TEST_STOP".TEST_STP_INT_P_REQ_AUX;
   "LBP_Axis8".SCC.CW1.TeststopStart := "DB1030_TEST_STOP".TEST_STP_INT_P_REQ_AUX;
   "LBP_Axis9".SCC.CW1.TeststopStart := "DB1030_TEST_STOP".TEST_STP_INT_P_REQ_AUX;
   "LBP_Axis10".SCC.CW1.TeststopStart := "DB1030_TEST_STOP".TEST_STP_INT_P_REQ_AUX;
   "LBP_Axis11".SCC.CW1.TeststopStart := "DB1030_TEST_STOP".TEST_STP_INT_P_REQ_AUX;
   "LBP_Axis12".SCC.CW1.TeststopStart := "DB1030_TEST_STOP".TEST_STP_INT_P_REQ_AUX;
   "LBP_Axis13".SCC.CW1.TeststopStart := "DB1030_TEST_STOP".TEST_STP_INT_P_REQ_AUX;
   "LBP_Axis14".SCC.CW1.TeststopStart := "DB1030_TEST_STOP".TEST_STP_INT_P_REQ_AUX;
   "LBP_Axis15".SCC.CW1.TeststopStart := "DB1030_TEST_STOP".TEST_STP_INT_P_REQ_AUX;
   "LBP_Axis16".SCC.CW1.TeststopStart := "DB1030_TEST_STOP".TEST_STP_INT_P_REQ_AUX;
   "LBP_Axis17".SCC.CW1.TeststopStart := "DB1030_TEST_STOP".TEST_STP_INT_P_REQ_AUX;
   "LBP_Axis18".SCC.CW1.TeststopStart := "DB1030_TEST_STOP".TEST_STP_INT_P_REQ_AUX;
   "LBP_Axis19".SCC.CW1.TeststopStart := "DB1030_TEST_STOP".TEST_STP_INT_P_REQ_AUX;
   "LBP_Axis20".SCC.CW1.TeststopStart := "DB1030_TEST_STOP".TEST_STP_INT_P_REQ_AUX;
   "LBP_Axis21".SCC.CW1.TeststopStart := "DB1030_TEST_STOP".TEST_STP_INT_P_REQ_AUX;
   "LBP_Axis22".SCC.CW1.TeststopStart := "DB1030_TEST_STOP".TEST_STP_INT_P_REQ_AUX;
   "LBP_Axis23".SCC.CW1.TeststopStart := "DB1030_TEST_STOP".TEST_STP_INT_P_REQ_AUX;
   "LBP_Axis24".SCC.CW1.TeststopStart := "DB1030_TEST_STOP".TEST_STP_INT_P_REQ_AUX;
   "LBP_Axis25".SCC.CW1.TeststopStart := "DB1030_TEST_STOP".TEST_STP_INT_P_REQ_AUX;
   "LBP_Axis26".SCC.CW1.TeststopStart := "DB1030_TEST_STOP".TEST_STP_INT_P_REQ_AUX;
   "LBP_Axis27".SCC.CW1.TeststopStart := "DB1030_TEST_STOP".TEST_STP_INT_P_REQ_AUX;
   "LBP_Axis28".SCC.CW1.TeststopStart := "DB1030_TEST_STOP".TEST_STP_INT_P_REQ_AUX;
   "LBP_Axis29".SCC.CW1.TeststopStart := "DB1030_TEST_STOP".TEST_STP_INT_P_REQ_AUX;
   "LBP_Axis30".SCC.CW1.TeststopStart := "DB1030_TEST_STOP".TEST_STP_INT_P_REQ_AUX;
   "LBP_Axis31".SCC.CW1.TeststopStart := "DB1030_TEST_STOP".TEST_STP_INT_P_REQ_AUX;
END_REGION

REGION Network 52: BRAKE TEST FAULT AXIS 1
   RUNG wire#powerrail
      Contact( "DB1031_X13_BRAKE_TEST".BRAKE_TEST_ERROR )
      wire#w1
      Contact( #BRAKE_TEST_AXIS_X13 )
      wire#w2
      Coil( "DB1030_TEST_STOP".TEST_STP_TST_BRK_F_AX_1 )
   END_RUNG
   RUNG wire#powerrail
      Contact( "DB1030_TEST_STOP".TEST_STP_SQ_TIME_EXCEEDED )
      Contact( "DB1030_TEST_STOP".TEST_STP_TST_BRK_AX_1 )
   END_RUNG wire#w1
   RUNG wire#powerrail
      Contact( "DB1030_TEST_STOP".TEST_STP_TST_BRK_F_AX_1 )
      I_Contact( "DB2120_MPP_ITC_IPC".RESET_FAULTS )
   END_RUNG wire#w1
   RUNG wire#w2
      Coil( "DB426_ALARMS_WARNINGS".ALARMS.GENERAL."700592" )
   END_RUNG
   // the same network as SCL:
   "DB1030_TEST_STOP".TEST_STP_TST_BRK_F_AX_1 := ("DB1031_X13_BRAKE_TEST".BRAKE_TEST_ERROR OR ("DB1030_TEST_STOP".TEST_STP_SQ_TIME_EXCEEDED AND "DB1030_TEST_STOP".TEST_STP_TST_BRK_AX_1) OR ("DB1030_TEST_STOP".TEST_STP_TST_BRK_F_AX_1 AND NOT "DB2120_MPP_ITC_IPC".RESET_FAULTS)) AND #BRAKE_TEST_AXIS_X13;
   "DB426_ALARMS_WARNINGS".ALARMS.GENERAL."700592" := "DB1030_TEST_STOP".TEST_STP_TST_BRK_F_AX_1;
END_REGION

REGION Network 53: BRAKE TEST FAULT AXIS 2
   RUNG wire#powerrail
      Contact( "DB1033_W11_BRAKE_TEST".BRAKE_TEST_ERROR )
      wire#w1
      Contact( #BRAKE_TEST_AXIS_W11 )
      wire#w2
      Coil( "DB1030_TEST_STOP".TEST_STP_TST_BRK_F_AX_2 )
   END_RUNG
   RUNG wire#powerrail
      Contact( "DB1030_TEST_STOP".TEST_STP_SQ_TIME_EXCEEDED )
      Contact( "DB1030_TEST_STOP".TEST_STP_TST_BRK_AX_2 )
   END_RUNG wire#w1
   RUNG wire#powerrail
      Contact( "DB1030_TEST_STOP".TEST_STP_TST_BRK_F_AX_2 )
      I_Contact( "DB2120_MPP_ITC_IPC".RESET_FAULTS )
   END_RUNG wire#w1
   RUNG wire#w2
      Coil( "DB426_ALARMS_WARNINGS".ALARMS.GENERAL."700593" )
   END_RUNG
   // the same network as SCL:
   "DB1030_TEST_STOP".TEST_STP_TST_BRK_F_AX_2 := ("DB1033_W11_BRAKE_TEST".BRAKE_TEST_ERROR OR ("DB1030_TEST_STOP".TEST_STP_SQ_TIME_EXCEEDED AND "DB1030_TEST_STOP".TEST_STP_TST_BRK_AX_2) OR ("DB1030_TEST_STOP".TEST_STP_TST_BRK_F_AX_2 AND NOT "DB2120_MPP_ITC_IPC".RESET_FAULTS)) AND #BRAKE_TEST_AXIS_W11;
   "DB426_ALARMS_WARNINGS".ALARMS.GENERAL."700593" := "DB1030_TEST_STOP".TEST_STP_TST_BRK_F_AX_2;
END_REGION

REGION Network 54: BRAKE TEST FAULT AXIS 3
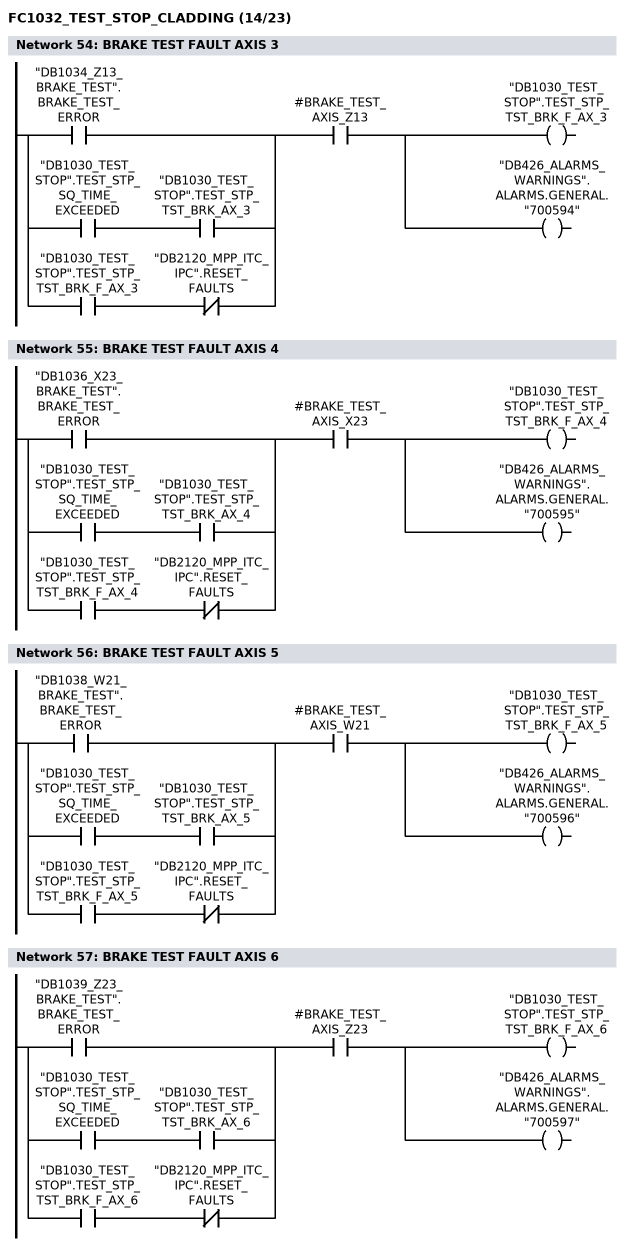
   RUNG wire#powerrail
      Contact( "DB1034_Z13_BRAKE_TEST".BRAKE_TEST_ERROR )
      wire#w1
      Contact( #BRAKE_TEST_AXIS_Z13 )
      wire#w2
      Coil( "DB1030_TEST_STOP".TEST_STP_TST_BRK_F_AX_3 )
   END_RUNG
   RUNG wire#powerrail
      Contact( "DB1030_TEST_STOP".TEST_STP_SQ_TIME_EXCEEDED )
      Contact( "DB1030_TEST_STOP".TEST_STP_TST_BRK_AX_3 )
   END_RUNG wire#w1
   RUNG wire#powerrail
      Contact( "DB1030_TEST_STOP".TEST_STP_TST_BRK_F_AX_3 )
      I_Contact( "DB2120_MPP_ITC_IPC".RESET_FAULTS )
   END_RUNG wire#w1
   RUNG wire#w2
      Coil( "DB426_ALARMS_WARNINGS".ALARMS.GENERAL."700594" )
   END_RUNG
   // the same network as SCL:
   "DB1030_TEST_STOP".TEST_STP_TST_BRK_F_AX_3 := ("DB1034_Z13_BRAKE_TEST".BRAKE_TEST_ERROR OR ("DB1030_TEST_STOP".TEST_STP_SQ_TIME_EXCEEDED AND "DB1030_TEST_STOP".TEST_STP_TST_BRK_AX_3) OR ("DB1030_TEST_STOP".TEST_STP_TST_BRK_F_AX_3 AND NOT "DB2120_MPP_ITC_IPC".RESET_FAULTS)) AND #BRAKE_TEST_AXIS_Z13;
   "DB426_ALARMS_WARNINGS".ALARMS.GENERAL."700594" := "DB1030_TEST_STOP".TEST_STP_TST_BRK_F_AX_3;
END_REGION

REGION Network 55: BRAKE TEST FAULT AXIS 4
   RUNG wire#powerrail
      Contact( "DB1036_X23_BRAKE_TEST".BRAKE_TEST_ERROR )
      wire#w1
      Contact( #BRAKE_TEST_AXIS_X23 )
      wire#w2
      Coil( "DB1030_TEST_STOP".TEST_STP_TST_BRK_F_AX_4 )
   END_RUNG
   RUNG wire#powerrail
      Contact( "DB1030_TEST_STOP".TEST_STP_SQ_TIME_EXCEEDED )
      Contact( "DB1030_TEST_STOP".TEST_STP_TST_BRK_AX_4 )
   END_RUNG wire#w1
   RUNG wire#powerrail
      Contact( "DB1030_TEST_STOP".TEST_STP_TST_BRK_F_AX_4 )
      I_Contact( "DB2120_MPP_ITC_IPC".RESET_FAULTS )
   END_RUNG wire#w1
   RUNG wire#w2
      Coil( "DB426_ALARMS_WARNINGS".ALARMS.GENERAL."700595" )
   END_RUNG
   // the same network as SCL:
   "DB1030_TEST_STOP".TEST_STP_TST_BRK_F_AX_4 := ("DB1036_X23_BRAKE_TEST".BRAKE_TEST_ERROR OR ("DB1030_TEST_STOP".TEST_STP_SQ_TIME_EXCEEDED AND "DB1030_TEST_STOP".TEST_STP_TST_BRK_AX_4) OR ("DB1030_TEST_STOP".TEST_STP_TST_BRK_F_AX_4 AND NOT "DB2120_MPP_ITC_IPC".RESET_FAULTS)) AND #BRAKE_TEST_AXIS_X23;
   "DB426_ALARMS_WARNINGS".ALARMS.GENERAL."700595" := "DB1030_TEST_STOP".TEST_STP_TST_BRK_F_AX_4;
END_REGION

REGION Network 56: BRAKE TEST FAULT AXIS 5
   RUNG wire#powerrail
      Contact( "DB1038_W21_BRAKE_TEST".BRAKE_TEST_ERROR )
      wire#w1
      Contact( #BRAKE_TEST_AXIS_W21 )
      wire#w2
      Coil( "DB1030_TEST_STOP".TEST_STP_TST_BRK_F_AX_5 )
   END_RUNG
   RUNG wire#powerrail
      Contact( "DB1030_TEST_STOP".TEST_STP_SQ_TIME_EXCEEDED )
      Contact( "DB1030_TEST_STOP".TEST_STP_TST_BRK_AX_5 )
   END_RUNG wire#w1
   RUNG wire#powerrail
      Contact( "DB1030_TEST_STOP".TEST_STP_TST_BRK_F_AX_5 )
      I_Contact( "DB2120_MPP_ITC_IPC".RESET_FAULTS )
   END_RUNG wire#w1
   RUNG wire#w2
      Coil( "DB426_ALARMS_WARNINGS".ALARMS.GENERAL."700596" )
   END_RUNG
   // the same network as SCL:
   "DB1030_TEST_STOP".TEST_STP_TST_BRK_F_AX_5 := ("DB1038_W21_BRAKE_TEST".BRAKE_TEST_ERROR OR ("DB1030_TEST_STOP".TEST_STP_SQ_TIME_EXCEEDED AND "DB1030_TEST_STOP".TEST_STP_TST_BRK_AX_5) OR ("DB1030_TEST_STOP".TEST_STP_TST_BRK_F_AX_5 AND NOT "DB2120_MPP_ITC_IPC".RESET_FAULTS)) AND #BRAKE_TEST_AXIS_W21;
   "DB426_ALARMS_WARNINGS".ALARMS.GENERAL."700596" := "DB1030_TEST_STOP".TEST_STP_TST_BRK_F_AX_5;
END_REGION

REGION Network 57: BRAKE TEST FAULT AXIS 6
   RUNG wire#powerrail
      Contact( "DB1039_Z23_BRAKE_TEST".BRAKE_TEST_ERROR )
      wire#w1
      Contact( #BRAKE_TEST_AXIS_Z23 )
      wire#w2
      Coil( "DB1030_TEST_STOP".TEST_STP_TST_BRK_F_AX_6 )
   END_RUNG
   RUNG wire#powerrail
      Contact( "DB1030_TEST_STOP".TEST_STP_SQ_TIME_EXCEEDED )
      Contact( "DB1030_TEST_STOP".TEST_STP_TST_BRK_AX_6 )
   END_RUNG wire#w1
   RUNG wire#powerrail
      Contact( "DB1030_TEST_STOP".TEST_STP_TST_BRK_F_AX_6 )
      I_Contact( "DB2120_MPP_ITC_IPC".RESET_FAULTS )
   END_RUNG wire#w1
   RUNG wire#w2
      Coil( "DB426_ALARMS_WARNINGS".ALARMS.GENERAL."700597" )
   END_RUNG
   // the same network as SCL:
   "DB1030_TEST_STOP".TEST_STP_TST_BRK_F_AX_6 := ("DB1039_Z23_BRAKE_TEST".BRAKE_TEST_ERROR OR ("DB1030_TEST_STOP".TEST_STP_SQ_TIME_EXCEEDED AND "DB1030_TEST_STOP".TEST_STP_TST_BRK_AX_6) OR ("DB1030_TEST_STOP".TEST_STP_TST_BRK_F_AX_6 AND NOT "DB2120_MPP_ITC_IPC".RESET_FAULTS)) AND #BRAKE_TEST_AXIS_Z23;
   "DB426_ALARMS_WARNINGS".ALARMS.GENERAL."700597" := "DB1030_TEST_STOP".TEST_STP_TST_BRK_F_AX_6;
END_REGION

REGION Network 58: BRAKE TEST FAULT AXIS 7
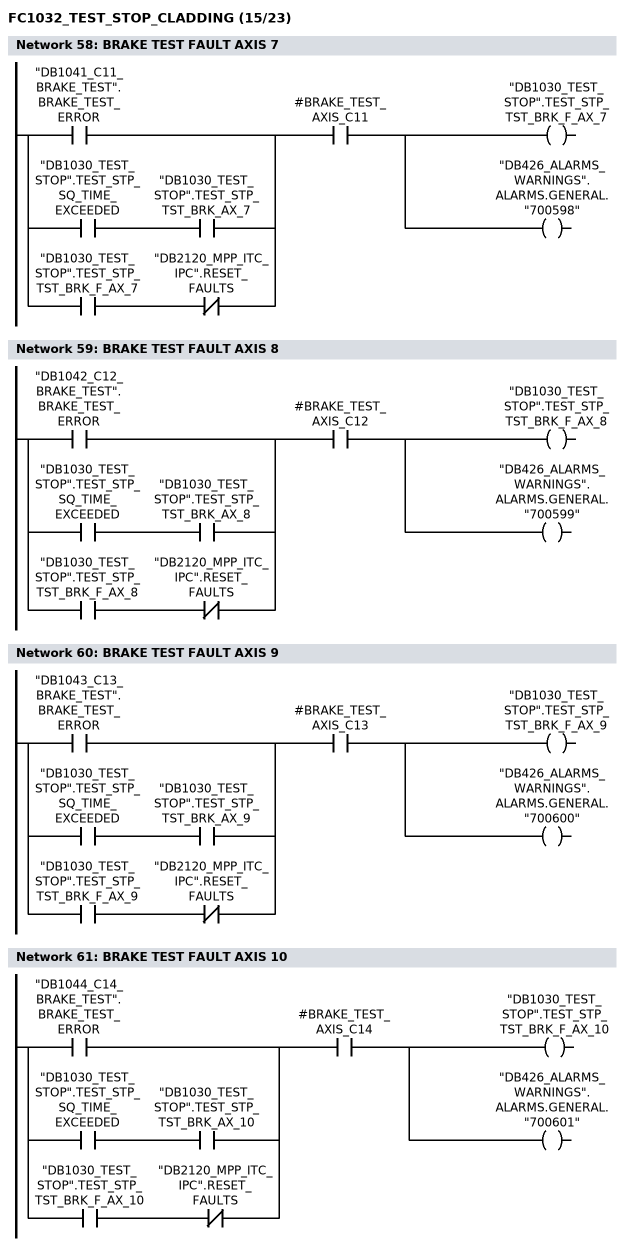
   RUNG wire#powerrail
      Contact( "DB1041_C11_BRAKE_TEST".BRAKE_TEST_ERROR )
      wire#w1
      Contact( #BRAKE_TEST_AXIS_C11 )
      wire#w2
      Coil( "DB1030_TEST_STOP".TEST_STP_TST_BRK_F_AX_7 )
   END_RUNG
   RUNG wire#powerrail
      Contact( "DB1030_TEST_STOP".TEST_STP_SQ_TIME_EXCEEDED )
      Contact( "DB1030_TEST_STOP".TEST_STP_TST_BRK_AX_7 )
   END_RUNG wire#w1
   RUNG wire#powerrail
      Contact( "DB1030_TEST_STOP".TEST_STP_TST_BRK_F_AX_7 )
      I_Contact( "DB2120_MPP_ITC_IPC".RESET_FAULTS )
   END_RUNG wire#w1
   RUNG wire#w2
      Coil( "DB426_ALARMS_WARNINGS".ALARMS.GENERAL."700598" )
   END_RUNG
   // the same network as SCL:
   "DB1030_TEST_STOP".TEST_STP_TST_BRK_F_AX_7 := ("DB1041_C11_BRAKE_TEST".BRAKE_TEST_ERROR OR ("DB1030_TEST_STOP".TEST_STP_SQ_TIME_EXCEEDED AND "DB1030_TEST_STOP".TEST_STP_TST_BRK_AX_7) OR ("DB1030_TEST_STOP".TEST_STP_TST_BRK_F_AX_7 AND NOT "DB2120_MPP_ITC_IPC".RESET_FAULTS)) AND #BRAKE_TEST_AXIS_C11;
   "DB426_ALARMS_WARNINGS".ALARMS.GENERAL."700598" := "DB1030_TEST_STOP".TEST_STP_TST_BRK_F_AX_7;
END_REGION

REGION Network 59: BRAKE TEST FAULT AXIS 8
   RUNG wire#powerrail
      Contact( "DB1042_C12_BRAKE_TEST".BRAKE_TEST_ERROR )
      wire#w1
      Contact( #BRAKE_TEST_AXIS_C12 )
      wire#w2
      Coil( "DB1030_TEST_STOP".TEST_STP_TST_BRK_F_AX_8 )
   END_RUNG
   RUNG wire#powerrail
      Contact( "DB1030_TEST_STOP".TEST_STP_SQ_TIME_EXCEEDED )
      Contact( "DB1030_TEST_STOP".TEST_STP_TST_BRK_AX_8 )
   END_RUNG wire#w1
   RUNG wire#powerrail
      Contact( "DB1030_TEST_STOP".TEST_STP_TST_BRK_F_AX_8 )
      I_Contact( "DB2120_MPP_ITC_IPC".RESET_FAULTS )
   END_RUNG wire#w1
   RUNG wire#w2
      Coil( "DB426_ALARMS_WARNINGS".ALARMS.GENERAL."700599" )
   END_RUNG
   // the same network as SCL:
   "DB1030_TEST_STOP".TEST_STP_TST_BRK_F_AX_8 := ("DB1042_C12_BRAKE_TEST".BRAKE_TEST_ERROR OR ("DB1030_TEST_STOP".TEST_STP_SQ_TIME_EXCEEDED AND "DB1030_TEST_STOP".TEST_STP_TST_BRK_AX_8) OR ("DB1030_TEST_STOP".TEST_STP_TST_BRK_F_AX_8 AND NOT "DB2120_MPP_ITC_IPC".RESET_FAULTS)) AND #BRAKE_TEST_AXIS_C12;
   "DB426_ALARMS_WARNINGS".ALARMS.GENERAL."700599" := "DB1030_TEST_STOP".TEST_STP_TST_BRK_F_AX_8;
END_REGION

REGION Network 60: BRAKE TEST FAULT AXIS 9
   RUNG wire#powerrail
      Contact( "DB1043_C13_BRAKE_TEST".BRAKE_TEST_ERROR )
      wire#w1
      Contact( #BRAKE_TEST_AXIS_C13 )
      wire#w2
      Coil( "DB1030_TEST_STOP".TEST_STP_TST_BRK_F_AX_9 )
   END_RUNG
   RUNG wire#powerrail
      Contact( "DB1030_TEST_STOP".TEST_STP_SQ_TIME_EXCEEDED )
      Contact( "DB1030_TEST_STOP".TEST_STP_TST_BRK_AX_9 )
   END_RUNG wire#w1
   RUNG wire#powerrail
      Contact( "DB1030_TEST_STOP".TEST_STP_TST_BRK_F_AX_9 )
      I_Contact( "DB2120_MPP_ITC_IPC".RESET_FAULTS )
   END_RUNG wire#w1
   RUNG wire#w2
      Coil( "DB426_ALARMS_WARNINGS".ALARMS.GENERAL."700600" )
   END_RUNG
   // the same network as SCL:
   "DB1030_TEST_STOP".TEST_STP_TST_BRK_F_AX_9 := ("DB1043_C13_BRAKE_TEST".BRAKE_TEST_ERROR OR ("DB1030_TEST_STOP".TEST_STP_SQ_TIME_EXCEEDED AND "DB1030_TEST_STOP".TEST_STP_TST_BRK_AX_9) OR ("DB1030_TEST_STOP".TEST_STP_TST_BRK_F_AX_9 AND NOT "DB2120_MPP_ITC_IPC".RESET_FAULTS)) AND #BRAKE_TEST_AXIS_C13;
   "DB426_ALARMS_WARNINGS".ALARMS.GENERAL."700600" := "DB1030_TEST_STOP".TEST_STP_TST_BRK_F_AX_9;
END_REGION

REGION Network 61: BRAKE TEST FAULT AXIS 10
   RUNG wire#powerrail
      Contact( "DB1044_C14_BRAKE_TEST".BRAKE_TEST_ERROR )
      wire#w1
      Contact( #BRAKE_TEST_AXIS_C14 )
      wire#w2
      Coil( "DB1030_TEST_STOP".TEST_STP_TST_BRK_F_AX_10 )
   END_RUNG
   RUNG wire#powerrail
      Contact( "DB1030_TEST_STOP".TEST_STP_SQ_TIME_EXCEEDED )
      Contact( "DB1030_TEST_STOP".TEST_STP_TST_BRK_AX_10 )
   END_RUNG wire#w1
   RUNG wire#powerrail
      Contact( "DB1030_TEST_STOP".TEST_STP_TST_BRK_F_AX_10 )
      I_Contact( "DB2120_MPP_ITC_IPC".RESET_FAULTS )
   END_RUNG wire#w1
   RUNG wire#w2
      Coil( "DB426_ALARMS_WARNINGS".ALARMS.GENERAL."700601" )
   END_RUNG
   // the same network as SCL:
   "DB1030_TEST_STOP".TEST_STP_TST_BRK_F_AX_10 := ("DB1044_C14_BRAKE_TEST".BRAKE_TEST_ERROR OR ("DB1030_TEST_STOP".TEST_STP_SQ_TIME_EXCEEDED AND "DB1030_TEST_STOP".TEST_STP_TST_BRK_AX_10) OR ("DB1030_TEST_STOP".TEST_STP_TST_BRK_F_AX_10 AND NOT "DB2120_MPP_ITC_IPC".RESET_FAULTS)) AND #BRAKE_TEST_AXIS_C14;
   "DB426_ALARMS_WARNINGS".ALARMS.GENERAL."700601" := "DB1030_TEST_STOP".TEST_STP_TST_BRK_F_AX_10;
END_REGION

REGION Network 62: BRAKE TEST FAULT AXIS 11
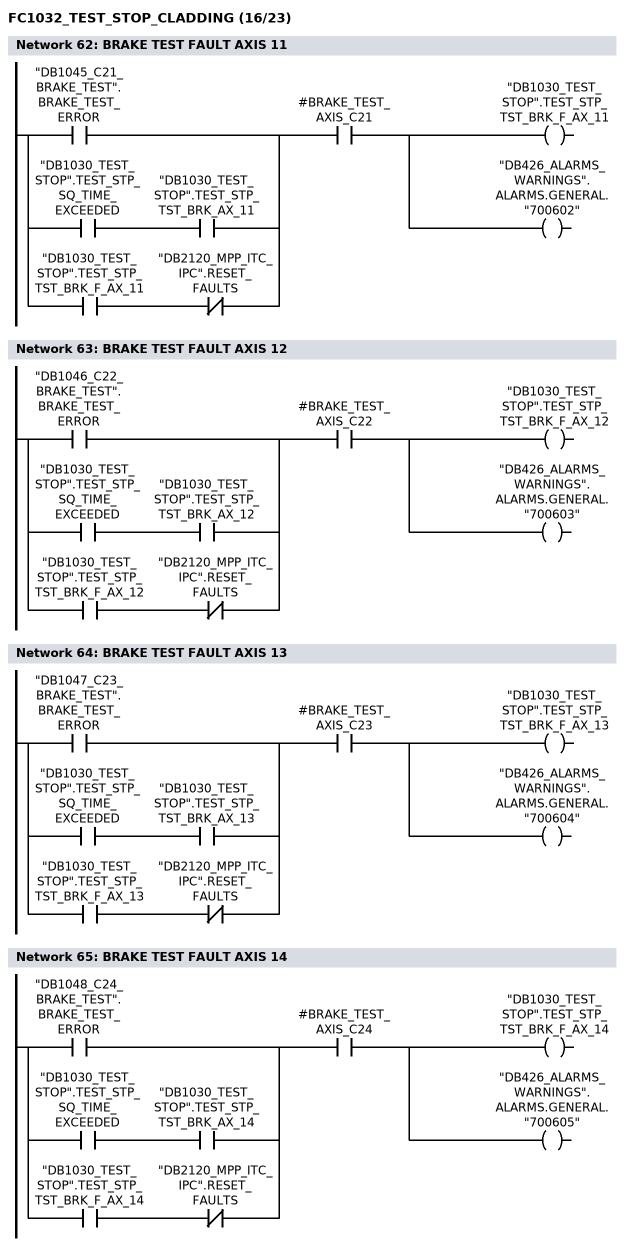
   RUNG wire#powerrail
      Contact( "DB1045_C21_BRAKE_TEST".BRAKE_TEST_ERROR )
      wire#w1
      Contact( #BRAKE_TEST_AXIS_C21 )
      wire#w2
      Coil( "DB1030_TEST_STOP".TEST_STP_TST_BRK_F_AX_11 )
   END_RUNG
   RUNG wire#powerrail
      Contact( "DB1030_TEST_STOP".TEST_STP_SQ_TIME_EXCEEDED )
      Contact( "DB1030_TEST_STOP".TEST_STP_TST_BRK_AX_11 )
   END_RUNG wire#w1
   RUNG wire#powerrail
      Contact( "DB1030_TEST_STOP".TEST_STP_TST_BRK_F_AX_11 )
      I_Contact( "DB2120_MPP_ITC_IPC".RESET_FAULTS )
   END_RUNG wire#w1
   RUNG wire#w2
      Coil( "DB426_ALARMS_WARNINGS".ALARMS.GENERAL."700602" )
   END_RUNG
   // the same network as SCL:
   "DB1030_TEST_STOP".TEST_STP_TST_BRK_F_AX_11 := ("DB1045_C21_BRAKE_TEST".BRAKE_TEST_ERROR OR ("DB1030_TEST_STOP".TEST_STP_SQ_TIME_EXCEEDED AND "DB1030_TEST_STOP".TEST_STP_TST_BRK_AX_11) OR ("DB1030_TEST_STOP".TEST_STP_TST_BRK_F_AX_11 AND NOT "DB2120_MPP_ITC_IPC".RESET_FAULTS)) AND #BRAKE_TEST_AXIS_C21;
   "DB426_ALARMS_WARNINGS".ALARMS.GENERAL."700602" := "DB1030_TEST_STOP".TEST_STP_TST_BRK_F_AX_11;
END_REGION

